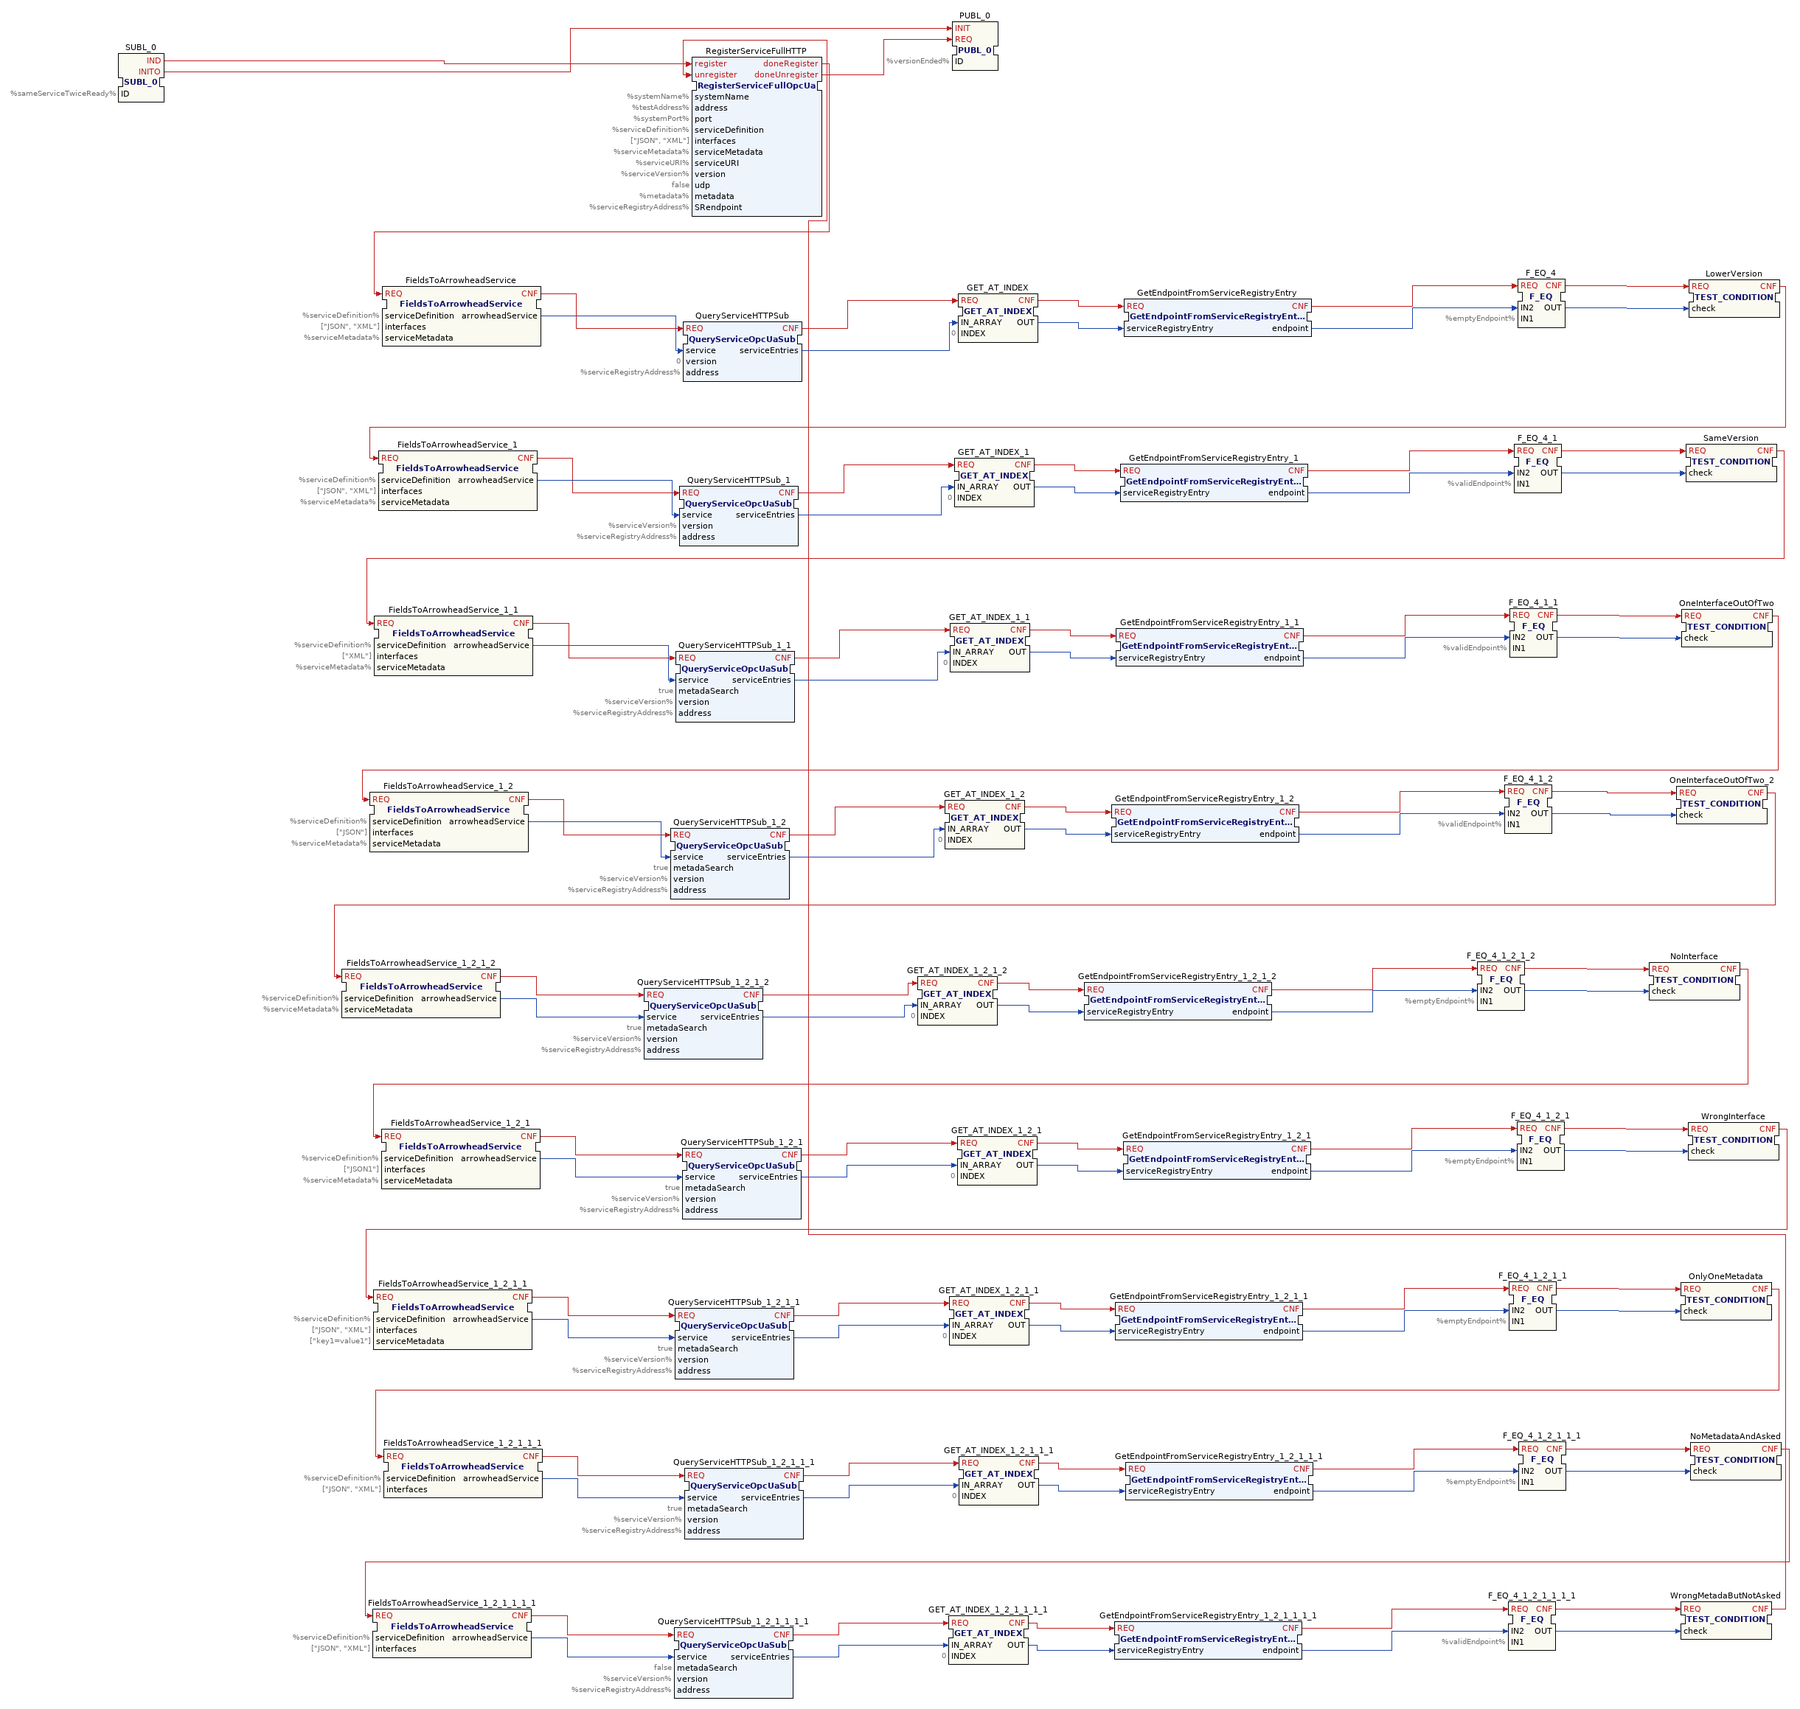
    [picture p25: application OpcUaTest5VersionAndMetadata]
    FBS
      FieldsToArrowheadService : FieldsToArrowheadService(serviceDefinition := %serviceDefinition%, interfaces := ["JSON", "XML"], serviceMetadata := %serviceMetadata%);
      GET_AT_INDEX : GET_AT_INDEX(INDEX := 0);
      F_EQ_4 : F_EQ(IN1 := %emptyEndpoint%);
      LowerVersion : TEST_CONDITION;
      FieldsToArrowheadService_1 : FieldsToArrowheadService(serviceDefinition := %serviceDefinition%, interfaces := ["JSON", "XML"], serviceMetadata := %serviceMetadata%);
      SameVersion : TEST_CONDITION;
      GET_AT_INDEX_1 : GET_AT_INDEX(INDEX := 0);
      F_EQ_4_1 : F_EQ(IN1 := %validEndpoint%);
      OneInterfaceOutOfTwo : TEST_CONDITION;
      F_EQ_4_1_1 : F_EQ(IN1 := %validEndpoint%);
      FieldsToArrowheadService_1_1 : FieldsToArrowheadService(serviceDefinition := %serviceDefinition%, interfaces := ["XML"], serviceMetadata := %serviceMetadata%);
      GET_AT_INDEX_1_1 : GET_AT_INDEX(INDEX := 0);
      OneInterfaceOutOfTwo_2 : TEST_CONDITION;
      F_EQ_4_1_2 : F_EQ(IN1 := %validEndpoint%);
      FieldsToArrowheadService_1_2 : FieldsToArrowheadService(serviceDefinition := %serviceDefinition%, interfaces := ["JSON"], serviceMetadata := %serviceMetadata%);
      GET_AT_INDEX_1_2 : GET_AT_INDEX(INDEX := 0);
      WrongInterface : TEST_CONDITION;
      GET_AT_INDEX_1_2_1 : GET_AT_INDEX(INDEX := 0);
      FieldsToArrowheadService_1_2_1 : FieldsToArrowheadService(serviceDefinition := %serviceDefinition%, interfaces := ["JSON1"], serviceMetadata := %serviceMetadata%);
      F_EQ_4_1_2_1 : F_EQ(IN1 := %emptyEndpoint%);
      SUBL_0 : SUBL_0(ID := %sameServiceTwiceReady%);
      OnlyOneMetadata : TEST_CONDITION;
      F_EQ_4_1_2_1_1 : F_EQ(IN1 := %emptyEndpoint%);
      FieldsToArrowheadService_1_2_1_1 : FieldsToArrowheadService(serviceDefinition := %serviceDefinition%, interfaces := ["JSON", "XML"], serviceMetadata := ["key1=value1"]);
      GET_AT_INDEX_1_2_1_1 : GET_AT_INDEX(INDEX := 0);
      FieldsToArrowheadService_1_2_1_1_1 : FieldsToArrowheadService(serviceDefinition := %serviceDefinition%, interfaces := ["JSON", "XML"]);
      F_EQ_4_1_2_1_1_1 : F_EQ(IN1 := %emptyEndpoint%);
      GET_AT_INDEX_1_2_1_1_1 : GET_AT_INDEX(INDEX := 0);
      NoMetadataAndAsked : TEST_CONDITION;
      F_EQ_4_1_2_1_2 : F_EQ(IN1 := %emptyEndpoint%);
      GET_AT_INDEX_1_2_1_2 : GET_AT_INDEX(INDEX := 0);
      FieldsToArrowheadService_1_2_1_2 : FieldsToArrowheadService(serviceDefinition := %serviceDefinition%, serviceMetadata := %serviceMetadata%);
      NoInterface : TEST_CONDITION;
      GET_AT_INDEX_1_2_1_1_1_1 : GET_AT_INDEX(INDEX := 0);
      F_EQ_4_1_2_1_1_1_1 : F_EQ(IN1 := %validEndpoint%);
      WrongMetadaButNotAsked : TEST_CONDITION;
      FieldsToArrowheadService_1_2_1_1_1_1 : FieldsToArrowheadService(serviceDefinition := %serviceDefinition%, interfaces := ["JSON", "XML"]);
      PUBL_0 : PUBL_0(ID := %versionEnded%);
    END_FBS
    SUBAPPS
      GetEndpointFromServiceRegistryEntry : GetEndpointFromServiceRegistryEntry;
      GetEndpointFromServiceRegistryEntry_1 : GetEndpointFromServiceRegistryEntry;
      GetEndpointFromServiceRegistryEntry_1_1 : GetEndpointFromServiceRegistryEntry;
      GetEndpointFromServiceRegistryEntry_1_2 : GetEndpointFromServiceRegistryEntry;
      GetEndpointFromServiceRegistryEntry_1_2_1 : GetEndpointFromServiceRegistryEntry;
      GetEndpointFromServiceRegistryEntry_1_2_1_1 : GetEndpointFromServiceRegistryEntry;
      GetEndpointFromServiceRegistryEntry_1_2_1_1_1 : GetEndpointFromServiceRegistryEntry;
      GetEndpointFromServiceRegistryEntry_1_2_1_2 : GetEndpointFromServiceRegistryEntry;
      GetEndpointFromServiceRegistryEntry_1_2_1_1_1_1 : GetEndpointFromServiceRegistryEntry;
      RegisterServiceFullHTTP : RegisterServiceFullOpcUa(systemName := %systemName%, address := %testAddress%, port := %systemPort%, serviceDefinition := %serviceDefinition%, interfaces := ["JSON", "XML"], serviceMetadata := %serviceMetadata%, serviceURI := %serviceURI%, version := %serviceVersion%, udp := false, metadata := %metadata%, SRendpoint := %serviceRegistryAddress%);
      QueryServiceHTTPSub : QueryServiceOpcUaSub(version := 0, address := %serviceRegistryAddress%);
      QueryServiceHTTPSub_1 : QueryServiceOpcUaSub(version := %serviceVersion%, address := %serviceRegistryAddress%);
      QueryServiceHTTPSub_1_1 : QueryServiceOpcUaSub(metadaSearch := true, version := %serviceVersion%, address := %serviceRegistryAddress%);
      QueryServiceHTTPSub_1_2 : QueryServiceOpcUaSub(metadaSearch := true, version := %serviceVersion%, address := %serviceRegistryAddress%);
      QueryServiceHTTPSub_1_2_1_2 : QueryServiceOpcUaSub(metadaSearch := true, version := %serviceVersion%, address := %serviceRegistryAddress%);
      QueryServiceHTTPSub_1_2_1 : QueryServiceOpcUaSub(metadaSearch := true, version := %serviceVersion%, address := %serviceRegistryAddress%);
      QueryServiceHTTPSub_1_2_1_1 : QueryServiceOpcUaSub(metadaSearch := true, version := %serviceVersion%, address := %serviceRegistryAddress%);
      QueryServiceHTTPSub_1_2_1_1_1 : QueryServiceOpcUaSub(metadaSearch := true, version := %serviceVersion%, address := %serviceRegistryAddress%);
      QueryServiceHTTPSub_1_2_1_1_1_1 : QueryServiceOpcUaSub(metadaSearch := false, version := %serviceVersion%, address := %serviceRegistryAddress%);
    END_SUBAPPS
    EVENT_CONNECTIONS
      GET_AT_INDEX.CNF TO GetEndpointFromServiceRegistryEntry.REQ;
      F_EQ_4.CNF TO LowerVersion.REQ;
      GetEndpointFromServiceRegistryEntry.CNF TO F_EQ_4.REQ;
      F_EQ_4_1.CNF TO SameVersion.REQ;
      GetEndpointFromServiceRegistryEntry_1.CNF TO F_EQ_4_1.REQ;
      GET_AT_INDEX_1.CNF TO GetEndpointFromServiceRegistryEntry_1.REQ;
      GET_AT_INDEX_1_1.CNF TO GetEndpointFromServiceRegistryEntry_1_1.REQ;
      GetEndpointFromServiceRegistryEntry_1_1.CNF TO F_EQ_4_1_1.REQ;
      F_EQ_4_1_1.CNF TO OneInterfaceOutOfTwo.REQ;
      GET_AT_INDEX_1_2.CNF TO GetEndpointFromServiceRegistryEntry_1_2.REQ;
      GetEndpointFromServiceRegistryEntry_1_2.CNF TO F_EQ_4_1_2.REQ;
      F_EQ_4_1_2.CNF TO OneInterfaceOutOfTwo_2.REQ;
      F_EQ_4_1_2_1.CNF TO WrongInterface.REQ;
      GET_AT_INDEX_1_2_1.CNF TO GetEndpointFromServiceRegistryEntry_1_2_1.REQ;
      GetEndpointFromServiceRegistryEntry_1_2_1.CNF TO F_EQ_4_1_2_1.REQ;
      GET_AT_INDEX_1_2_1_1.CNF TO GetEndpointFromServiceRegistryEntry_1_2_1_1.REQ;
      GetEndpointFromServiceRegistryEntry_1_2_1_1.CNF TO F_EQ_4_1_2_1_1.REQ;
      F_EQ_4_1_2_1_1.CNF TO OnlyOneMetadata.REQ;
      F_EQ_4_1_2_1_1_1.CNF TO NoMetadataAndAsked.REQ;
      GetEndpointFromServiceRegistryEntry_1_2_1_1_1.CNF TO F_EQ_4_1_2_1_1_1.REQ;
      GET_AT_INDEX_1_2_1_1_1.CNF TO GetEndpointFromServiceRegistryEntry_1_2_1_1_1.REQ;
      F_EQ_4_1_2_1_2.CNF TO NoInterface.REQ;
      GET_AT_INDEX_1_2_1_2.CNF TO GetEndpointFromServiceRegistryEntry_1_2_1_2.REQ;
      GetEndpointFromServiceRegistryEntry_1_2_1_2.CNF TO F_EQ_4_1_2_1_2.REQ;
      GET_AT_INDEX_1_2_1_1_1_1.CNF TO GetEndpointFromServiceRegistryEntry_1_2_1_1_1_1.REQ;
      F_EQ_4_1_2_1_1_1_1.CNF TO WrongMetadaButNotAsked.REQ;
      GetEndpointFromServiceRegistryEntry_1_2_1_1_1_1.CNF TO F_EQ_4_1_2_1_1_1_1.REQ;
      LowerVersion.CNF TO FieldsToArrowheadService_1.REQ;
      SameVersion.CNF TO FieldsToArrowheadService_1_1.REQ;
      OneInterfaceOutOfTwo.CNF TO FieldsToArrowheadService_1_2.REQ;
      OneInterfaceOutOfTwo_2.CNF TO FieldsToArrowheadService_1_2_1_2.REQ;
      NoInterface.CNF TO FieldsToArrowheadService_1_2_1.REQ;
      WrongInterface.CNF TO FieldsToArrowheadService_1_2_1_1.REQ;
      OnlyOneMetadata.CNF TO FieldsToArrowheadService_1_2_1_1_1.REQ;
      NoMetadataAndAsked.CNF TO FieldsToArrowheadService_1_2_1_1_1_1.REQ;
      SUBL_0.IND TO RegisterServiceFullHTTP.register;
      WrongMetadaButNotAsked.CNF TO RegisterServiceFullHTTP.unregister;
      RegisterServiceFullHTTP.doneRegister TO FieldsToArrowheadService.REQ;
      FieldsToArrowheadService.CNF TO QueryServiceHTTPSub.REQ;
      QueryServiceHTTPSub.CNF TO GET_AT_INDEX.REQ;
      FieldsToArrowheadService_1.CNF TO QueryServiceHTTPSub_1.REQ;
      QueryServiceHTTPSub_1.CNF TO GET_AT_INDEX_1.REQ;
      FieldsToArrowheadService_1_1.CNF TO QueryServiceHTTPSub_1_1.REQ;
      QueryServiceHTTPSub_1_1.CNF TO GET_AT_INDEX_1_1.REQ;
      FieldsToArrowheadService_1_2.CNF TO QueryServiceHTTPSub_1_2.REQ;
      QueryServiceHTTPSub_1_2.CNF TO GET_AT_INDEX_1_2.REQ;
      FieldsToArrowheadService_1_2_1_2.CNF TO QueryServiceHTTPSub_1_2_1_2.REQ;
      QueryServiceHTTPSub_1_2_1_2.CNF TO GET_AT_INDEX_1_2_1_2.REQ;
      FieldsToArrowheadService_1_2_1.CNF TO QueryServiceHTTPSub_1_2_1.REQ;
      QueryServiceHTTPSub_1_2_1.CNF TO GET_AT_INDEX_1_2_1.REQ;
      FieldsToArrowheadService_1_2_1_1.CNF TO QueryServiceHTTPSub_1_2_1_1.REQ;
      QueryServiceHTTPSub_1_2_1_1.CNF TO GET_AT_INDEX_1_2_1_1.REQ;
      FieldsToArrowheadService_1_2_1_1_1.CNF TO QueryServiceHTTPSub_1_2_1_1_1.REQ;
      QueryServiceHTTPSub_1_2_1_1_1.CNF TO GET_AT_INDEX_1_2_1_1_1.REQ;
      FieldsToArrowheadService_1_2_1_1_1_1.CNF TO QueryServiceHTTPSub_1_2_1_1_1_1.REQ;
      QueryServiceHTTPSub_1_2_1_1_1_1.CNF TO GET_AT_INDEX_1_2_1_1_1_1.REQ;
      SUBL_0.INITO TO PUBL_0.INIT;
      RegisterServiceFullHTTP.doneUnregister TO PUBL_0.REQ;
    END_CONNECTIONS
    DATA_CONNECTIONS
      GET_AT_INDEX.OUT TO GetEndpointFromServiceRegistryEntry.serviceRegistryEntry;
      F_EQ_4.OUT TO LowerVersion.check;
      GetEndpointFromServiceRegistryEntry.endpoint TO F_EQ_4.IN2;
      GetEndpointFromServiceRegistryEntry_1.endpoint TO F_EQ_4_1.IN2;
      F_EQ_4_1.OUT TO SameVersion.check;
      GET_AT_INDEX_1.OUT TO GetEndpointFromServiceRegistryEntry_1.serviceRegistryEntry;
      GET_AT_INDEX_1_1.OUT TO GetEndpointFromServiceRegistryEntry_1_1.serviceRegistryEntry;
      F_EQ_4_1_1.OUT TO OneInterfaceOutOfTwo.check;
      GetEndpointFromServiceRegistryEntry_1_1.endpoint TO F_EQ_4_1_1.IN2;
      GET_AT_INDEX_1_2.OUT TO GetEndpointFromServiceRegistryEntry_1_2.serviceRegistryEntry;
      F_EQ_4_1_2.OUT TO OneInterfaceOutOfTwo_2.check;
      GetEndpointFromServiceRegistryEntry_1_2.endpoint TO F_EQ_4_1_2.IN2;
      GetEndpointFromServiceRegistryEntry_1_2_1.endpoint TO F_EQ_4_1_2_1.IN2;
      F_EQ_4_1_2_1.OUT TO WrongInterface.check;
      GET_AT_INDEX_1_2_1.OUT TO GetEndpointFromServiceRegistryEntry_1_2_1.serviceRegistryEntry;
      F_EQ_4_1_2_1_1.OUT TO OnlyOneMetadata.check;
      GET_AT_INDEX_1_2_1_1.OUT TO GetEndpointFromServiceRegistryEntry_1_2_1_1.serviceRegistryEntry;
      GetEndpointFromServiceRegistryEntry_1_2_1_1.endpoint TO F_EQ_4_1_2_1_1.IN2;
      F_EQ_4_1_2_1_1_1.OUT TO NoMetadataAndAsked.check;
      GET_AT_INDEX_1_2_1_1_1.OUT TO GetEndpointFromServiceRegistryEntry_1_2_1_1_1.serviceRegistryEntry;
      GetEndpointFromServiceRegistryEntry_1_2_1_1_1.endpoint TO F_EQ_4_1_2_1_1_1.IN2;
      F_EQ_4_1_2_1_2.OUT TO NoInterface.check;
      GET_AT_INDEX_1_2_1_2.OUT TO GetEndpointFromServiceRegistryEntry_1_2_1_2.serviceRegistryEntry;
      GetEndpointFromServiceRegistryEntry_1_2_1_2.endpoint TO F_EQ_4_1_2_1_2.IN2;
      GET_AT_INDEX_1_2_1_1_1_1.OUT TO GetEndpointFromServiceRegistryEntry_1_2_1_1_1_1.serviceRegistryEntry;
      GetEndpointFromServiceRegistryEntry_1_2_1_1_1_1.endpoint TO F_EQ_4_1_2_1_1_1_1.IN2;
      F_EQ_4_1_2_1_1_1_1.OUT TO WrongMetadaButNotAsked.check;
      FieldsToArrowheadService.arrowheadService TO QueryServiceHTTPSub.service;
      QueryServiceHTTPSub.serviceEntries TO GET_AT_INDEX.IN_ARRAY;
      FieldsToArrowheadService_1.arrowheadService TO QueryServiceHTTPSub_1.service;
      QueryServiceHTTPSub_1.serviceEntries TO GET_AT_INDEX_1.IN_ARRAY;
      FieldsToArrowheadService_1_1.arrowheadService TO QueryServiceHTTPSub_1_1.service;
      QueryServiceHTTPSub_1_1.serviceEntries TO GET_AT_INDEX_1_1.IN_ARRAY;
      FieldsToArrowheadService_1_2.arrowheadService TO QueryServiceHTTPSub_1_2.service;
      QueryServiceHTTPSub_1_2.serviceEntries TO GET_AT_INDEX_1_2.IN_ARRAY;
      FieldsToArrowheadService_1_2_1_2.arrowheadService TO QueryServiceHTTPSub_1_2_1_2.service;
      QueryServiceHTTPSub_1_2_1_2.serviceEntries TO GET_AT_INDEX_1_2_1_2.IN_ARRAY;
      FieldsToArrowheadService_1_2_1.arrowheadService TO QueryServiceHTTPSub_1_2_1.service;
      QueryServiceHTTPSub_1_2_1.serviceEntries TO GET_AT_INDEX_1_2_1.IN_ARRAY;
      FieldsToArrowheadService_1_2_1_1.arrowheadService TO QueryServiceHTTPSub_1_2_1_1.service;
      QueryServiceHTTPSub_1_2_1_1.serviceEntries TO GET_AT_INDEX_1_2_1_1.IN_ARRAY;
      FieldsToArrowheadService_1_2_1_1_1.arrowheadService TO QueryServiceHTTPSub_1_2_1_1_1.service;
      QueryServiceHTTPSub_1_2_1_1_1.serviceEntries TO GET_AT_INDEX_1_2_1_1_1.IN_ARRAY;
      FieldsToArrowheadService_1_2_1_1_1_1.arrowheadService TO QueryServiceHTTPSub_1_2_1_1_1_1.service;
      QueryServiceHTTPSub_1_2_1_1_1_1.serviceEntries TO GET_AT_INDEX_1_2_1_1_1_1.IN_ARRAY;
    END_CONNECTIONS
  END_APPLICATION
  APPLICATION OpcUaTest6RegisterMoreServiceSubApp
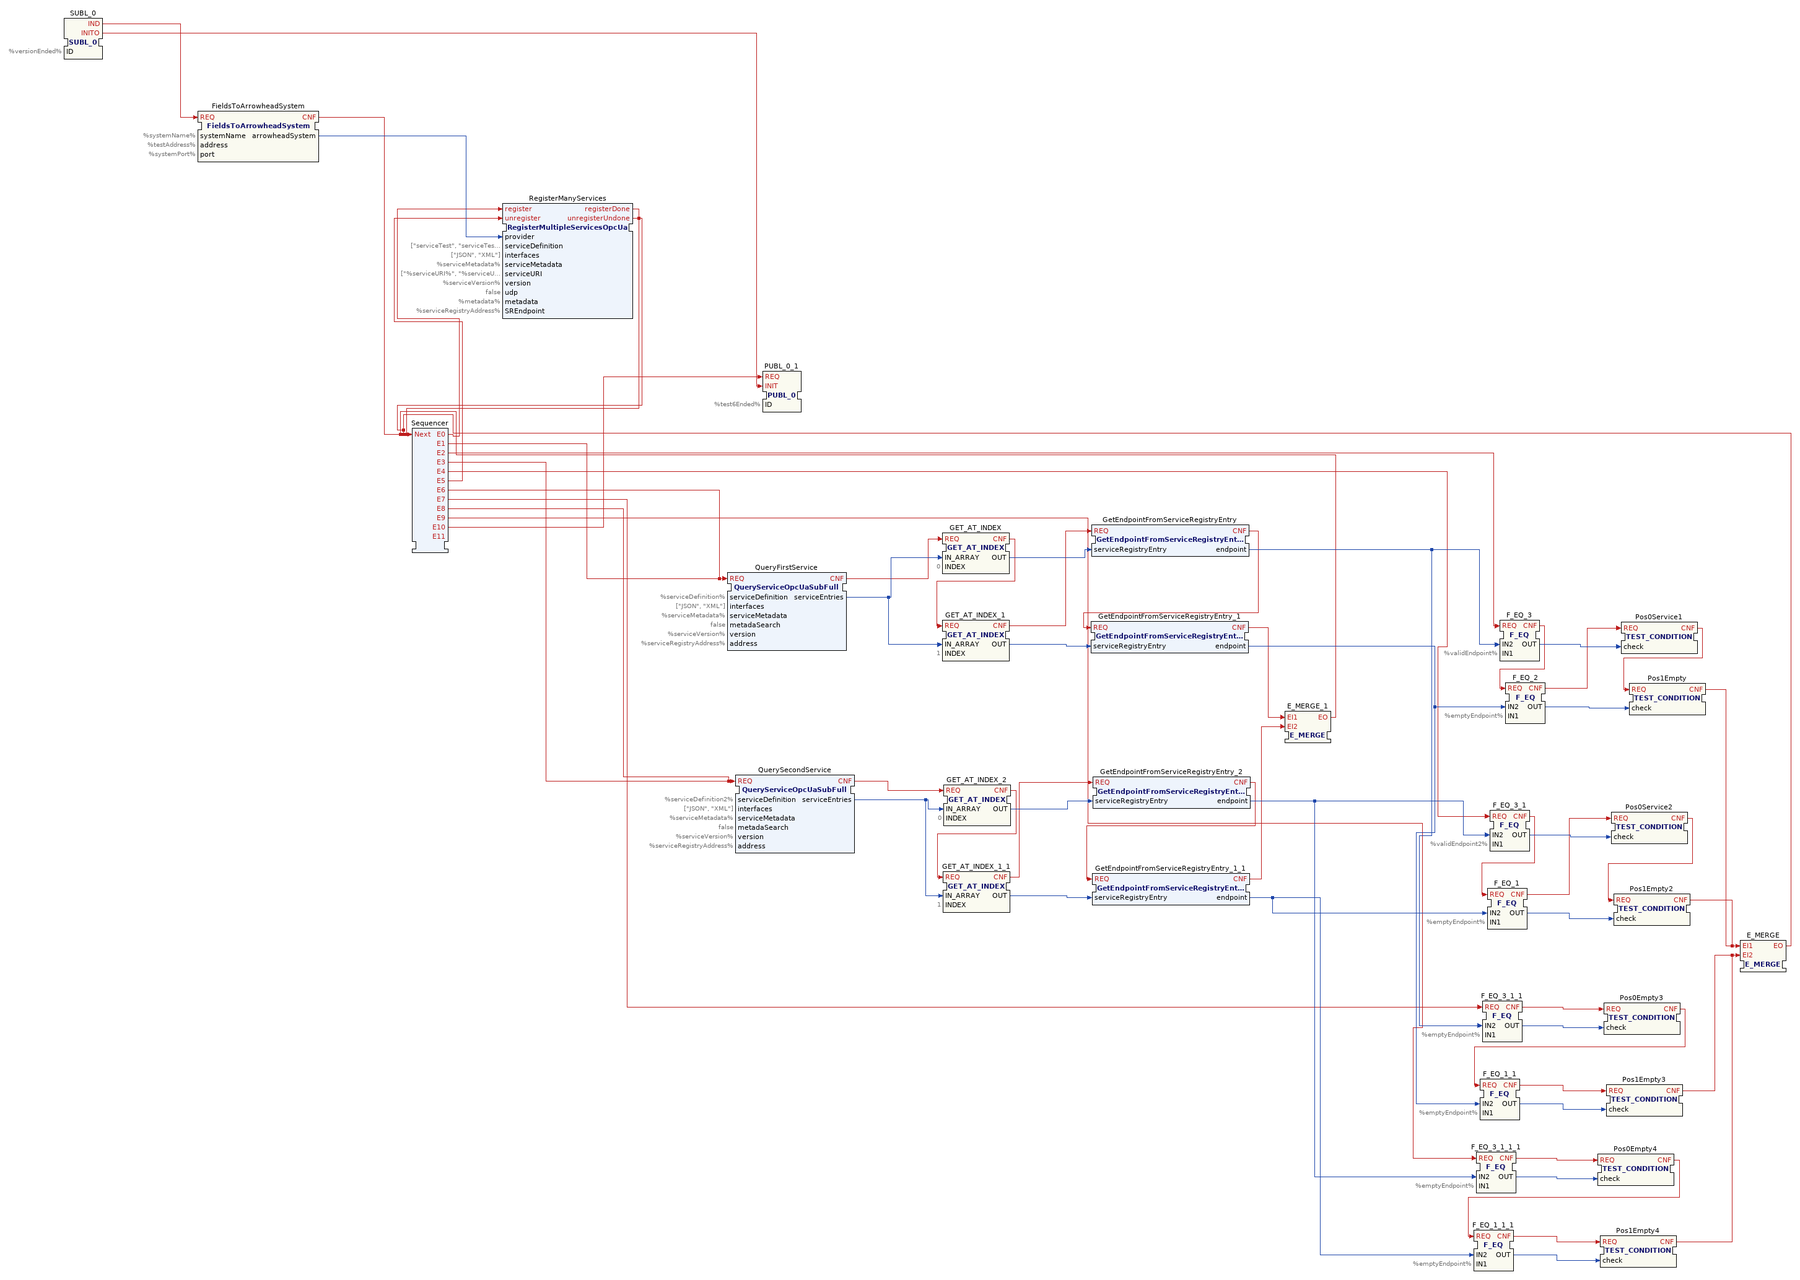
    FBS
      SUBL_0 : SUBL_0(ID := %versionEnded%);
      GET_AT_INDEX_1 : GET_AT_INDEX(INDEX := 1);
      FieldsToArrowheadSystem : FieldsToArrowheadSystem(systemName := %systemName%, address := %testAddress%, port := %systemPort%);
      F_EQ_2 : F_EQ(IN1 := %emptyEndpoint%);
      GET_AT_INDEX : GET_AT_INDEX(INDEX := 0);
      Pos1Empty2 : TEST_CONDITION;
      F_EQ_1 : F_EQ(IN1 := %emptyEndpoint%);
      Pos1Empty : TEST_CONDITION;
      GET_AT_INDEX_1_1 : GET_AT_INDEX(INDEX := 1);
      GET_AT_INDEX_2 : GET_AT_INDEX(INDEX := 0);
      Pos0Service1 : TEST_CONDITION;
      F_EQ_3 : F_EQ(IN1 := %validEndpoint%);
      F_EQ_3_1 : F_EQ(IN1 := %validEndpoint2%);
      Pos0Service2 : TEST_CONDITION;
      PUBL_0_1 : PUBL_0(ID := %test6Ended%);
      F_EQ_1_1 : F_EQ(IN1 := %emptyEndpoint%);
      F_EQ_3_1_1 : F_EQ(IN1 := %emptyEndpoint%);
      Pos1Empty3 : TEST_CONDITION;
      Pos0Empty3 : TEST_CONDITION;
      F_EQ_1_1_1 : F_EQ(IN1 := %emptyEndpoint%);
      Pos0Empty4 : TEST_CONDITION;
      Pos1Empty4 : TEST_CONDITION;
      F_EQ_3_1_1_1 : F_EQ(IN1 := %emptyEndpoint%);
      E_MERGE : E_MERGE;
      E_MERGE_1 : E_MERGE;
    END_FBS
    SUBAPPS
      GetEndpointFromServiceRegistryEntry_1 : GetEndpointFromServiceRegistryEntry;
      GetEndpointFromServiceRegistryEntry : GetEndpointFromServiceRegistryEntry;
      GetEndpointFromServiceRegistryEntry_1_1 : GetEndpointFromServiceRegistryEntry;
      GetEndpointFromServiceRegistryEntry_2 : GetEndpointFromServiceRegistryEntry;
      RegisterManyServices : RegisterMultipleServicesOpcUa(serviceDefinition := ["serviceTest", "serviceTest2"], interfaces := ["JSON", "XML"], serviceMetadata := %serviceMetadata%, serviceURI := ["%serviceURI%", "%serviceURI2%"], version := %serviceVersion%, udp := false, metadata := %metadata%, SREndpoint := %serviceRegistryAddress%);
      QueryFirstService : QueryServiceOpcUaSubFull(serviceDefinition := %serviceDefinition%, interfaces := ["JSON", "XML"], serviceMetadata := %serviceMetadata%, metadaSearch := false, version := %serviceVersion%, address := %serviceRegistryAddress%);
      QuerySecondService : QueryServiceOpcUaSubFull(serviceDefinition := %serviceDefinition2%, interfaces := ["JSON", "XML"], serviceMetadata := %serviceMetadata%, metadaSearch := false, version := %serviceVersion%, address := %serviceRegistryAddress%);
    END_SUBAPPS
    SUBAPPLICATION Sequencer
      EVENT_INPUT
        Next;
      END_EVENT
      EVENT_OUTPUT
        E0;
        E1;
        E2;
        E3;
        E4;
        E5;
        E6;
        E7;
        E8;
        E9;
        E10;
        E11;
      END_EVENT
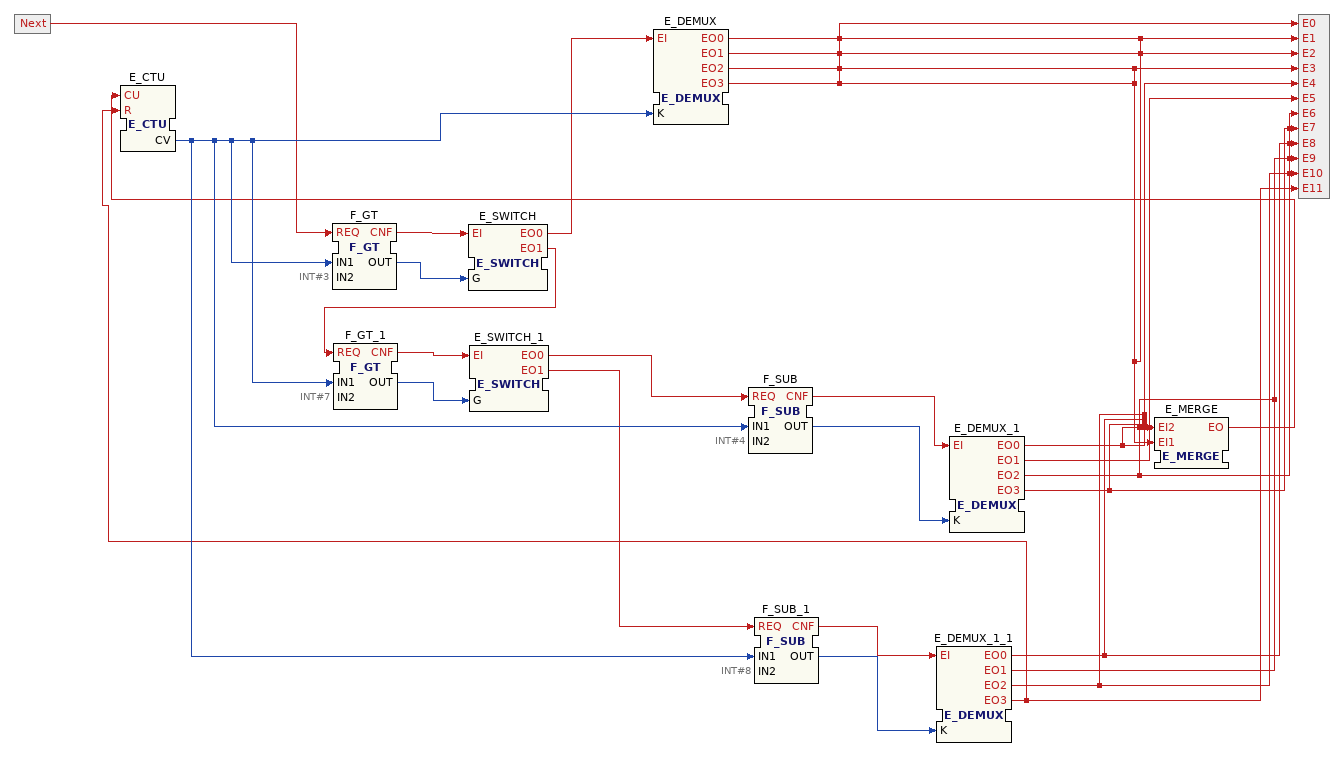
      FBS
        E_DEMUX : E_DEMUX;
        E_CTU : E_CTU;
        E_DEMUX_1 : E_DEMUX;
        E_SWITCH : E_SWITCH;
        F_GT : F_GT(IN2 := INT#3);
        E_MERGE : E_MERGE;
        F_SUB : F_SUB(IN2 := INT#4);
        E_DEMUX_1_1 : E_DEMUX;
        F_GT_1 : F_GT(IN2 := INT#7);
        F_SUB_1 : F_SUB(IN2 := INT#8);
        E_SWITCH_1 : E_SWITCH;
      END_FBS
      EVENT_CONNECTIONS
        E_DEMUX.EO0 TO E0;
        E_DEMUX.EO1 TO E1;
        E_DEMUX.EO2 TO E2;
        E_DEMUX.EO3 TO E3;
        E_DEMUX_1.EO0 TO E4;
        E_DEMUX_1.EO1 TO E5;
        E_DEMUX_1.EO2 TO E6;
        E_DEMUX_1.EO3 TO E7;
        F_GT.CNF TO E_SWITCH.EI;
        E_SWITCH.EO0 TO E_DEMUX.EI;
        E_MERGE.EO TO E_CTU.CU;
        F_SUB.CNF TO E_DEMUX_1.EI;
        E_DEMUX_1.EO0 TO E_MERGE.EI2;
        E_DEMUX_1.EO1 TO E_MERGE.EI2;
        E_DEMUX_1.EO2 TO E_MERGE.EI2;
        E_DEMUX.EO3 TO E_MERGE.EI1;
        E_DEMUX.EO2 TO E_MERGE.EI1;
        E_DEMUX.EO1 TO E_MERGE.EI1;
        E_DEMUX.EO0 TO E_MERGE.EI1;
        E_SWITCH.EO1 TO F_GT_1.REQ;
        F_GT_1.CNF TO E_SWITCH_1.EI;
        E_SWITCH_1.EO0 TO F_SUB.REQ;
        E_SWITCH_1.EO1 TO F_SUB_1.REQ;
        F_SUB_1.CNF TO E_DEMUX_1_1.EI;
        E_DEMUX_1_1.EO0 TO E8;
        E_DEMUX_1_1.EO1 TO E9;
        E_DEMUX_1_1.EO2 TO E10;
        E_DEMUX_1_1.EO3 TO E11;
        E_DEMUX_1.EO3 TO E_MERGE.EI2;
        E_DEMUX_1_1.EO0 TO E_MERGE.EI2;
        E_DEMUX_1_1.EO1 TO E_MERGE.EI2;
        E_DEMUX_1_1.EO2 TO E_MERGE.EI2;
        E_DEMUX_1_1.EO3 TO E_CTU.R;
        Next TO F_GT.REQ;
      END_CONNECTIONS
      DATA_CONNECTIONS
        E_CTU.CV TO E_DEMUX.K;
        F_GT.OUT TO E_SWITCH.G;
        F_SUB.OUT TO E_DEMUX_1.K;
        E_CTU.CV TO F_GT.IN1;
        E_CTU.CV TO F_SUB.IN1;
        E_CTU.CV TO F_SUB_1.IN1;
        E_CTU.CV TO F_GT_1.IN1;
        F_GT_1.OUT TO E_SWITCH_1.G;
        F_SUB_1.OUT TO E_DEMUX_1_1.K;
      END_CONNECTIONS
    END_SUBAPPLICATION
    EVENT_CONNECTIONS
      GET_AT_INDEX_1_1.CNF TO GetEndpointFromServiceRegistryEntry_2.REQ;
      GET_AT_INDEX.CNF TO GET_AT_INDEX_1.REQ;
      GET_AT_INDEX_2.CNF TO GET_AT_INDEX_1_1.REQ;
      GET_AT_INDEX_1.CNF TO GetEndpointFromServiceRegistryEntry.REQ;
      GetEndpointFromServiceRegistryEntry.CNF TO GetEndpointFromServiceRegistryEntry_1.REQ;
      GetEndpointFromServiceRegistryEntry_2.CNF TO GetEndpointFromServiceRegistryEntry_1_1.REQ;
      SUBL_0.IND TO FieldsToArrowheadSystem.REQ;
      F_EQ_3.CNF TO F_EQ_2.REQ;
      F_EQ_2.CNF TO Pos0Service1.REQ;
      Pos0Service1.CNF TO Pos1Empty.REQ;
      F_EQ_3_1.CNF TO F_EQ_1.REQ;
      F_EQ_1.CNF TO Pos0Service2.REQ;
      Pos0Service2.CNF TO Pos1Empty2.REQ;
      FieldsToArrowheadSystem.CNF TO Sequencer.Next;
      F_EQ_3_1_1.CNF TO Pos0Empty3.REQ;
      F_EQ_1_1.CNF TO Pos1Empty3.REQ;
      F_EQ_1_1_1.CNF TO Pos1Empty4.REQ;
      F_EQ_3_1_1_1.CNF TO Pos0Empty4.REQ;
      Pos0Empty3.CNF TO F_EQ_1_1.REQ;
      Pos0Empty4.CNF TO F_EQ_1_1_1.REQ;
      E_MERGE.EO TO Sequencer.Next;
      Pos1Empty.CNF TO E_MERGE.EI1;
      Pos1Empty2.CNF TO E_MERGE.EI1;
      Pos1Empty3.CNF TO E_MERGE.EI2;
      Pos1Empty4.CNF TO E_MERGE.EI2;
      Sequencer.E2 TO F_EQ_3.REQ;
      GetEndpointFromServiceRegistryEntry_1.CNF TO E_MERGE_1.EI1;
      GetEndpointFromServiceRegistryEntry_1_1.CNF TO E_MERGE_1.EI2;
      E_MERGE_1.EO TO Sequencer.Next;
      Sequencer.E4 TO F_EQ_3_1.REQ;
      Sequencer.E7 TO F_EQ_3_1_1.REQ;
      Sequencer.E9 TO F_EQ_3_1_1_1.REQ;
      Sequencer.E0 TO RegisterManyServices.register;
      Sequencer.E5 TO RegisterManyServices.unregister;
      RegisterManyServices.registerDone TO Sequencer.Next;
      RegisterManyServices.unregisterUndone TO Sequencer.Next;
      Sequencer.E1 TO QueryFirstService.REQ;
      Sequencer.E6 TO QueryFirstService.REQ;
      QueryFirstService.CNF TO GET_AT_INDEX.REQ;
      Sequencer.E3 TO QuerySecondService.REQ;
      Sequencer.E8 TO QuerySecondService.REQ;
      QuerySecondService.CNF TO GET_AT_INDEX_2.REQ;
      Sequencer.E10 TO PUBL_0_1.REQ;
      SUBL_0.INITO TO PUBL_0_1.INIT;
    END_CONNECTIONS
    DATA_CONNECTIONS
      GET_AT_INDEX.OUT TO GetEndpointFromServiceRegistryEntry.serviceRegistryEntry;
      GET_AT_INDEX_2.OUT TO GetEndpointFromServiceRegistryEntry_2.serviceRegistryEntry;
      F_EQ_1.OUT TO Pos1Empty2.check;
      GetEndpointFromServiceRegistryEntry_2.endpoint TO F_EQ_3_1.IN2;
      GET_AT_INDEX_1.OUT TO GetEndpointFromServiceRegistryEntry_1.serviceRegistryEntry;
      F_EQ_2.OUT TO Pos1Empty.check;
      F_EQ_3_1.OUT TO Pos0Service2.check;
      GetEndpointFromServiceRegistryEntry.endpoint TO F_EQ_3.IN2;
      GET_AT_INDEX_1_1.OUT TO GetEndpointFromServiceRegistryEntry_1_1.serviceRegistryEntry;
      F_EQ_3.OUT TO Pos0Service1.check;
      GetEndpointFromServiceRegistryEntry_1.endpoint TO F_EQ_2.IN2;
      GetEndpointFromServiceRegistryEntry_1_1.endpoint TO F_EQ_1.IN2;
      F_EQ_3_1_1.OUT TO Pos0Empty3.check;
      F_EQ_1_1.OUT TO Pos1Empty3.check;
      F_EQ_3_1_1_1.OUT TO Pos0Empty4.check;
      F_EQ_1_1_1.OUT TO Pos1Empty4.check;
      GetEndpointFromServiceRegistryEntry.endpoint TO F_EQ_3_1_1.IN2;
      GetEndpointFromServiceRegistryEntry_1.endpoint TO F_EQ_1_1.IN2;
      GetEndpointFromServiceRegistryEntry_2.endpoint TO F_EQ_3_1_1_1.IN2;
      GetEndpointFromServiceRegistryEntry_1_1.endpoint TO F_EQ_1_1_1.IN2;
      FieldsToArrowheadSystem.arrowheadSystem TO RegisterManyServices.provider;
      QueryFirstService.serviceEntries TO GET_AT_INDEX_1.IN_ARRAY;
      QueryFirstService.serviceEntries TO GET_AT_INDEX.IN_ARRAY;
      QuerySecondService.serviceEntries TO GET_AT_INDEX_1_1.IN_ARRAY;
      QuerySecondService.serviceEntries TO GET_AT_INDEX_2.IN_ARRAY;
    END_CONNECTIONS
  END_APPLICATION
  APPLICATION OpcUaTest7OrchestrationNoRules
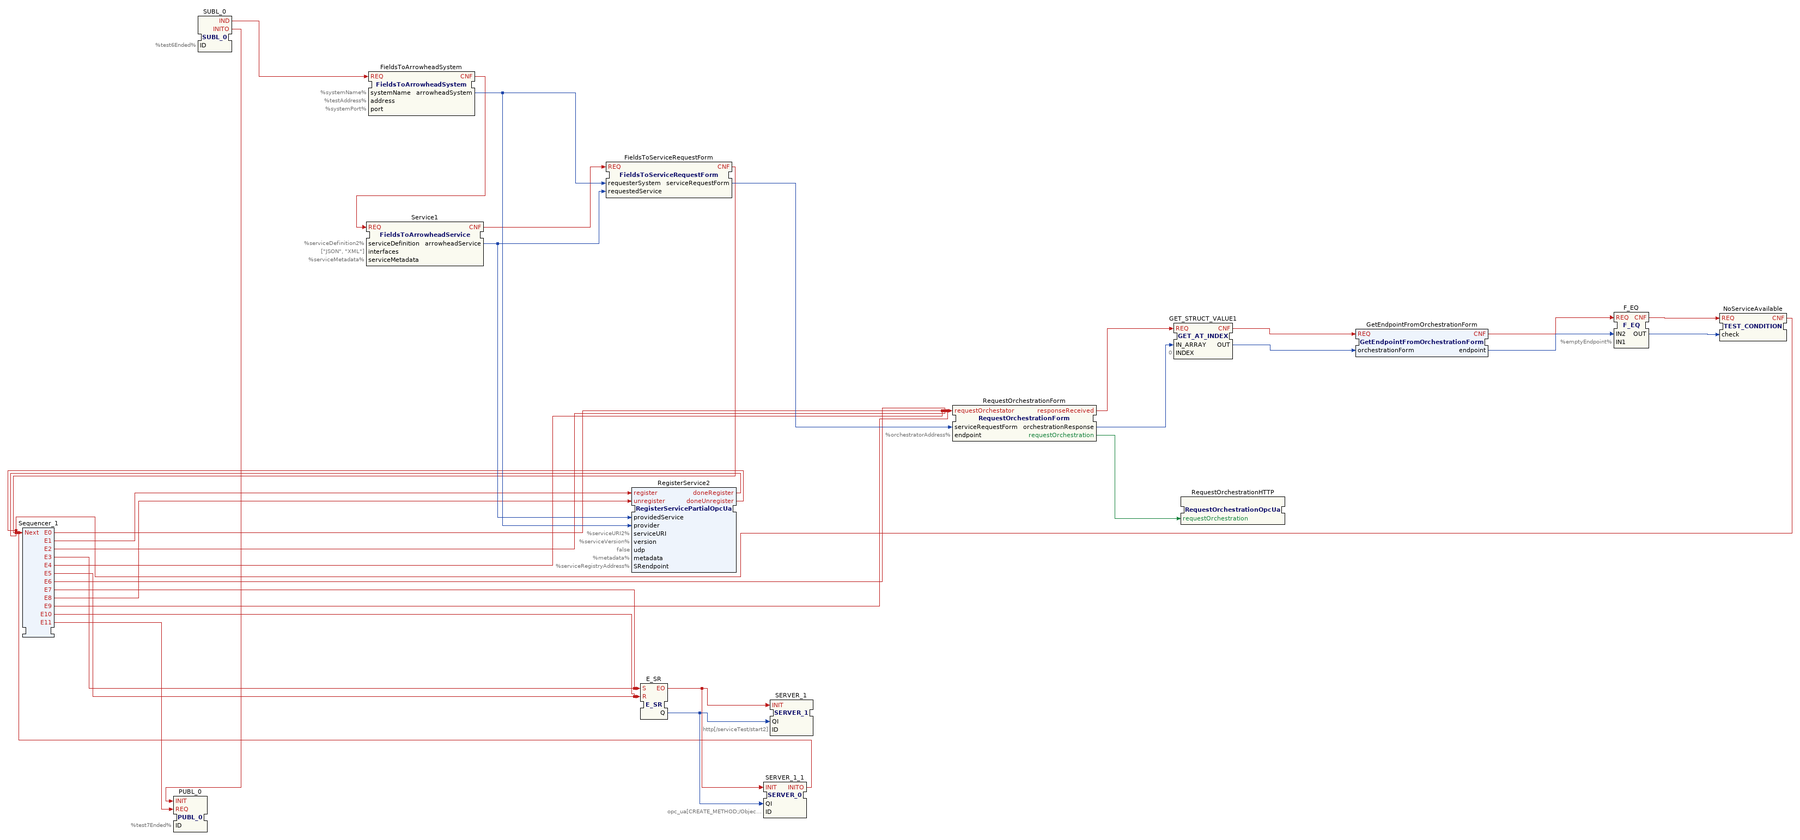
    FBS
      FieldsToServiceRequestForm : FieldsToServiceRequestForm;
      FieldsToArrowheadSystem : FieldsToArrowheadSystem(systemName := %systemName%, address := %testAddress%, port := %systemPort%);
      Service1 : FieldsToArrowheadService(serviceDefinition := %serviceDefinition2%, interfaces := ["JSON", "XML"], serviceMetadata := %serviceMetadata%);
      F_EQ : F_EQ(IN1 := %emptyEndpoint%);
      NoServiceAvailable : TEST_CONDITION;
      SERVER_1 : SERVER_1(ID := http[/serviceTest/start2]);
      E_SR : E_SR;
      SUBL_0 : SUBL_0(ID := %test6Ended%);
      PUBL_0 : PUBL_0(ID := %test7Ended%);
      GET_STRUCT_VALUE1 : GET_AT_INDEX(INDEX := 0);
      RequestOrchestrationForm : RequestOrchestrationForm(endpoint := %orchestratorAddress%);
      RequestOrchestrationHTTP : RequestOrchestrationOpcUa;
      SERVER_1_1 : SERVER_0(ID := opc_ua[CREATE_METHOD;/Objects/serviceTest/start2]);
    END_FBS
    SUBAPPS
      GetEndpointFromOrchestrationForm : GetEndpointFromOrchestrationForm;
      RegisterService2 : RegisterServicePartialOpcUa(serviceURI := %serviceURI2%, version := %serviceVersion%, udp := false, metadata := %metadata%, SRendpoint := %serviceRegistryAddress%);
    END_SUBAPPS
    SUBAPPLICATION Sequencer_1
      EVENT_INPUT
        Next;
      END_EVENT
      EVENT_OUTPUT
        E0;
        E1;
        E2;
        E3;
        E4;
        E5;
        E6;
        E7;
        E8;
        E9;
        E10;
        E11;
      END_EVENT
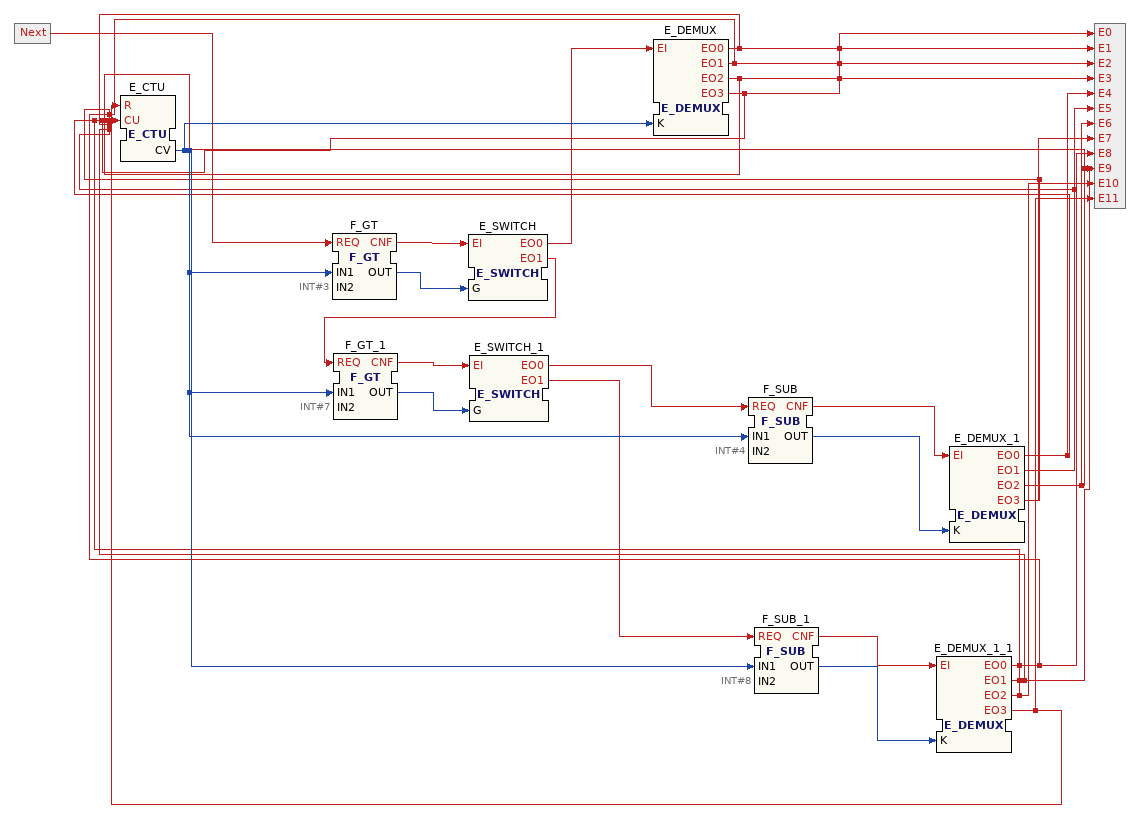
      FBS
        E_DEMUX : E_DEMUX;
        E_CTU : E_CTU;
        E_DEMUX_1 : E_DEMUX;
        E_SWITCH : E_SWITCH;
        F_GT : F_GT(IN2 := INT#3);
        F_SUB : F_SUB(IN2 := INT#4);
        E_DEMUX_1_1 : E_DEMUX;
        F_GT_1 : F_GT(IN2 := INT#7);
        F_SUB_1 : F_SUB(IN2 := INT#8);
        E_SWITCH_1 : E_SWITCH;
      END_FBS
      EVENT_CONNECTIONS
        E_DEMUX.EO0 TO E0;
        E_DEMUX.EO1 TO E1;
        E_DEMUX.EO2 TO E2;
        E_DEMUX.EO3 TO E3;
        E_DEMUX_1.EO0 TO E4;
        E_DEMUX_1.EO1 TO E5;
        E_DEMUX_1.EO2 TO E6;
        E_DEMUX_1.EO3 TO E7;
        F_GT.CNF TO E_SWITCH.EI;
        E_SWITCH.EO0 TO E_DEMUX.EI;
        F_SUB.CNF TO E_DEMUX_1.EI;
        E_SWITCH.EO1 TO F_GT_1.REQ;
        F_GT_1.CNF TO E_SWITCH_1.EI;
        E_SWITCH_1.EO0 TO F_SUB.REQ;
        E_SWITCH_1.EO1 TO F_SUB_1.REQ;
        F_SUB_1.CNF TO E_DEMUX_1_1.EI;
        E_DEMUX_1_1.EO0 TO E8;
        E_DEMUX_1_1.EO1 TO E9;
        E_DEMUX_1_1.EO2 TO E10;
        E_DEMUX_1_1.EO3 TO E11;
        E_DEMUX_1_1.EO3 TO E_CTU.R;
        Next TO F_GT.REQ;
        E_DEMUX.EO3 TO E_CTU.CU;
        E_DEMUX.EO2 TO E_CTU.CU;
        E_DEMUX.EO1 TO E_CTU.CU;
        E_DEMUX.EO0 TO E_CTU.CU;
        E_DEMUX_1_1.EO2 TO E_CTU.CU;
        E_DEMUX_1_1.EO1 TO E_CTU.CU;
        E_DEMUX_1_1.EO0 TO E_CTU.CU;
        E_DEMUX_1.EO3 TO E_CTU.CU;
        E_DEMUX_1.EO2 TO E_CTU.CU;
        E_DEMUX_1.EO1 TO E_CTU.CU;
        E_DEMUX_1.EO0 TO E_CTU.CU;
      END_CONNECTIONS
      DATA_CONNECTIONS
        E_CTU.CV TO E_DEMUX.K;
        F_GT.OUT TO E_SWITCH.G;
        F_SUB.OUT TO E_DEMUX_1.K;
        E_CTU.CV TO F_GT.IN1;
        E_CTU.CV TO F_SUB.IN1;
        E_CTU.CV TO F_SUB_1.IN1;
        E_CTU.CV TO F_GT_1.IN1;
        F_GT_1.OUT TO E_SWITCH_1.G;
        F_SUB_1.OUT TO E_DEMUX_1_1.K;
      END_CONNECTIONS
    END_SUBAPPLICATION
    EVENT_CONNECTIONS
      FieldsToArrowheadSystem.CNF TO Service1.REQ;
      Service1.CNF TO FieldsToServiceRequestForm.REQ;
      F_EQ.CNF TO NoServiceAvailable.REQ;
      GetEndpointFromOrchestrationForm.CNF TO F_EQ.REQ;
      E_SR.EO TO SERVER_1.INIT;
      SUBL_0.IND TO FieldsToArrowheadSystem.REQ;
      GET_STRUCT_VALUE1.CNF TO GetEndpointFromOrchestrationForm.REQ;
      Sequencer_1.E3 TO E_SR.S;
      Sequencer_1.E5 TO E_SR.R;
      Sequencer_1.E7 TO E_SR.S;
      Sequencer_1.E10 TO E_SR.R;
      NoServiceAvailable.CNF TO Sequencer_1.Next;
      FieldsToServiceRequestForm.CNF TO Sequencer_1.Next;
      Sequencer_1.E0 TO RequestOrchestrationForm.requestOrchestator;
      Sequencer_1.E2 TO RequestOrchestrationForm.requestOrchestator;
      Sequencer_1.E4 TO RequestOrchestrationForm.requestOrchestator;
      Sequencer_1.E6 TO RequestOrchestrationForm.requestOrchestator;
      Sequencer_1.E9 TO RequestOrchestrationForm.requestOrchestator;
      RequestOrchestrationForm.responseReceived TO GET_STRUCT_VALUE1.REQ;
      Sequencer_1.E1 TO RegisterService2.register;
      Sequencer_1.E8 TO RegisterService2.unregister;
      RegisterService2.doneRegister TO Sequencer_1.Next;
      RegisterService2.doneUnregister TO Sequencer_1.Next;
      E_SR.EO TO SERVER_1_1.INIT;
      SERVER_1_1.INITO TO Sequencer_1.Next;
      SUBL_0.INITO TO PUBL_0.INIT;
      Sequencer_1.E11 TO PUBL_0.REQ;
    END_CONNECTIONS
    DATA_CONNECTIONS
      FieldsToArrowheadSystem.arrowheadSystem TO FieldsToServiceRequestForm.requesterSystem;
      Service1.arrowheadService TO FieldsToServiceRequestForm.requestedService;
      F_EQ.OUT TO NoServiceAvailable.check;
      GetEndpointFromOrchestrationForm.endpoint TO F_EQ.IN2;
      E_SR.Q TO SERVER_1.QI;
      GET_STRUCT_VALUE1.OUT TO GetEndpointFromOrchestrationForm.orchestrationForm;
      FieldsToServiceRequestForm.serviceRequestForm TO RequestOrchestrationForm.serviceRequestForm;
      RequestOrchestrationForm.orchestrationResponse TO GET_STRUCT_VALUE1.IN_ARRAY;
      Service1.arrowheadService TO RegisterService2.providedService;
      FieldsToArrowheadSystem.arrowheadSystem TO RegisterService2.provider;
      E_SR.Q TO SERVER_1_1.QI;
    END_CONNECTIONS
    ADAPTER_CONNECTIONS
      RequestOrchestrationForm.requestOrchestration TO RequestOrchestrationHTTP.requestOrchestration;
    END_CONNECTIONS
  END_APPLICATION
  APPLICATION OpcUaTest8OrchestrationWithRules
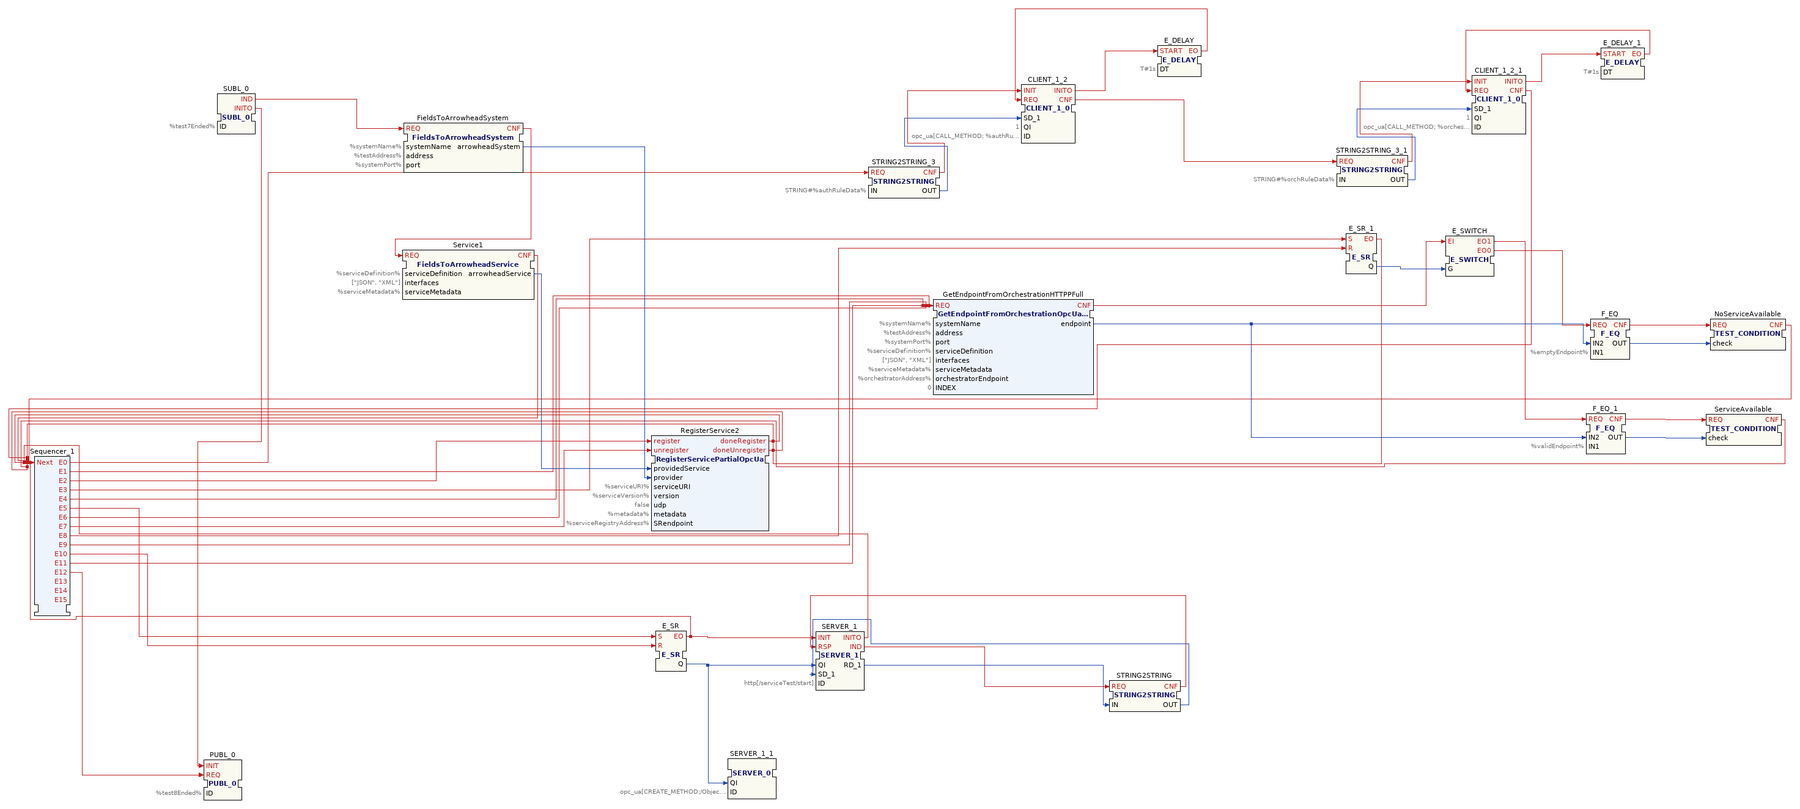
    FBS
      FieldsToArrowheadSystem : FieldsToArrowheadSystem(systemName := %systemName%, address := %testAddress%, port := %systemPort%);
      Service1 : FieldsToArrowheadService(serviceDefinition := %serviceDefinition%, interfaces := ["JSON", "XML"], serviceMetadata := %serviceMetadata%);
      F_EQ : F_EQ(IN1 := %emptyEndpoint%);
      NoServiceAvailable : TEST_CONDITION;
      SERVER_1 : SERVER_1(ID := http[/serviceTest/start]);
      E_SR : E_SR;
      SUBL_0 : SUBL_0(ID := %test7Ended%);
      PUBL_0 : PUBL_0(ID := %test8Ended%);
      F_EQ_1 : F_EQ(IN1 := %validEndpoint%);
      ServiceAvailable : TEST_CONDITION;
      E_SR_1 : E_SR;
      E_SWITCH : E_SWITCH;
      STRING2STRING : STRING2STRING;
      SERVER_1_1 : SERVER_0(ID := opc_ua[CREATE_METHOD;/Objects/serviceTest/start2]);
      E_DELAY : E_DELAY(DT := T#1s);
      E_DELAY_1 : E_DELAY(DT := T#1s);
      STRING2STRING_3 : STRING2STRING(IN := STRING#%authRuleData%);
      STRING2STRING_3_1 : STRING2STRING(IN := STRING#%orchRuleData%);
      CLIENT_1_2 : CLIENT_1_0(QI := 1, ID := opc_ua[CALL_METHOD; %authRuleEndpoint%#; /Objects/2:Authorization/2:addSystemToAuthorized]);
      CLIENT_1_2_1 : CLIENT_1_0(QI := 1, ID := opc_ua[CALL_METHOD; %orchestratorEndpoint%#; /Objects/2:Orchestrator/2:store]);
    END_FBS
    SUBAPPS
      RegisterService2 : RegisterServicePartialOpcUa(serviceURI := %serviceURI%, version := %serviceVersion%, udp := false, metadata := %metadata%, SRendpoint := %serviceRegistryAddress%);
      GetEndpointFromOrchestrationHTTPPFull : GetEndpointFromOrchestrationOpcUaFull(systemName := %systemName%, address := %testAddress%, port := %systemPort%, serviceDefinition := %serviceDefinition%, interfaces := ["JSON", "XML"], serviceMetadata := %serviceMetadata%, orchestratorEndpoint := %orchestratorAddress%, INDEX := 0);
    END_SUBAPPS
    SUBAPPLICATION Sequencer_1
      EVENT_INPUT
        Next;
      END_EVENT
      EVENT_OUTPUT
        E0;
        E1;
        E2;
        E3;
        E4;
        E5;
        E6;
        E7;
        E8;
        E9;
        E10;
        E11;
        E12;
        E13;
        E14;
        E15;
      END_EVENT
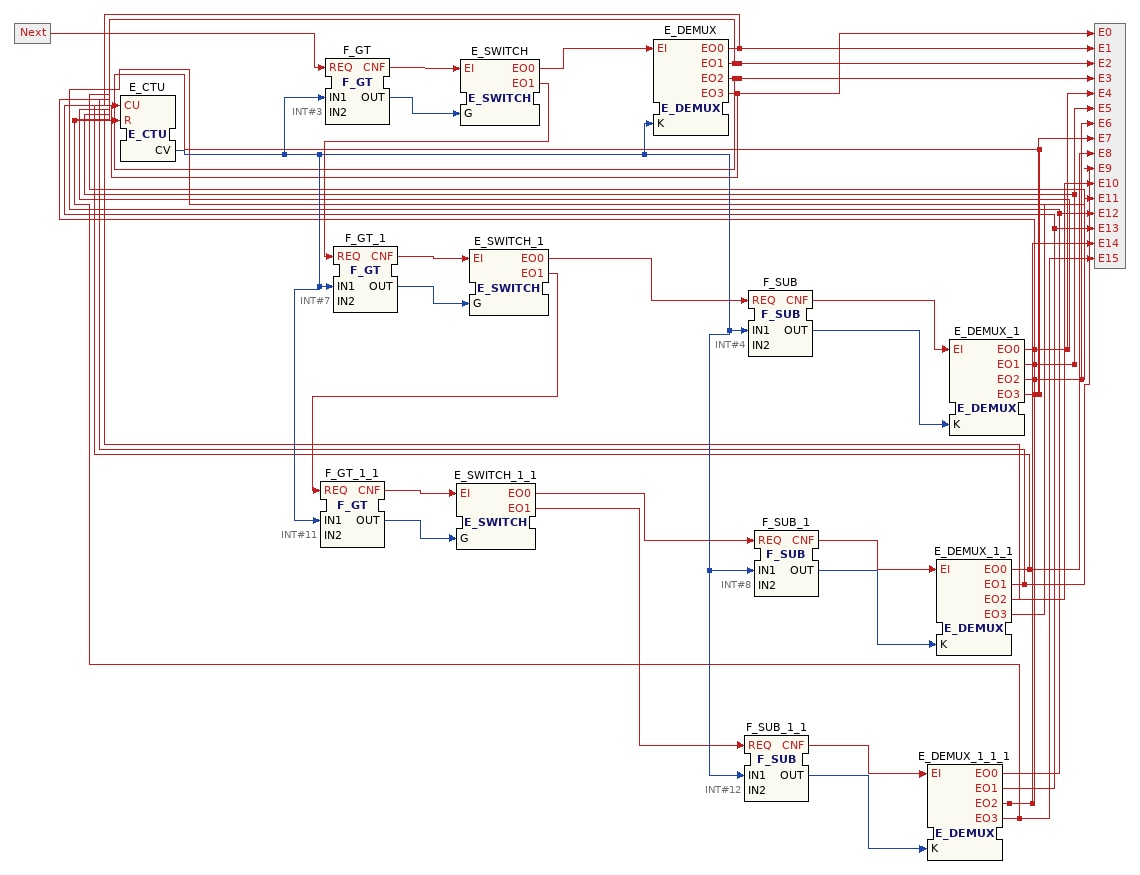
      FBS
        E_DEMUX : E_DEMUX;
        E_CTU : E_CTU;
        E_DEMUX_1 : E_DEMUX;
        E_SWITCH : E_SWITCH;
        F_GT : F_GT(IN2 := INT#3);
        F_SUB : F_SUB(IN2 := INT#4);
        E_DEMUX_1_1 : E_DEMUX;
        F_GT_1 : F_GT(IN2 := INT#7);
        F_SUB_1 : F_SUB(IN2 := INT#8);
        E_SWITCH_1 : E_SWITCH;
        F_GT_1_1 : F_GT(IN2 := INT#11);
        E_SWITCH_1_1 : E_SWITCH;
        E_DEMUX_1_1_1 : E_DEMUX;
        F_SUB_1_1 : F_SUB(IN2 := INT#12);
      END_FBS
      EVENT_CONNECTIONS
        E_DEMUX.EO0 TO E0;
        E_DEMUX.EO1 TO E1;
        E_DEMUX.EO2 TO E2;
        E_DEMUX.EO3 TO E3;
        E_DEMUX_1.EO0 TO E4;
        E_DEMUX_1.EO1 TO E5;
        E_DEMUX_1.EO2 TO E6;
        E_DEMUX_1.EO3 TO E7;
        F_GT.CNF TO E_SWITCH.EI;
        E_SWITCH.EO0 TO E_DEMUX.EI;
        F_SUB.CNF TO E_DEMUX_1.EI;
        E_SWITCH.EO1 TO F_GT_1.REQ;
        F_GT_1.CNF TO E_SWITCH_1.EI;
        E_SWITCH_1.EO0 TO F_SUB.REQ;
        F_SUB_1.CNF TO E_DEMUX_1_1.EI;
        E_DEMUX_1_1.EO0 TO E8;
        E_DEMUX_1_1.EO1 TO E9;
        E_DEMUX_1_1.EO2 TO E10;
        E_DEMUX.EO3 TO E_CTU.CU;
        E_DEMUX.EO2 TO E_CTU.CU;
        E_DEMUX.EO1 TO E_CTU.CU;
        E_DEMUX.EO0 TO E_CTU.CU;
        E_DEMUX_1_1.EO2 TO E_CTU.CU;
        E_DEMUX_1_1.EO1 TO E_CTU.CU;
        E_DEMUX_1_1.EO0 TO E_CTU.CU;
        E_DEMUX_1.EO3 TO E_CTU.CU;
        E_DEMUX_1.EO2 TO E_CTU.CU;
        E_DEMUX_1.EO1 TO E_CTU.CU;
        E_DEMUX_1.EO0 TO E_CTU.CU;
        F_GT_1_1.CNF TO E_SWITCH_1_1.EI;
        F_SUB_1_1.CNF TO E_DEMUX_1_1_1.EI;
        E_DEMUX_1_1_1.EO0 TO E12;
        E_DEMUX_1_1_1.EO1 TO E13;
        E_DEMUX_1_1_1.EO2 TO E14;
        E_DEMUX_1_1_1.EO3 TO E15;
        E_SWITCH_1.EO1 TO F_GT_1_1.REQ;
        E_SWITCH_1_1.EO0 TO F_SUB_1.REQ;
        E_SWITCH_1_1.EO1 TO F_SUB_1_1.REQ;
        E_DEMUX_1_1_1.EO3 TO E_CTU.R;
        E_DEMUX_1_1_1.EO0 TO E_CTU.CU;
        E_DEMUX_1_1_1.EO1 TO E_CTU.CU;
        E_DEMUX_1_1_1.EO2 TO E_CTU.CU;
        E_DEMUX_1_1_1.EO3 TO E_CTU.CU;
        E_DEMUX_1_1.EO3 TO E11;
        E_DEMUX_1_1.EO3 TO E_CTU.CU;
        Next TO F_GT.REQ;
      END_CONNECTIONS
      DATA_CONNECTIONS
        E_CTU.CV TO E_DEMUX.K;
        F_GT.OUT TO E_SWITCH.G;
        F_SUB.OUT TO E_DEMUX_1.K;
        E_CTU.CV TO F_GT.IN1;
        E_CTU.CV TO F_SUB.IN1;
        E_CTU.CV TO F_SUB_1.IN1;
        E_CTU.CV TO F_GT_1.IN1;
        F_GT_1.OUT TO E_SWITCH_1.G;
        F_SUB_1.OUT TO E_DEMUX_1_1.K;
        F_GT_1_1.OUT TO E_SWITCH_1_1.G;
        F_SUB_1_1.OUT TO E_DEMUX_1_1_1.K;
        E_CTU.CV TO F_SUB_1_1.IN1;
        E_CTU.CV TO F_GT_1_1.IN1;
      END_CONNECTIONS
    END_SUBAPPLICATION
    EVENT_CONNECTIONS
      F_EQ.CNF TO NoServiceAvailable.REQ;
      E_SR.EO TO SERVER_1.INIT;
      SUBL_0.IND TO FieldsToArrowheadSystem.REQ;
      NoServiceAvailable.CNF TO Sequencer_1.Next;
      FieldsToArrowheadSystem.CNF TO Service1.REQ;
      F_EQ_1.CNF TO ServiceAvailable.REQ;
      E_SWITCH.EO1 TO F_EQ_1.REQ;
      E_SWITCH.EO0 TO F_EQ.REQ;
      E_SR_1.EO TO Sequencer_1.Next;
      SERVER_1.INITO TO Sequencer_1.Next;
      SERVER_1.IND TO STRING2STRING.REQ;
      STRING2STRING.CNF TO SERVER_1.RSP;
      ServiceAvailable.CNF TO Sequencer_1.Next;
      Sequencer_1.E3 TO E_SR_1.S;
      Sequencer_1.E5 TO E_SR.S;
      Sequencer_1.E8 TO E_SR_1.R;
      Sequencer_1.E10 TO E_SR.R;
      Service1.CNF TO Sequencer_1.Next;
      Sequencer_1.E2 TO RegisterService2.register;
      Sequencer_1.E7 TO RegisterService2.unregister;
      RegisterService2.doneRegister TO Sequencer_1.Next;
      RegisterService2.doneUnregister TO Sequencer_1.Next;
      Sequencer_1.E11 TO GetEndpointFromOrchestrationHTTPPFull.REQ;
      Sequencer_1.E9 TO GetEndpointFromOrchestrationHTTPPFull.REQ;
      Sequencer_1.E6 TO GetEndpointFromOrchestrationHTTPPFull.REQ;
      Sequencer_1.E4 TO GetEndpointFromOrchestrationHTTPPFull.REQ;
      Sequencer_1.E1 TO GetEndpointFromOrchestrationHTTPPFull.REQ;
      GetEndpointFromOrchestrationHTTPPFull.CNF TO E_SWITCH.EI;
      SUBL_0.INITO TO PUBL_0.INIT;
      Sequencer_1.E12 TO PUBL_0.REQ;
      Sequencer_1.E0 TO STRING2STRING_3.REQ;
      E_SR.EO TO Sequencer_1.Next;
      STRING2STRING_3.CNF TO CLIENT_1_2.INIT;
      E_DELAY.EO TO CLIENT_1_2.REQ;
      CLIENT_1_2.INITO TO E_DELAY.START;
      CLIENT_1_2.CNF TO STRING2STRING_3_1.REQ;
      STRING2STRING_3_1.CNF TO CLIENT_1_2_1.INIT;
      E_DELAY_1.EO TO CLIENT_1_2_1.REQ;
      CLIENT_1_2_1.INITO TO E_DELAY_1.START;
      CLIENT_1_2_1.CNF TO Sequencer_1.Next;
    END_CONNECTIONS
    DATA_CONNECTIONS
      F_EQ.OUT TO NoServiceAvailable.check;
      E_SR.Q TO SERVER_1.QI;
      F_EQ_1.OUT TO ServiceAvailable.check;
      E_SR_1.Q TO E_SWITCH.G;
      SERVER_1.RD_1 TO STRING2STRING.IN;
      STRING2STRING.OUT TO SERVER_1.SD_1;
      E_SR.Q TO SERVER_1_1.QI;
      Service1.arrowheadService TO RegisterService2.providedService;
      FieldsToArrowheadSystem.arrowheadSystem TO RegisterService2.provider;
      GetEndpointFromOrchestrationHTTPPFull.endpoint TO F_EQ_1.IN2;
      GetEndpointFromOrchestrationHTTPPFull.endpoint TO F_EQ.IN2;
      STRING2STRING_3.OUT TO CLIENT_1_2.SD_1;
      STRING2STRING_3_1.OUT TO CLIENT_1_2_1.SD_1;
    END_CONNECTIONS
  END_APPLICATION
  APPLICATION OpcUaTest9PublishSubscribe
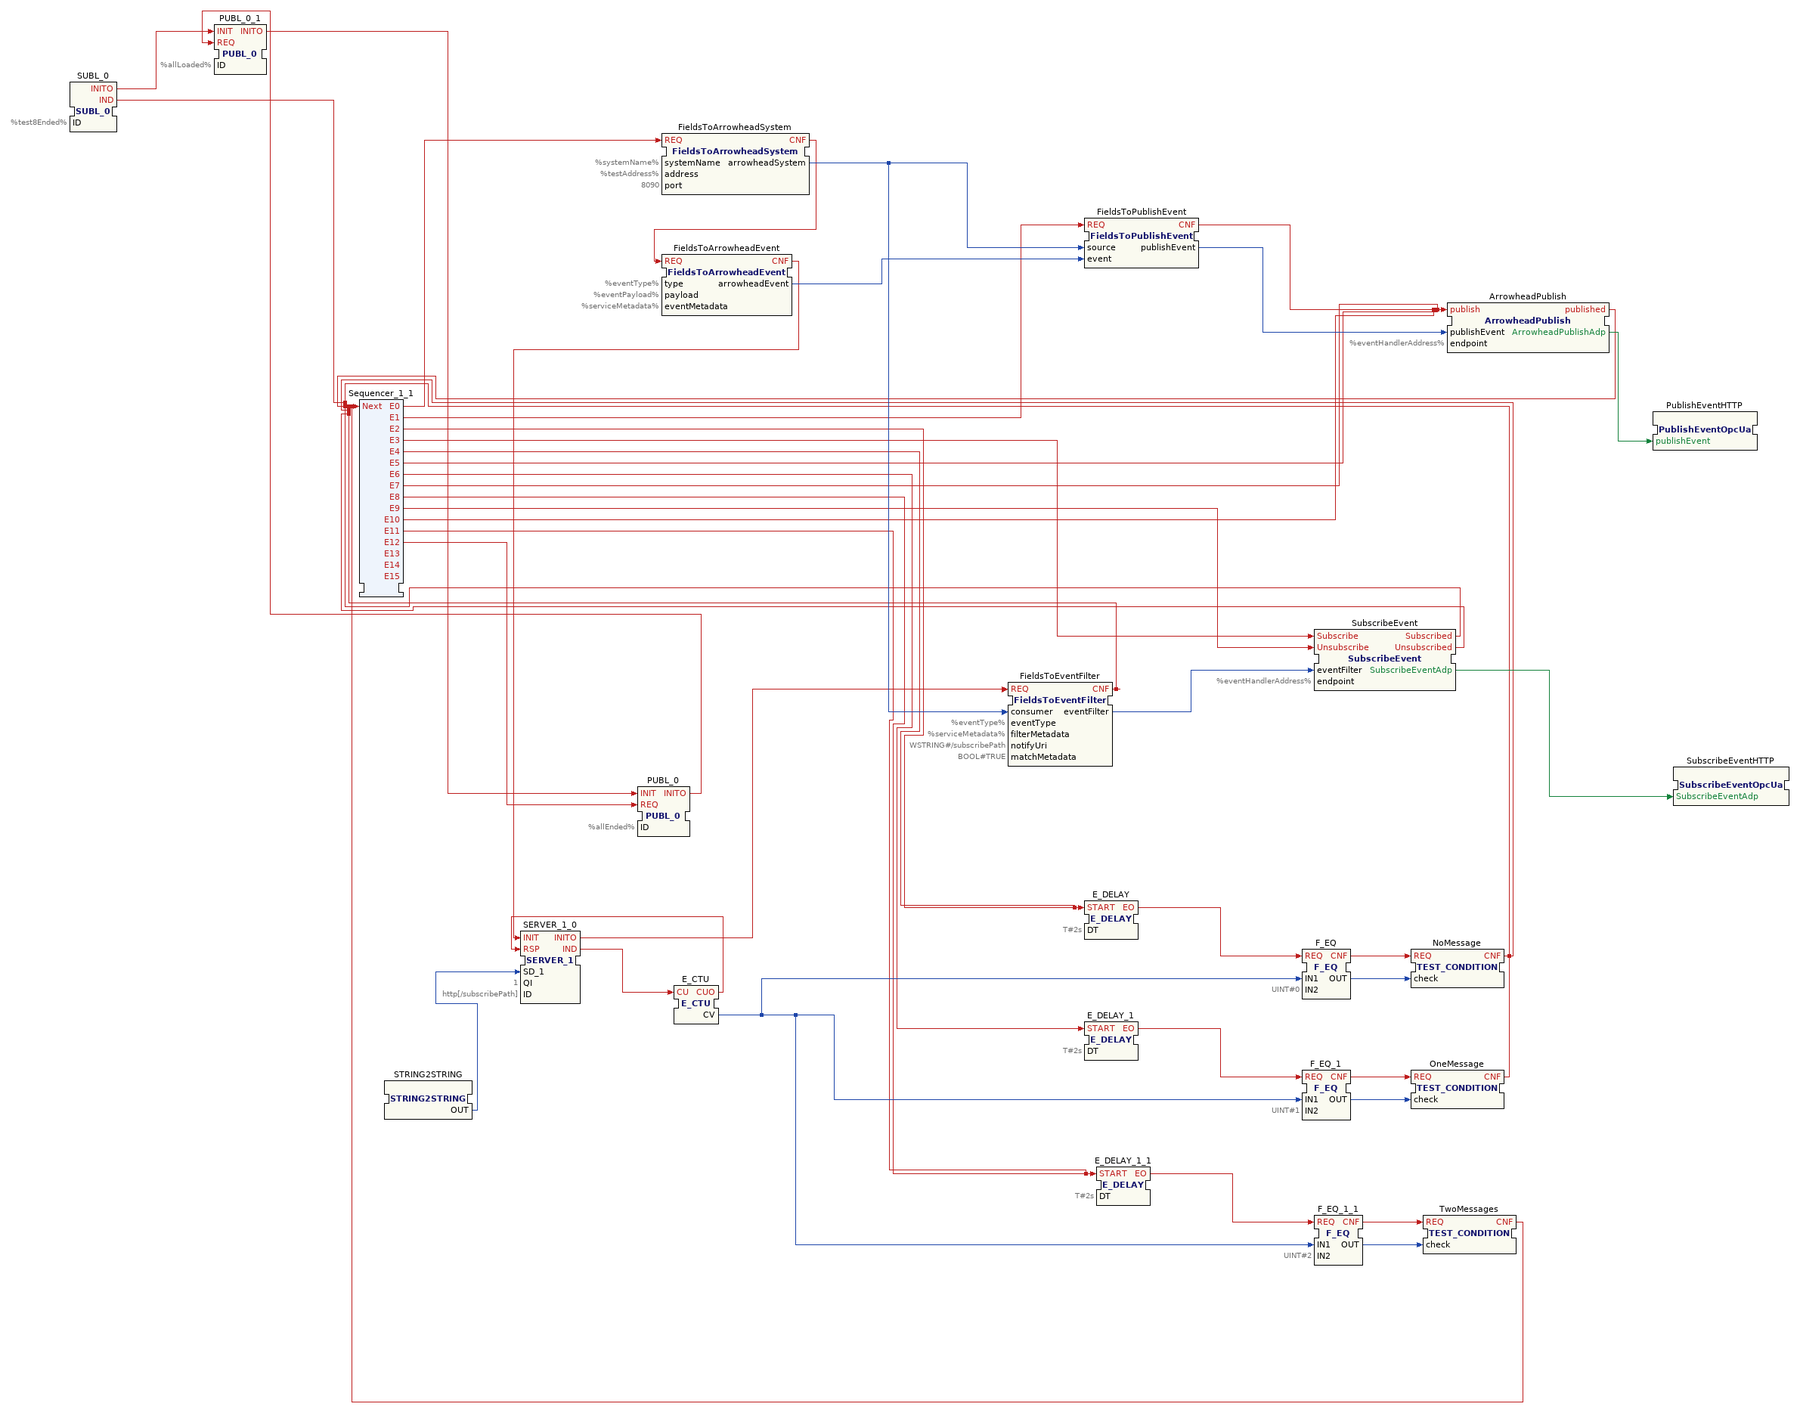
    FBS
      FieldsToPublishEvent : FieldsToPublishEvent;
      FieldsToArrowheadSystem : FieldsToArrowheadSystem(systemName := %systemName%, address := %testAddress%, port := 8090);
      ArrowheadPublish : ArrowheadPublish(endpoint := %eventHandlerAddress%);
      PublishEventHTTP : PublishEventOpcUa;
      FieldsToArrowheadEvent : FieldsToArrowheadEvent(type := %eventType%, payload := %eventPayload%, eventMetadata := %serviceMetadata%);
      FieldsToEventFilter : FieldsToEventFilter(eventType := %eventType%, filterMetadata := %serviceMetadata%, notifyUri := WSTRING#/subscribePath, matchMetadata := BOOL#TRUE);
      SubscribeEvent : SubscribeEvent(endpoint := %eventHandlerAddress%);
      SubscribeEventHTTP : SubscribeEventOpcUa;
      E_CTU : E_CTU;
      F_EQ : F_EQ(IN2 := UINT#0);
      E_DELAY : E_DELAY(DT := T#2s);
      NoMessage : TEST_CONDITION;
      F_EQ_1 : F_EQ(IN2 := UINT#1);
      OneMessage : TEST_CONDITION;
      E_DELAY_1 : E_DELAY(DT := T#2s);
      E_DELAY_1_1 : E_DELAY(DT := T#2s);
      F_EQ_1_1 : F_EQ(IN2 := UINT#2);
      TwoMessages : TEST_CONDITION;
      SUBL_0 : SUBL_0(ID := %test8Ended%);
      PUBL_0_1 : PUBL_0(ID := %allLoaded%);
      PUBL_0 : PUBL_0(ID := %allEnded%);
      SERVER_1_0 : SERVER_1(QI := 1, ID := http[/subscribePath]);
      STRING2STRING : STRING2STRING;
    END_FBS
    SUBAPPLICATION Sequencer_1_1
      EVENT_INPUT
        Next;
      END_EVENT
      EVENT_OUTPUT
        E0;
        E1;
        E2;
        E3;
        E4;
        E5;
        E6;
        E7;
        E8;
        E9;
        E10;
        E11;
        E12;
        E13;
        E14;
        E15;
      END_EVENT
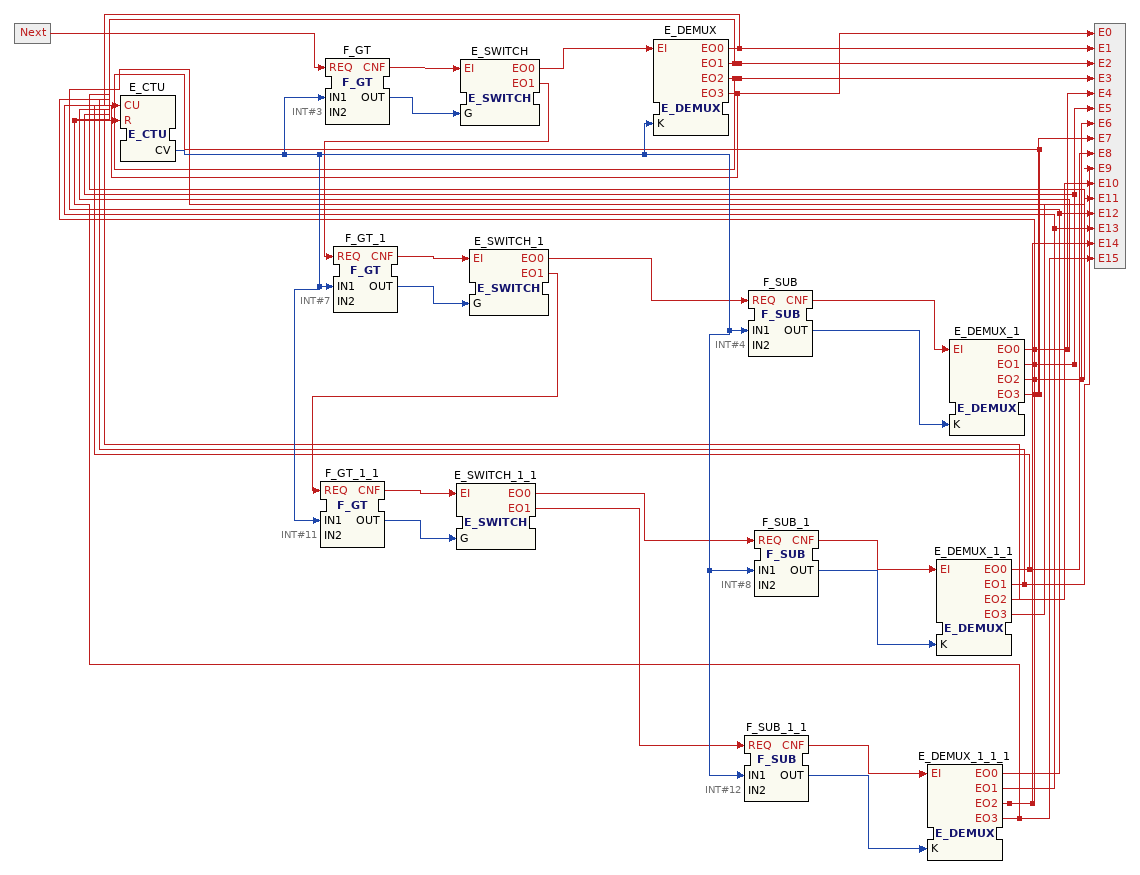
      FBS
        E_DEMUX : E_DEMUX;
        E_CTU : E_CTU;
        E_DEMUX_1 : E_DEMUX;
        E_SWITCH : E_SWITCH;
        F_GT : F_GT(IN2 := INT#3);
        F_SUB : F_SUB(IN2 := INT#4);
        E_DEMUX_1_1 : E_DEMUX;
        F_GT_1 : F_GT(IN2 := INT#7);
        F_SUB_1 : F_SUB(IN2 := INT#8);
        E_SWITCH_1 : E_SWITCH;
        F_GT_1_1 : F_GT(IN2 := INT#11);
        E_SWITCH_1_1 : E_SWITCH;
        E_DEMUX_1_1_1 : E_DEMUX;
        F_SUB_1_1 : F_SUB(IN2 := INT#12);
      END_FBS
      EVENT_CONNECTIONS
        E_DEMUX.EO0 TO E0;
        E_DEMUX.EO1 TO E1;
        E_DEMUX.EO2 TO E2;
        E_DEMUX.EO3 TO E3;
        E_DEMUX_1.EO0 TO E4;
        E_DEMUX_1.EO1 TO E5;
        E_DEMUX_1.EO2 TO E6;
        E_DEMUX_1.EO3 TO E7;
        F_GT.CNF TO E_SWITCH.EI;
        E_SWITCH.EO0 TO E_DEMUX.EI;
        F_SUB.CNF TO E_DEMUX_1.EI;
        E_SWITCH.EO1 TO F_GT_1.REQ;
        F_GT_1.CNF TO E_SWITCH_1.EI;
        E_SWITCH_1.EO0 TO F_SUB.REQ;
        F_SUB_1.CNF TO E_DEMUX_1_1.EI;
        E_DEMUX_1_1.EO0 TO E8;
        E_DEMUX_1_1.EO1 TO E9;
        E_DEMUX_1_1.EO2 TO E10;
        E_DEMUX.EO3 TO E_CTU.CU;
        E_DEMUX.EO2 TO E_CTU.CU;
        E_DEMUX.EO1 TO E_CTU.CU;
        E_DEMUX.EO0 TO E_CTU.CU;
        E_DEMUX_1_1.EO2 TO E_CTU.CU;
        E_DEMUX_1_1.EO1 TO E_CTU.CU;
        E_DEMUX_1_1.EO0 TO E_CTU.CU;
        E_DEMUX_1.EO3 TO E_CTU.CU;
        E_DEMUX_1.EO2 TO E_CTU.CU;
        E_DEMUX_1.EO1 TO E_CTU.CU;
        E_DEMUX_1.EO0 TO E_CTU.CU;
        F_GT_1_1.CNF TO E_SWITCH_1_1.EI;
        F_SUB_1_1.CNF TO E_DEMUX_1_1_1.EI;
        E_DEMUX_1_1_1.EO0 TO E12;
        E_DEMUX_1_1_1.EO1 TO E13;
        E_DEMUX_1_1_1.EO2 TO E14;
        E_DEMUX_1_1_1.EO3 TO E15;
        E_SWITCH_1.EO1 TO F_GT_1_1.REQ;
        E_SWITCH_1_1.EO0 TO F_SUB_1.REQ;
        E_SWITCH_1_1.EO1 TO F_SUB_1_1.REQ;
        E_DEMUX_1_1_1.EO3 TO E_CTU.R;
        E_DEMUX_1_1_1.EO0 TO E_CTU.CU;
        E_DEMUX_1_1_1.EO1 TO E_CTU.CU;
        E_DEMUX_1_1_1.EO2 TO E_CTU.CU;
        E_DEMUX_1_1_1.EO3 TO E_CTU.CU;
        E_DEMUX_1_1.EO3 TO E11;
        E_DEMUX_1_1.EO3 TO E_CTU.CU;
        Next TO F_GT.REQ;
      END_CONNECTIONS
      DATA_CONNECTIONS
        E_CTU.CV TO E_DEMUX.K;
        F_GT.OUT TO E_SWITCH.G;
        F_SUB.OUT TO E_DEMUX_1.K;
        E_CTU.CV TO F_GT.IN1;
        E_CTU.CV TO F_SUB.IN1;
        E_CTU.CV TO F_SUB_1.IN1;
        E_CTU.CV TO F_GT_1.IN1;
        F_GT_1.OUT TO E_SWITCH_1.G;
        F_SUB_1.OUT TO E_DEMUX_1_1.K;
        F_GT_1_1.OUT TO E_SWITCH_1_1.G;
        F_SUB_1_1.OUT TO E_DEMUX_1_1_1.K;
        E_CTU.CV TO F_SUB_1_1.IN1;
        E_CTU.CV TO F_GT_1_1.IN1;
      END_CONNECTIONS
    END_SUBAPPLICATION
    EVENT_CONNECTIONS
      FieldsToPublishEvent.CNF TO ArrowheadPublish.publish;
      FieldsToArrowheadSystem.CNF TO FieldsToArrowheadEvent.REQ;
      E_DELAY.EO TO F_EQ.REQ;
      F_EQ.CNF TO NoMessage.REQ;
      E_DELAY_1.EO TO F_EQ_1.REQ;
      F_EQ_1.CNF TO OneMessage.REQ;
      E_DELAY_1_1.EO TO F_EQ_1_1.REQ;
      F_EQ_1_1.CNF TO TwoMessages.REQ;
      Sequencer_1_1.E0 TO FieldsToArrowheadSystem.REQ;
      Sequencer_1_1.E1 TO FieldsToPublishEvent.REQ;
      Sequencer_1_1.E2 TO E_DELAY.START;
      Sequencer_1_1.E3 TO SubscribeEvent.Subscribe;
      Sequencer_1_1.E4 TO E_DELAY.START;
      Sequencer_1_1.E5 TO ArrowheadPublish.publish;
      Sequencer_1_1.E6 TO E_DELAY_1.START;
      Sequencer_1_1.E7 TO ArrowheadPublish.publish;
      Sequencer_1_1.E8 TO E_DELAY_1_1.START;
      Sequencer_1_1.E9 TO SubscribeEvent.Unsubscribe;
      Sequencer_1_1.E10 TO ArrowheadPublish.publish;
      TwoMessages.CNF TO Sequencer_1_1.Next;
      OneMessage.CNF TO Sequencer_1_1.Next;
      NoMessage.CNF TO Sequencer_1_1.Next;
      FieldsToEventFilter.CNF TO Sequencer_1_1.Next;
      Sequencer_1_1.E11 TO E_DELAY_1_1.START;
      ArrowheadPublish.published TO Sequencer_1_1.Next;
      SubscribeEvent.Subscribed TO Sequencer_1_1.Next;
      SubscribeEvent.Unsubscribed TO Sequencer_1_1.Next;
      SUBL_0.INITO TO PUBL_0_1.INIT;
      SUBL_0.IND TO Sequencer_1_1.Next;
      PUBL_0_1.INITO TO PUBL_0.INIT;
      Sequencer_1_1.E12 TO PUBL_0.REQ;
      PUBL_0.INITO TO PUBL_0_1.REQ;
      FieldsToArrowheadEvent.CNF TO SERVER_1_0.INIT;
      E_CTU.CUO TO SERVER_1_0.RSP;
      SERVER_1_0.INITO TO FieldsToEventFilter.REQ;
      SERVER_1_0.IND TO E_CTU.CU;
    END_CONNECTIONS
    DATA_CONNECTIONS
      FieldsToArrowheadSystem.arrowheadSystem TO FieldsToPublishEvent.source;
      FieldsToPublishEvent.publishEvent TO ArrowheadPublish.publishEvent;
      FieldsToArrowheadEvent.arrowheadEvent TO FieldsToPublishEvent.event;
      FieldsToEventFilter.eventFilter TO SubscribeEvent.eventFilter;
      FieldsToArrowheadSystem.arrowheadSystem TO FieldsToEventFilter.consumer;
      E_CTU.CV TO F_EQ.IN1;
      F_EQ.OUT TO NoMessage.check;
      E_CTU.CV TO F_EQ_1.IN1;
      F_EQ_1.OUT TO OneMessage.check;
      F_EQ_1_1.OUT TO TwoMessages.check;
      E_CTU.CV TO F_EQ_1_1.IN1;
      STRING2STRING.OUT TO SERVER_1_0.SD_1;
    END_CONNECTIONS
    ADAPTER_CONNECTIONS
      ArrowheadPublish.ArrowheadPublishAdp TO PublishEventHTTP.publishEvent;
      SubscribeEvent.SubscribeEventAdp TO SubscribeEventHTTP.SubscribeEventAdp;
    END_CONNECTIONS
  END_APPLICATION
  APPLICATION HTTPTest9PublishSubscribe
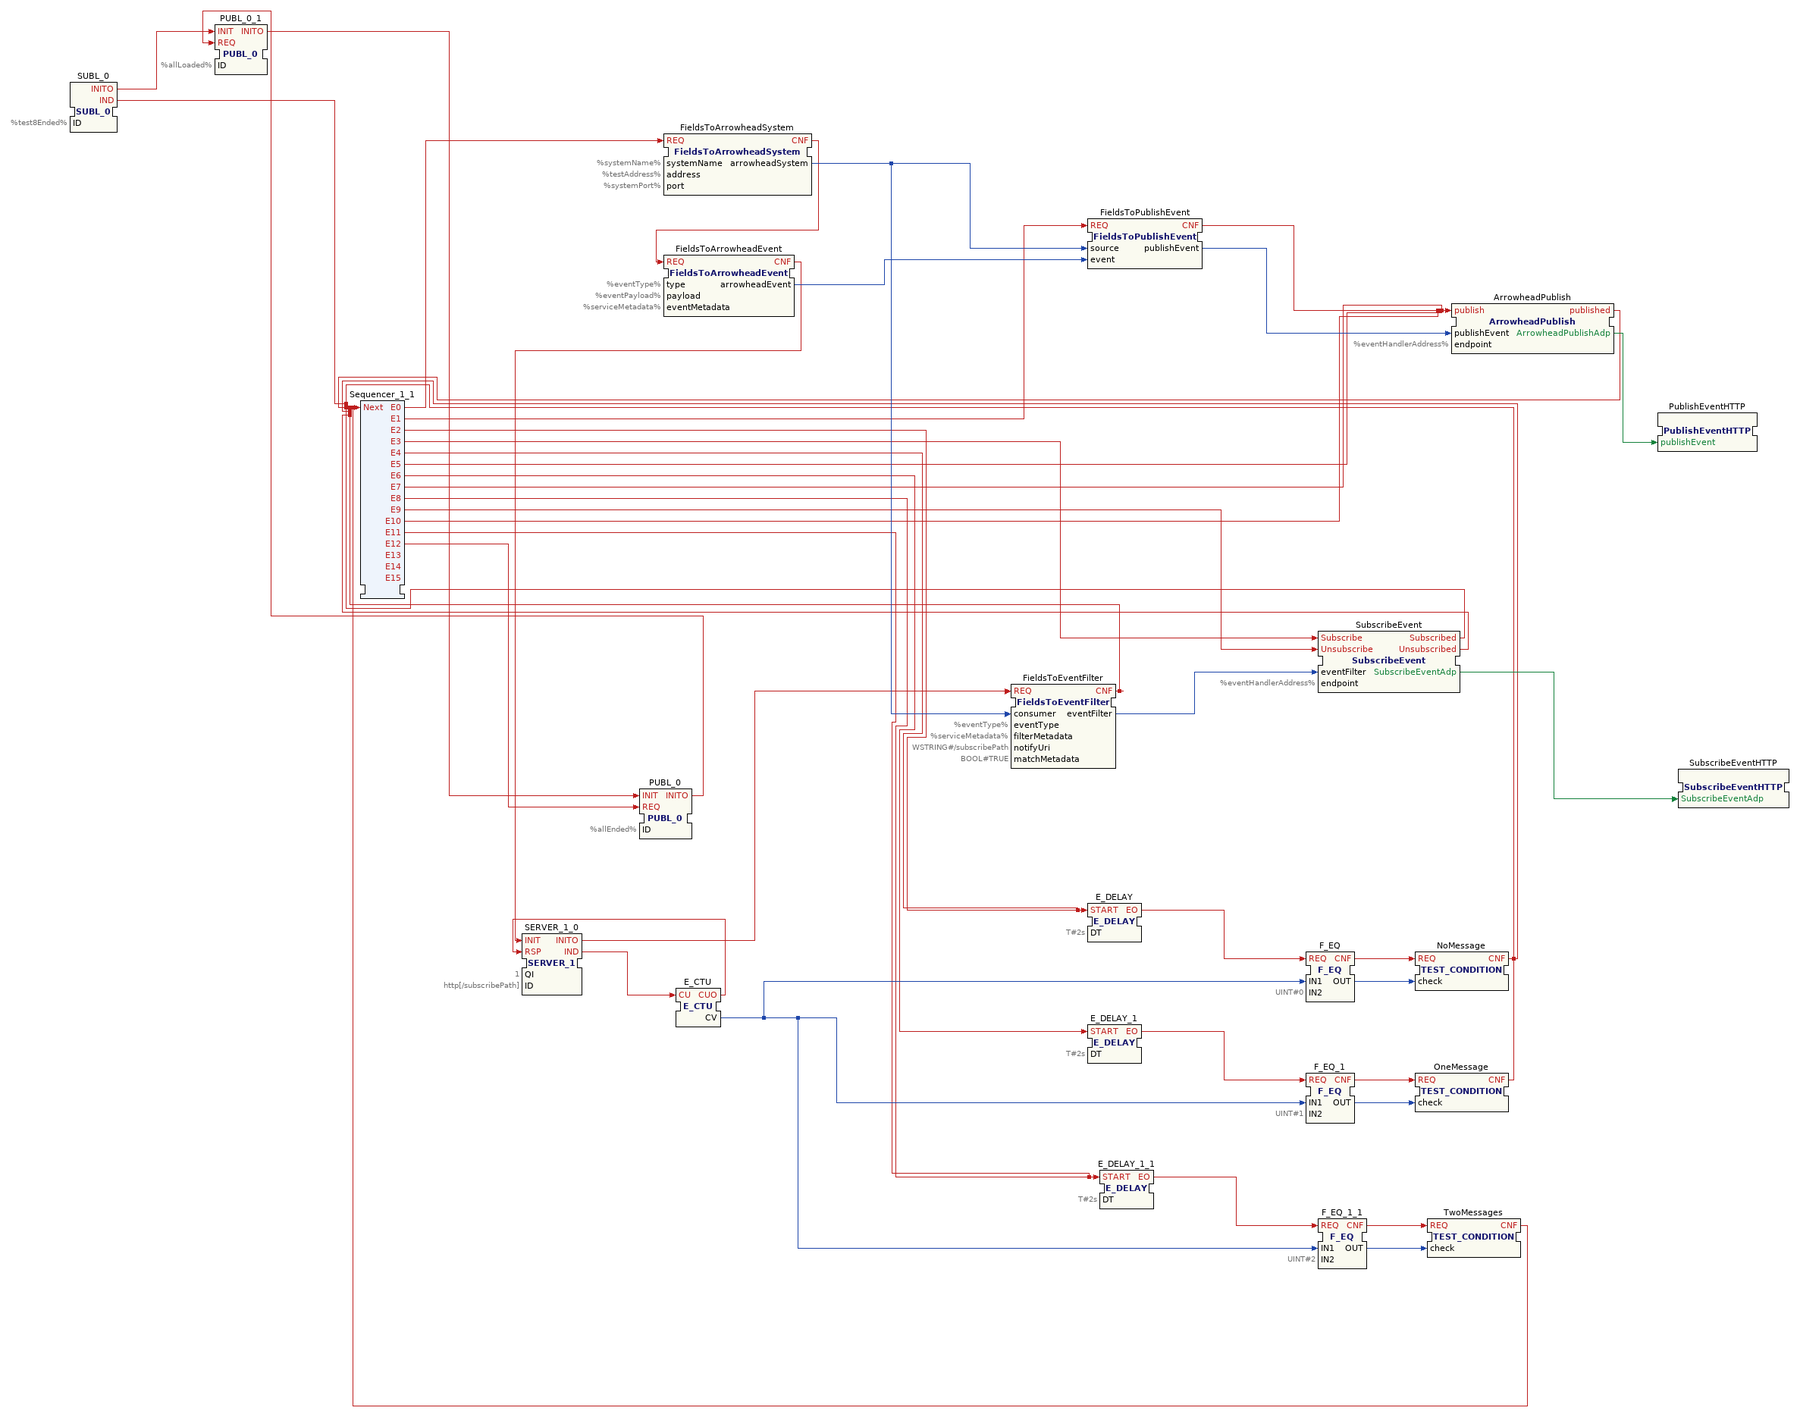
    FBS
      FieldsToPublishEvent : FieldsToPublishEvent;
      FieldsToArrowheadSystem : FieldsToArrowheadSystem(systemName := %systemName%, address := %testAddress%, port := %systemPort%);
      ArrowheadPublish : ArrowheadPublish(endpoint := %eventHandlerAddress%);
      FieldsToArrowheadEvent : FieldsToArrowheadEvent(type := %eventType%, payload := %eventPayload%, eventMetadata := %serviceMetadata%);
      FieldsToEventFilter : FieldsToEventFilter(eventType := %eventType%, filterMetadata := %serviceMetadata%, notifyUri := WSTRING#/subscribePath, matchMetadata := BOOL#TRUE);
      SubscribeEvent : SubscribeEvent(endpoint := %eventHandlerAddress%);
      E_CTU : E_CTU;
      F_EQ : F_EQ(IN2 := UINT#0);
      E_DELAY : E_DELAY(DT := T#2s);
      NoMessage : TEST_CONDITION;
      F_EQ_1 : F_EQ(IN2 := UINT#1);
      OneMessage : TEST_CONDITION;
      E_DELAY_1 : E_DELAY(DT := T#2s);
      E_DELAY_1_1 : E_DELAY(DT := T#2s);
      F_EQ_1_1 : F_EQ(IN2 := UINT#2);
      TwoMessages : TEST_CONDITION;
      SERVER_1_0 : SERVER_1(QI := 1, ID := http[/subscribePath]);
      SUBL_0 : SUBL_0(ID := %test8Ended%);
      PUBL_0_1 : PUBL_0(ID := %allLoaded%);
      PUBL_0 : PUBL_0(ID := %allEnded%);
      PublishEventHTTP : PublishEventHTTP;
      SubscribeEventHTTP : SubscribeEventHTTP;
    END_FBS
    SUBAPPLICATION Sequencer_1_1
      EVENT_INPUT
        Next;
      END_EVENT
      EVENT_OUTPUT
        E0;
        E1;
        E2;
        E3;
        E4;
        E5;
        E6;
        E7;
        E8;
        E9;
        E10;
        E11;
        E12;
        E13;
        E14;
        E15;
      END_EVENT
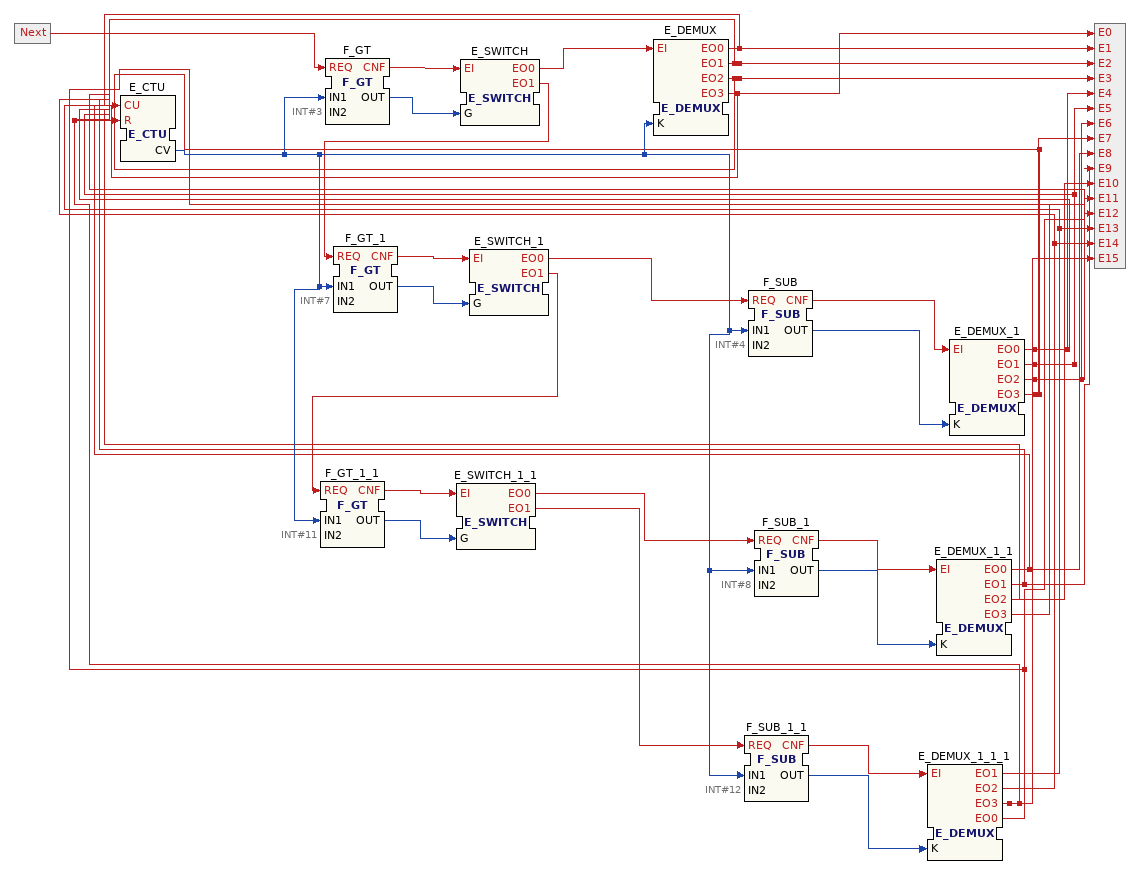
      FBS
        E_DEMUX : E_DEMUX;
        E_CTU : E_CTU;
        E_DEMUX_1 : E_DEMUX;
        E_SWITCH : E_SWITCH;
        F_GT : F_GT(IN2 := INT#3);
        F_SUB : F_SUB(IN2 := INT#4);
        E_DEMUX_1_1 : E_DEMUX;
        F_GT_1 : F_GT(IN2 := INT#7);
        F_SUB_1 : F_SUB(IN2 := INT#8);
        E_SWITCH_1 : E_SWITCH;
        F_GT_1_1 : F_GT(IN2 := INT#11);
        E_SWITCH_1_1 : E_SWITCH;
        E_DEMUX_1_1_1 : E_DEMUX;
        F_SUB_1_1 : F_SUB(IN2 := INT#12);
      END_FBS
      EVENT_CONNECTIONS
        E_DEMUX.EO0 TO E0;
        E_DEMUX.EO1 TO E1;
        E_DEMUX.EO2 TO E2;
        E_DEMUX.EO3 TO E3;
        E_DEMUX_1.EO0 TO E4;
        E_DEMUX_1.EO1 TO E5;
        E_DEMUX_1.EO2 TO E6;
        E_DEMUX_1.EO3 TO E7;
        F_GT.CNF TO E_SWITCH.EI;
        E_SWITCH.EO0 TO E_DEMUX.EI;
        F_SUB.CNF TO E_DEMUX_1.EI;
        E_SWITCH.EO1 TO F_GT_1.REQ;
        F_GT_1.CNF TO E_SWITCH_1.EI;
        E_SWITCH_1.EO0 TO F_SUB.REQ;
        F_SUB_1.CNF TO E_DEMUX_1_1.EI;
        E_DEMUX_1_1.EO0 TO E8;
        E_DEMUX_1_1.EO1 TO E9;
        E_DEMUX_1_1.EO2 TO E10;
        E_DEMUX.EO3 TO E_CTU.CU;
        E_DEMUX.EO2 TO E_CTU.CU;
        E_DEMUX.EO1 TO E_CTU.CU;
        E_DEMUX.EO0 TO E_CTU.CU;
        E_DEMUX_1_1.EO2 TO E_CTU.CU;
        E_DEMUX_1_1.EO1 TO E_CTU.CU;
        E_DEMUX_1_1.EO0 TO E_CTU.CU;
        E_DEMUX_1.EO3 TO E_CTU.CU;
        E_DEMUX_1.EO2 TO E_CTU.CU;
        E_DEMUX_1.EO1 TO E_CTU.CU;
        E_DEMUX_1.EO0 TO E_CTU.CU;
        F_GT_1_1.CNF TO E_SWITCH_1_1.EI;
        F_SUB_1_1.CNF TO E_DEMUX_1_1_1.EI;
        E_DEMUX_1_1_1.EO1 TO E13;
        E_DEMUX_1_1_1.EO2 TO E14;
        E_DEMUX_1_1_1.EO3 TO E15;
        E_SWITCH_1.EO1 TO F_GT_1_1.REQ;
        E_SWITCH_1_1.EO0 TO F_SUB_1.REQ;
        E_SWITCH_1_1.EO1 TO F_SUB_1_1.REQ;
        E_DEMUX_1_1_1.EO3 TO E_CTU.R;
        E_DEMUX_1_1_1.EO0 TO E_CTU.CU;
        E_DEMUX_1_1_1.EO1 TO E_CTU.CU;
        E_DEMUX_1_1_1.EO2 TO E_CTU.CU;
        E_DEMUX_1_1_1.EO3 TO E_CTU.CU;
        E_DEMUX_1_1.EO3 TO E11;
        E_DEMUX_1_1.EO3 TO E_CTU.CU;
        Next TO F_GT.REQ;
        E_DEMUX_1_1_1.EO0 TO E12;
      END_CONNECTIONS
      DATA_CONNECTIONS
        E_CTU.CV TO E_DEMUX.K;
        F_GT.OUT TO E_SWITCH.G;
        F_SUB.OUT TO E_DEMUX_1.K;
        E_CTU.CV TO F_GT.IN1;
        E_CTU.CV TO F_SUB.IN1;
        E_CTU.CV TO F_SUB_1.IN1;
        E_CTU.CV TO F_GT_1.IN1;
        F_GT_1.OUT TO E_SWITCH_1.G;
        F_SUB_1.OUT TO E_DEMUX_1_1.K;
        F_GT_1_1.OUT TO E_SWITCH_1_1.G;
        F_SUB_1_1.OUT TO E_DEMUX_1_1_1.K;
        E_CTU.CV TO F_SUB_1_1.IN1;
        E_CTU.CV TO F_GT_1_1.IN1;
      END_CONNECTIONS
    END_SUBAPPLICATION
    EVENT_CONNECTIONS
      FieldsToPublishEvent.CNF TO ArrowheadPublish.publish;
      FieldsToArrowheadSystem.CNF TO FieldsToArrowheadEvent.REQ;
      E_DELAY.EO TO F_EQ.REQ;
      F_EQ.CNF TO NoMessage.REQ;
      E_DELAY_1.EO TO F_EQ_1.REQ;
      F_EQ_1.CNF TO OneMessage.REQ;
      E_DELAY_1_1.EO TO F_EQ_1_1.REQ;
      F_EQ_1_1.CNF TO TwoMessages.REQ;
      Sequencer_1_1.E0 TO FieldsToArrowheadSystem.REQ;
      Sequencer_1_1.E1 TO FieldsToPublishEvent.REQ;
      Sequencer_1_1.E2 TO E_DELAY.START;
      Sequencer_1_1.E3 TO SubscribeEvent.Subscribe;
      Sequencer_1_1.E4 TO E_DELAY.START;
      Sequencer_1_1.E5 TO ArrowheadPublish.publish;
      Sequencer_1_1.E6 TO E_DELAY_1.START;
      Sequencer_1_1.E7 TO ArrowheadPublish.publish;
      Sequencer_1_1.E8 TO E_DELAY_1_1.START;
      Sequencer_1_1.E9 TO SubscribeEvent.Unsubscribe;
      Sequencer_1_1.E10 TO ArrowheadPublish.publish;
      TwoMessages.CNF TO Sequencer_1_1.Next;
      OneMessage.CNF TO Sequencer_1_1.Next;
      NoMessage.CNF TO Sequencer_1_1.Next;
      FieldsToEventFilter.CNF TO Sequencer_1_1.Next;
      Sequencer_1_1.E11 TO E_DELAY_1_1.START;
      ArrowheadPublish.published TO Sequencer_1_1.Next;
      SubscribeEvent.Subscribed TO Sequencer_1_1.Next;
      FieldsToArrowheadEvent.CNF TO SERVER_1_0.INIT;
      E_CTU.CUO TO SERVER_1_0.RSP;
      SERVER_1_0.INITO TO FieldsToEventFilter.REQ;
      SERVER_1_0.IND TO E_CTU.CU;
      SubscribeEvent.Unsubscribed TO Sequencer_1_1.Next;
      SUBL_0.INITO TO PUBL_0_1.INIT;
      SUBL_0.IND TO Sequencer_1_1.Next;
      PUBL_0_1.INITO TO PUBL_0.INIT;
      PUBL_0.INITO TO PUBL_0_1.REQ;
      Sequencer_1_1.E12 TO PUBL_0.REQ;
    END_CONNECTIONS
    DATA_CONNECTIONS
      FieldsToArrowheadSystem.arrowheadSystem TO FieldsToPublishEvent.source;
      FieldsToPublishEvent.publishEvent TO ArrowheadPublish.publishEvent;
      FieldsToArrowheadEvent.arrowheadEvent TO FieldsToPublishEvent.event;
      FieldsToEventFilter.eventFilter TO SubscribeEvent.eventFilter;
      FieldsToArrowheadSystem.arrowheadSystem TO FieldsToEventFilter.consumer;
      E_CTU.CV TO F_EQ.IN1;
      F_EQ.OUT TO NoMessage.check;
      E_CTU.CV TO F_EQ_1.IN1;
      F_EQ_1.OUT TO OneMessage.check;
      F_EQ_1_1.OUT TO TwoMessages.check;
      E_CTU.CV TO F_EQ_1_1.IN1;
    END_CONNECTIONS
    ADAPTER_CONNECTIONS
      ArrowheadPublish.ArrowheadPublishAdp TO PublishEventHTTP.publishEvent;
      SubscribeEvent.SubscribeEventAdp TO SubscribeEventHTTP.SubscribeEventAdp;
    END_CONNECTIONS
  END_APPLICATION
  DEVICE HTTPTest : FORTE_PC(MGR_ID := %httpTestAddress%)
    {SET_ATTRIBUTE(Profile, HOLOBLOC)} (* device profile *)
    RESOURCE cleanAll : EMB_RES
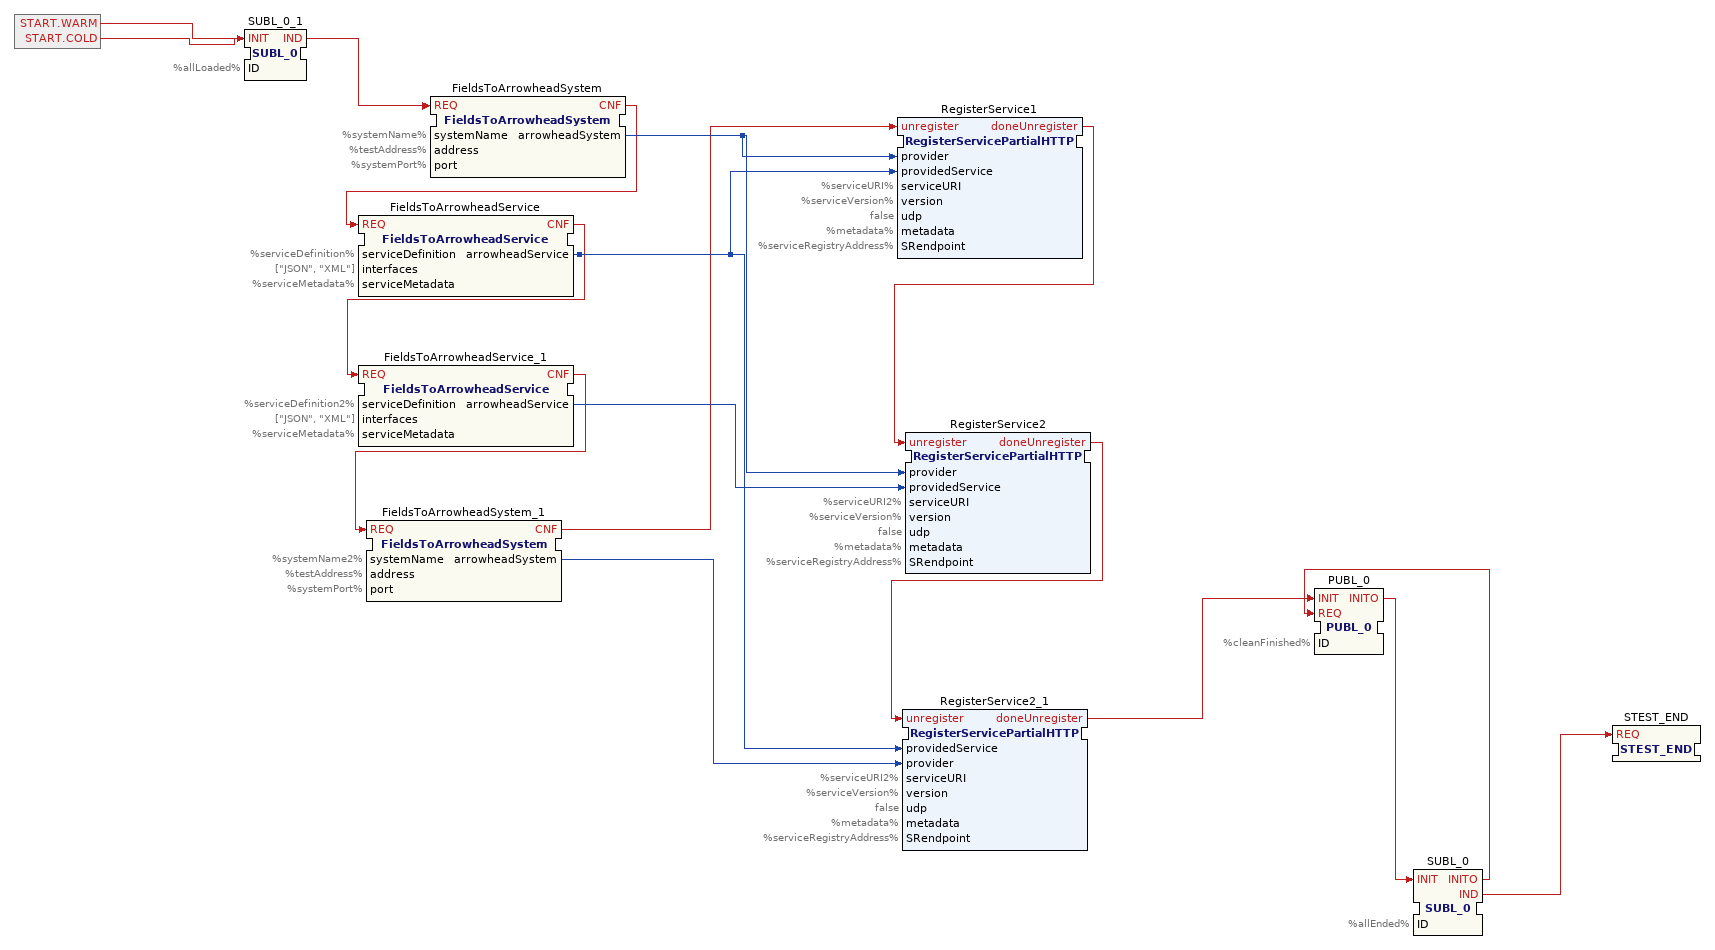
      FBS
        FieldsToArrowheadSystem : FieldsToArrowheadSystem(systemName := %systemName%, address := %testAddress%, port := %systemPort%);
        PUBL_0 : PUBL_0(ID := %cleanFinished%);
        FieldsToArrowheadService : FieldsToArrowheadService(serviceDefinition := %serviceDefinition%, interfaces := ["JSON", "XML"], serviceMetadata := %serviceMetadata%);
        FieldsToArrowheadService_1 : FieldsToArrowheadService(serviceDefinition := %serviceDefinition2%, interfaces := ["JSON", "XML"], serviceMetadata := %serviceMetadata%);
        FieldsToArrowheadSystem_1 : FieldsToArrowheadSystem(systemName := %systemName2%, address := %testAddress%, port := %systemPort%);
        SUBL_0 : SUBL_0(ID := %allEnded%);
        STEST_END : STEST_END;
        SUBL_0_1 : SUBL_0(ID := %allLoaded%);
      END_FBS
      SUBAPPS
        RegisterService1 : RegisterServicePartialHTTP(serviceURI := %serviceURI%, version := %serviceVersion%, udp := false, metadata := %metadata%, SRendpoint := %serviceRegistryAddress%);
        RegisterService2 : RegisterServicePartialHTTP(serviceURI := %serviceURI2%, version := %serviceVersion%, udp := false, metadata := %metadata%, SRendpoint := %serviceRegistryAddress%);
        RegisterService2_1 : RegisterServicePartialHTTP(serviceURI := %serviceURI2%, version := %serviceVersion%, udp := false, metadata := %metadata%, SRendpoint := %serviceRegistryAddress%);
      END_SUBAPPS
      EVENT_CONNECTIONS
        RegisterService1.doneUnregister TO RegisterService2.unregister;
        FieldsToArrowheadSystem.CNF TO FieldsToArrowheadService.REQ;
        FieldsToArrowheadService.CNF TO FieldsToArrowheadService_1.REQ;
        RegisterService2.doneUnregister TO RegisterService2_1.unregister;
        RegisterService2_1.doneUnregister TO PUBL_0.INIT;
        FieldsToArrowheadSystem_1.CNF TO RegisterService1.unregister;
        FieldsToArrowheadService_1.CNF TO FieldsToArrowheadSystem_1.REQ;
        SUBL_0.INITO TO PUBL_0.REQ;
        PUBL_0.INITO TO SUBL_0.INIT;
        SUBL_0.IND TO STEST_END.REQ;
        SUBL_0_1.IND TO FieldsToArrowheadSystem.REQ;
        START.WARM TO SUBL_0_1.INIT;
        START.COLD TO SUBL_0_1.INIT;
      END_CONNECTIONS
      DATA_CONNECTIONS
        FieldsToArrowheadSystem.arrowheadSystem TO RegisterService1.provider;
        FieldsToArrowheadSystem.arrowheadSystem TO RegisterService2.provider;
        FieldsToArrowheadService.arrowheadService TO RegisterService1.providedService;
        FieldsToArrowheadService_1.arrowheadService TO RegisterService2.providedService;
        FieldsToArrowheadService.arrowheadService TO RegisterService2_1.providedService;
        FieldsToArrowheadSystem_1.arrowheadSystem TO RegisterService2_1.provider;
      END_CONNECTIONS
    END_RESOURCE
    RESOURCE RegisterUnregister : EMB_RES
      FBS
        GET_AT_INDEX : GET_AT_INDEX(INDEX := 0);
        ServiceNotRegisteredPos1 : TEST_CONDITION;
        FieldsToServiceQueryForm : FieldsToServiceQueryForm(version := %serviceVersion%);
        QueryServiceHTTP : QueryServiceHTTP;
        FieldsToArrowheadService : FieldsToArrowheadService(serviceDefinition := %serviceDefinition%, interfaces := ["JSON", "XML"], serviceMetadata := %serviceMetadata%);
        F_EQ : F_EQ(IN1 := %emptyEndpoint%);
        QueryService : QueryService(address := %serviceRegistryAddress%);
        Registered : E_SR;
        E_SWITCH : E_SWITCH;
        F_EQ_1 : F_EQ(IN1 := %validEndpoint%);
        ServiceRegisteredPos0 : TEST_CONDITION;
        RegisterServiceHTTP : RegisterServiceHTTP;
        RegisterService : RegisterService(endpoint := %serviceRegistryAddress%);
        FieldsToServiceRegistryEntry : FieldsToServiceRegistryEntry(serviceURI := %serviceURI%, version := %serviceVersion%, udp := false, metadata := %metadata%);
        FieldsToArrowheadSystem : FieldsToArrowheadSystem(systemName := %systemName%, address := %testAddress%, port := %systemPort%);
        F_EQ_2 : F_EQ(IN1 := %emptyEndpoint%);
        ServiceNotRegisteredPos0 : TEST_CONDITION;
        GET_AT_INDEX_1 : GET_AT_INDEX(INDEX := 1);
        PUBLISH_0 : PUBL_0(ID := %firstResourceReady%);
        SUBL_0 : SUBL_0(ID := %cleanFinished%);
      END_FBS
      SUBAPPS
        GetEndpointFromServiceRegistryEntry : GetEndpointFromServiceRegistryEntry;
        GetEndpointFromServiceRegistryEntry_1 : GetEndpointFromServiceRegistryEntry;
      END_SUBAPPS
      SUBAPPLICATION Sequencer
        EVENT_INPUT
          Next;
        END_EVENT
        EVENT_OUTPUT
          E0;
          E1;
          E2;
          E3;
          E4;
          E5;
          E6;
          E7;
        END_EVENT
      END_SUBAPPLICATION
      EVENT_CONNECTIONS
        FieldsToArrowheadService.CNF TO FieldsToServiceQueryForm.REQ;
        F_EQ.CNF TO ServiceNotRegisteredPos1.REQ;
        GET_AT_INDEX.CNF TO GetEndpointFromServiceRegistryEntry.REQ;
        QueryService.queried TO GET_AT_INDEX.REQ;
        GetEndpointFromServiceRegistryEntry.CNF TO E_SWITCH.EI;
        E_SWITCH.EO1 TO F_EQ_1.REQ;
        F_EQ_1.CNF TO ServiceRegisteredPos0.REQ;
        ServiceRegisteredPos0.CNF TO Sequencer.Next;
        RegisterService.doneUnregister TO Sequencer.Next;
        RegisterService.doneUnregister TO Registered.R;
        RegisterService.doneRegister TO Sequencer.Next;
        RegisterService.doneRegister TO Registered.S;
        FieldsToArrowheadSystem.CNF TO FieldsToServiceRegistryEntry.REQ;
        F_EQ_2.CNF TO ServiceNotRegisteredPos0.REQ;
        GET_AT_INDEX_1.CNF TO GetEndpointFromServiceRegistryEntry_1.REQ;
        QueryService.queried TO GET_AT_INDEX_1.REQ;
        E_SWITCH.EO0 TO F_EQ_2.REQ;
        GetEndpointFromServiceRegistryEntry_1.CNF TO F_EQ.REQ;
        ServiceNotRegisteredPos0.CNF TO Sequencer.Next;
        FieldsToServiceQueryForm.CNF TO FieldsToArrowheadSystem.REQ;
        FieldsToServiceRegistryEntry.CNF TO Sequencer.Next;
        Sequencer.E4 TO QueryService.query;
        Sequencer.E3 TO RegisterService.unregister;
        Sequencer.E2 TO QueryService.query;
        Sequencer.E1 TO RegisterService.register;
        Sequencer.E0 TO QueryService.query;
        SUBL_0.IND TO FieldsToArrowheadService.REQ;
        START.WARM TO SUBL_0.INIT;
        START.COLD TO SUBL_0.INIT;
        Sequencer.E5 TO PUBLISH_0.REQ;
        SUBL_0.INITO TO PUBLISH_0.INIT;
      END_CONNECTIONS
      DATA_CONNECTIONS
        FieldsToArrowheadService.arrowheadService TO FieldsToServiceQueryForm.service;
        F_EQ.OUT TO ServiceNotRegisteredPos1.check;
        GET_AT_INDEX.OUT TO GetEndpointFromServiceRegistryEntry.serviceRegistryEntry;
        FieldsToServiceQueryForm.serviceQueryForm TO QueryService.serviceQueryForm;
        QueryService.serviceEntries TO GET_AT_INDEX.IN_ARRAY;
        Registered.Q TO E_SWITCH.G;
        F_EQ_1.OUT TO ServiceRegisteredPos0.check;
        GetEndpointFromServiceRegistryEntry.endpoint TO F_EQ_1.IN2;
        FieldsToServiceRegistryEntry.serviceRegistryEntry TO RegisterService.serviceRegistryEntry;
        FieldsToArrowheadService.arrowheadService TO FieldsToServiceRegistryEntry.providedService;
        FieldsToArrowheadSystem.arrowheadSystem TO FieldsToServiceRegistryEntry.provider;
        F_EQ_2.OUT TO ServiceNotRegisteredPos0.check;
        GET_AT_INDEX_1.OUT TO GetEndpointFromServiceRegistryEntry_1.serviceRegistryEntry;
        QueryService.serviceEntries TO GET_AT_INDEX_1.IN_ARRAY;
        GetEndpointFromServiceRegistryEntry.endpoint TO F_EQ_2.IN2;
        GetEndpointFromServiceRegistryEntry_1.endpoint TO F_EQ.IN2;
      END_CONNECTIONS
      ADAPTER_CONNECTIONS
        QueryService.queryServices TO QueryServiceHTTP.queryServices;
        RegisterService.registerService TO RegisterServiceHTTP.registerService;
      END_CONNECTIONS
    END_RESOURCE
    RESOURCE DoubleRegister : EMB_RES
      FBS
        QueryService : QueryService(address := %serviceRegistryAddress%);
        QueryServiceHTTP : QueryServiceHTTP;
        GET_AT_INDEX : GET_AT_INDEX(INDEX := 0);
        F_EQ : F_EQ(IN1 := %emptyEndpoint%);
        ServiceNotRegisteredPos1 : TEST_CONDITION;
        FieldsToArrowheadService : FieldsToArrowheadService(serviceDefinition := %serviceDefinition%, interfaces := ["JSON", "XML"], serviceMetadata := %serviceMetadata%);
        FieldsToServiceQueryForm : FieldsToServiceQueryForm(version := %serviceVersion%);
        Registered : E_SR;
        E_SWITCH : E_SWITCH;
        F_EQ_1 : F_EQ(IN1 := %validEndpoint%);
        ServiceRegisteredPos0 : TEST_CONDITION;
        FieldsToArrowheadSystem : FieldsToArrowheadSystem(systemName := %systemName%, address := %testAddress%, port := %systemPort%);
        FieldsToServiceRegistryEntry : FieldsToServiceRegistryEntry(serviceURI := %serviceURI%, version := %serviceVersion%, udp := false, metadata := %metadata%);
        RegisterService : RegisterService(endpoint := %serviceRegistryAddress%);
        RegisterServiceHTTP : RegisterServiceHTTP;
        GET_AT_INDEX_1 : GET_AT_INDEX(INDEX := 1);
        F_EQ_2 : F_EQ(IN1 := %emptyEndpoint%);
        ServiceNotRegisteredPos0 : TEST_CONDITION;
        SUBSCRIBE_0 : SUBL_0(ID := %firstResourceReady%);
        PUBL_0 : PUBL_0(ID := %secondResourceReady%);
      END_FBS
      SUBAPPS
        GetEndpointFromServiceRegistryEntry : GetEndpointFromServiceRegistryEntry;
        GetEndpointFromServiceRegistryEntry_1 : GetEndpointFromServiceRegistryEntry;
      END_SUBAPPS
      SUBAPPLICATION Sequencer
        EVENT_INPUT
          Next;
        END_EVENT
        EVENT_OUTPUT
          E0;
          E1;
          E2;
          E3;
          E4;
          E5;
          E6;
          E7;
        END_EVENT
      END_SUBAPPLICATION
      EVENT_CONNECTIONS
        QueryService.queried TO GET_AT_INDEX.REQ;
        F_EQ.CNF TO ServiceNotRegisteredPos1.REQ;
        GET_AT_INDEX.CNF TO GetEndpointFromServiceRegistryEntry.REQ;
        FieldsToArrowheadService.CNF TO FieldsToServiceQueryForm.REQ;
        GetEndpointFromServiceRegistryEntry.CNF TO E_SWITCH.EI;
        E_SWITCH.EO1 TO F_EQ_1.REQ;
        F_EQ_1.CNF TO ServiceRegisteredPos0.REQ;
        ServiceRegisteredPos0.CNF TO Sequencer.Next;
        FieldsToArrowheadSystem.CNF TO FieldsToServiceRegistryEntry.REQ;
        RegisterService.doneRegister TO Registered.S;
        RegisterService.doneUnregister TO Registered.R;
        QueryService.queried TO GET_AT_INDEX_1.REQ;
        E_SWITCH.EO0 TO F_EQ_2.REQ;
        F_EQ_2.CNF TO ServiceNotRegisteredPos0.REQ;
        ServiceNotRegisteredPos0.CNF TO Sequencer.Next;
        START.COLD TO SUBSCRIBE_0.INIT;
        START.WARM TO SUBSCRIBE_0.INIT;
        Sequencer.E0 TO RegisterService.register;
        Sequencer.E1 TO RegisterService.register;
        Sequencer.E2 TO QueryService.query;
        Sequencer.E4 TO QueryService.query;
        FieldsToServiceRegistryEntry.CNF TO Sequencer.Next;
        SUBSCRIBE_0.IND TO FieldsToArrowheadService.REQ;
        FieldsToServiceQueryForm.CNF TO FieldsToArrowheadSystem.REQ;
        Sequencer.E3 TO RegisterService.unregister;
        RegisterService.doneRegister TO Sequencer.Next;
        RegisterService.doneUnregister TO Sequencer.Next;
        Sequencer.E5 TO PUBL_0.REQ;
        SUBSCRIBE_0.INITO TO PUBL_0.INIT;
        GET_AT_INDEX_1.CNF TO GetEndpointFromServiceRegistryEntry_1.REQ;
        GetEndpointFromServiceRegistryEntry_1.CNF TO F_EQ.REQ;
      END_CONNECTIONS
      DATA_CONNECTIONS
        QueryService.serviceEntries TO GET_AT_INDEX.IN_ARRAY;
        F_EQ.OUT TO ServiceNotRegisteredPos1.check;
        GET_AT_INDEX.OUT TO GetEndpointFromServiceRegistryEntry.serviceRegistryEntry;
        FieldsToArrowheadService.arrowheadService TO FieldsToServiceQueryForm.service;
        FieldsToServiceQueryForm.serviceQueryForm TO QueryService.serviceQueryForm;
        Registered.Q TO E_SWITCH.G;
        GetEndpointFromServiceRegistryEntry.endpoint TO F_EQ_1.IN2;
        F_EQ_1.OUT TO ServiceRegisteredPos0.check;
        FieldsToArrowheadService.arrowheadService TO FieldsToServiceRegistryEntry.providedService;
        FieldsToArrowheadSystem.arrowheadSystem TO FieldsToServiceRegistryEntry.provider;
        FieldsToServiceRegistryEntry.serviceRegistryEntry TO RegisterService.serviceRegistryEntry;
        QueryService.serviceEntries TO GET_AT_INDEX_1.IN_ARRAY;
        GetEndpointFromServiceRegistryEntry.endpoint TO F_EQ_2.IN2;
        F_EQ_2.OUT TO ServiceNotRegisteredPos0.check;
        GET_AT_INDEX_1.OUT TO GetEndpointFromServiceRegistryEntry_1.serviceRegistryEntry;
        GetEndpointFromServiceRegistryEntry_1.endpoint TO F_EQ.IN2;
      END_CONNECTIONS
      ADAPTER_CONNECTIONS
        QueryService.queryServices TO QueryServiceHTTP.queryServices;
        RegisterService.registerService TO RegisterServiceHTTP.registerService;
      END_CONNECTIONS
    END_RESOURCE
    RESOURCE RegisterMoreServices : EMB_RES
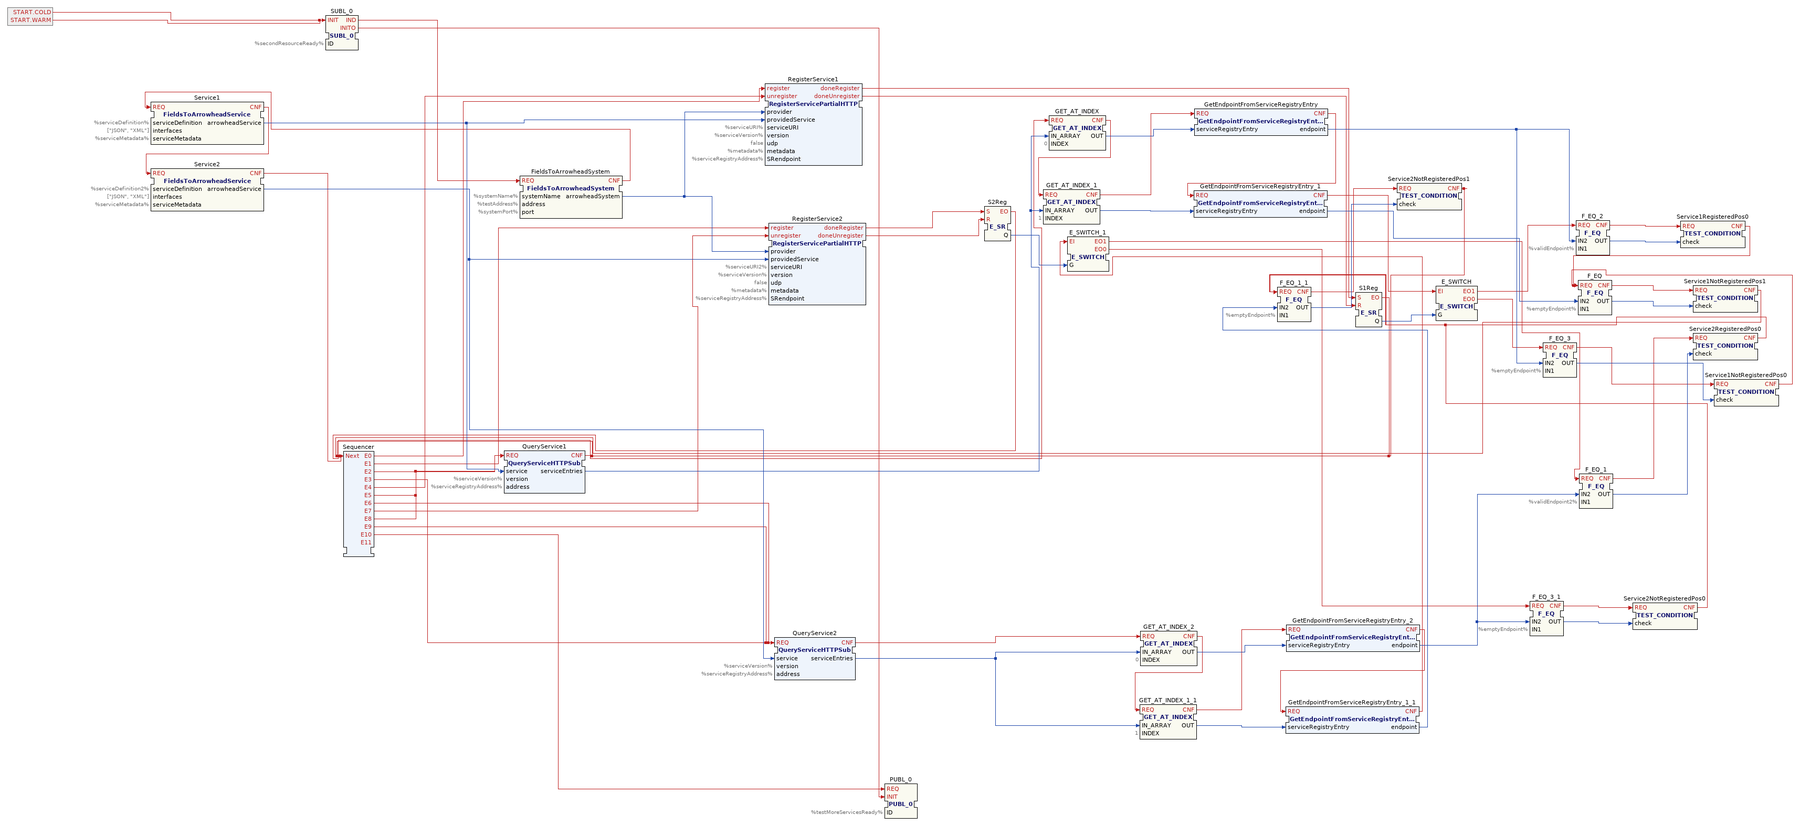
      FBS
        E_SWITCH : E_SWITCH;
        FieldsToArrowheadSystem : FieldsToArrowheadSystem(systemName := %systemName%, address := %testAddress%, port := %systemPort%);
        Service2RegisteredPos0 : TEST_CONDITION;
        Service1RegisteredPos0 : TEST_CONDITION;
        F_EQ : F_EQ(IN1 := %emptyEndpoint%);
        F_EQ_2 : F_EQ(IN1 := %validEndpoint%);
        Service1NotRegisteredPos1 : TEST_CONDITION;
        GET_AT_INDEX : GET_AT_INDEX(INDEX := 0);
        GET_AT_INDEX_1 : GET_AT_INDEX(INDEX := 1);
        F_EQ_1 : F_EQ(IN1 := %validEndpoint2%);
        S1Reg : E_SR;
        Service2NotRegisteredPos1 : TEST_CONDITION;
        F_EQ_1_1 : F_EQ(IN1 := %emptyEndpoint%);
        S2Reg : E_SR;
        E_SWITCH_1 : E_SWITCH;
        GET_AT_INDEX_1_1 : GET_AT_INDEX(INDEX := 1);
        GET_AT_INDEX_2 : GET_AT_INDEX(INDEX := 0);
        SUBL_0 : SUBL_0(ID := %secondResourceReady%);
        F_EQ_3 : F_EQ(IN1 := %emptyEndpoint%);
        Service1NotRegisteredPos0 : TEST_CONDITION;
        F_EQ_3_1 : F_EQ(IN1 := %emptyEndpoint%);
        Service2NotRegisteredPos0 : TEST_CONDITION;
        Service1 : FieldsToArrowheadService(serviceDefinition := %serviceDefinition%, interfaces := ["JSON", "XML"], serviceMetadata := %serviceMetadata%);
        Service2 : FieldsToArrowheadService(serviceDefinition := %serviceDefinition2%, interfaces := ["JSON", "XML"], serviceMetadata := %serviceMetadata%);
        PUBL_0 : PUBL_0(ID := %testMoreServicesReady%);
      END_FBS
      SUBAPPS
        GetEndpointFromServiceRegistryEntry_1 : GetEndpointFromServiceRegistryEntry;
        GetEndpointFromServiceRegistryEntry : GetEndpointFromServiceRegistryEntry;
        RegisterService2 : RegisterServicePartialHTTP(serviceURI := %serviceURI2%, version := %serviceVersion%, udp := false, metadata := %metadata%, SRendpoint := %serviceRegistryAddress%);
        RegisterService1 : RegisterServicePartialHTTP(serviceURI := %serviceURI%, version := %serviceVersion%, udp := false, metadata := %metadata%, SRendpoint := %serviceRegistryAddress%);
        GetEndpointFromServiceRegistryEntry_1_1 : GetEndpointFromServiceRegistryEntry;
        GetEndpointFromServiceRegistryEntry_2 : GetEndpointFromServiceRegistryEntry;
        QueryService2 : QueryServiceHTTPSub(version := %serviceVersion%, address := %serviceRegistryAddress%);
        QueryService1 : QueryServiceHTTPSub(version := %serviceVersion%, address := %serviceRegistryAddress%);
      END_SUBAPPS
      SUBAPPLICATION Sequencer
        EVENT_INPUT
          Next;
        END_EVENT
        EVENT_OUTPUT
          E0;
          E1;
          E2;
          E3;
          E4;
          E5;
          E6;
          E7;
          E8;
          E9;
          E10;
          E11;
        END_EVENT
      END_SUBAPPLICATION
      EVENT_CONNECTIONS
        F_EQ_2.CNF TO Service1RegisteredPos0.REQ;
        F_EQ.CNF TO Service1NotRegisteredPos1.REQ;
        F_EQ_1.CNF TO Service2RegisteredPos0.REQ;
        RegisterService1.doneRegister TO S1Reg.S;
        RegisterService1.doneUnregister TO S1Reg.R;
        F_EQ_1_1.CNF TO Service2NotRegisteredPos1.REQ;
        RegisterService2.doneRegister TO S2Reg.S;
        RegisterService2.doneUnregister TO S2Reg.R;
        SUBL_0.IND TO FieldsToArrowheadSystem.REQ;
        GET_AT_INDEX.CNF TO GET_AT_INDEX_1.REQ;
        GET_AT_INDEX_1.CNF TO GetEndpointFromServiceRegistryEntry.REQ;
        GetEndpointFromServiceRegistryEntry.CNF TO GetEndpointFromServiceRegistryEntry_1.REQ;
        Service1RegisteredPos0.CNF TO F_EQ.REQ;
        Service2RegisteredPos0.CNF TO F_EQ_1_1.REQ;
        QueryService2.CNF TO GET_AT_INDEX_2.REQ;
        GET_AT_INDEX_2.CNF TO GET_AT_INDEX_1_1.REQ;
        GET_AT_INDEX_1_1.CNF TO GetEndpointFromServiceRegistryEntry_2.REQ;
        GetEndpointFromServiceRegistryEntry_2.CNF TO GetEndpointFromServiceRegistryEntry_1_1.REQ;
        GetEndpointFromServiceRegistryEntry_1.CNF TO E_SWITCH.EI;
        E_SWITCH.EO1 TO F_EQ_2.REQ;
        E_SWITCH.EO0 TO F_EQ_3.REQ;
        F_EQ_3.CNF TO Service1NotRegisteredPos0.REQ;
        Service1NotRegisteredPos0.CNF TO F_EQ.REQ;
        F_EQ_3_1.CNF TO Service2NotRegisteredPos0.REQ;
        GetEndpointFromServiceRegistryEntry_1_1.CNF TO E_SWITCH_1.EI;
        E_SWITCH_1.EO1 TO F_EQ_1.REQ;
        E_SWITCH_1.EO0 TO F_EQ_3_1.REQ;
        Service2NotRegisteredPos0.CNF TO F_EQ_1_1.REQ;
        Service2NotRegisteredPos1.CNF TO Sequencer.Next;
        Service1NotRegisteredPos1.CNF TO Sequencer.Next;
        START.COLD TO SUBL_0.INIT;
        START.WARM TO SUBL_0.INIT;
        S2Reg.EO TO Sequencer.Next;
        S1Reg.EO TO Sequencer.Next;
        Sequencer.E0 TO RegisterService1.register;
        Sequencer.E1 TO RegisterService2.register;
        Sequencer.E3 TO QueryService2.REQ;
        Sequencer.E4 TO RegisterService1.unregister;
        Sequencer.E6 TO QueryService2.REQ;
        Sequencer.E7 TO RegisterService2.unregister;
        Sequencer.E9 TO QueryService2.REQ;
        Sequencer.E2 TO QueryService1.REQ;
        Sequencer.E5 TO QueryService1.REQ;
        Sequencer.E8 TO QueryService1.REQ;
        QueryService1.CNF TO GET_AT_INDEX.REQ;
        FieldsToArrowheadSystem.CNF TO Service1.REQ;
        Service1.CNF TO Service2.REQ;
        Service2.CNF TO Sequencer.Next;
        Sequencer.E10 TO PUBL_0.REQ;
        SUBL_0.INITO TO PUBL_0.INIT;
      END_CONNECTIONS
      DATA_CONNECTIONS
        F_EQ_2.OUT TO Service1RegisteredPos0.check;
        F_EQ.OUT TO Service1NotRegisteredPos1.check;
        GET_AT_INDEX.OUT TO GetEndpointFromServiceRegistryEntry.serviceRegistryEntry;
        GET_AT_INDEX_1.OUT TO GetEndpointFromServiceRegistryEntry_1.serviceRegistryEntry;
        F_EQ_1.OUT TO Service2RegisteredPos0.check;
        S1Reg.Q TO E_SWITCH.G;
        FieldsToArrowheadSystem.arrowheadSystem TO RegisterService2.provider;
        FieldsToArrowheadSystem.arrowheadSystem TO RegisterService1.provider;
        F_EQ_1_1.OUT TO Service2NotRegisteredPos1.check;
        S2Reg.Q TO E_SWITCH_1.G;
        GET_AT_INDEX_1_1.OUT TO GetEndpointFromServiceRegistryEntry_1_1.serviceRegistryEntry;
        QueryService2.serviceEntries TO GET_AT_INDEX_1_1.IN_ARRAY;
        QueryService2.serviceEntries TO GET_AT_INDEX_2.IN_ARRAY;
        GET_AT_INDEX_2.OUT TO GetEndpointFromServiceRegistryEntry_2.serviceRegistryEntry;
        GetEndpointFromServiceRegistryEntry_1.endpoint TO F_EQ.IN2;
        GetEndpointFromServiceRegistryEntry.endpoint TO F_EQ_2.IN2;
        GetEndpointFromServiceRegistryEntry_2.endpoint TO F_EQ_1.IN2;
        GetEndpointFromServiceRegistryEntry_1_1.endpoint TO F_EQ_1_1.IN2;
        GetEndpointFromServiceRegistryEntry.endpoint TO F_EQ_3.IN2;
        F_EQ_3.OUT TO Service1NotRegisteredPos0.check;
        F_EQ_3_1.OUT TO Service2NotRegisteredPos0.check;
        GetEndpointFromServiceRegistryEntry_2.endpoint TO F_EQ_3_1.IN2;
        QueryService1.serviceEntries TO GET_AT_INDEX.IN_ARRAY;
        QueryService1.serviceEntries TO GET_AT_INDEX_1.IN_ARRAY;
        Service1.arrowheadService TO RegisterService1.providedService;
        Service2.arrowheadService TO RegisterService2.providedService;
        Service1.arrowheadService TO QueryService1.service;
        Service2.arrowheadService TO QueryService2.service;
      END_CONNECTIONS
    END_RESOURCE
    RESOURCE SameServiceTwice : EMB_RES
      FBS
        SUBL_0 : SUBL_0(ID := %testMoreServicesReady%);
        Service1 : FieldsToArrowheadService(serviceDefinition := %serviceDefinition%, interfaces := ["JSON", "XML"], serviceMetadata := %serviceMetadata%);
        FieldsToArrowheadSystem : FieldsToArrowheadSystem(systemName := %systemName%, address := %testAddress%, port := %systemPort%);
        GET_AT_INDEX_1 : GET_AT_INDEX(INDEX := 1);
        GET_AT_INDEX : GET_AT_INDEX(INDEX := 0);
        Service1RegisteredPos0 : TEST_CONDITION;
        F_EQ_2 : F_EQ(IN1 := %validEndpoint%);
        BothServicesRegistered : TEST_CONDITION;
        F_EQ_3 : F_EQ(IN1 := %validEndpoint2%);
        F_EQ : F_EQ(IN1 := %validEndpoint%);
        F_EQ_2_1 : F_EQ(IN1 := %validEndpoint2%);
        F_EQ_3_1 : F_EQ(IN1 := %validEndpoint%);
        Service2RegisteredPos0 : TEST_CONDITION;
        F_EQ_1 : F_EQ(IN1 := %validEndpoint2%);
        BothServicesNotRegistered : TEST_CONDITION;
        F_EQ_1_1 : F_EQ(IN1 := %emptyEndpoint%);
        F_EQ_1_1_1 : F_EQ(IN1 := %emptyEndpoint%);
        Service2NotRegisteredPos1 : TEST_CONDITION;
        F_EQ_4 : F_EQ(IN1 := %emptyEndpoint%);
        F_EQ_4_1 : F_EQ(IN1 := %emptyEndpoint%);
        Service1NotRegisteredPos1 : TEST_CONDITION;
        F_AND : F_AND;
        E_MERGE : E_MERGE;
        E_MERGE_1 : E_MERGE;
        F_AND_1 : F_AND;
        F_OR : F_OR;
        F_AND_1_1 : F_AND;
        BOOL2BOOL : BOOL2BOOL;
        BOOL2BOOL_1 : BOOL2BOOL;
        FieldsToArrowheadSystem_1 : FieldsToArrowheadSystem(systemName := %systemName2%, address := %testAddress%, port := %systemPort%);
        PUBL_0 : PUBL_0(ID := %sameServiceTwiceReady%);
      END_FBS
      SUBAPPS
        RegisterService2 : RegisterServicePartialHTTP(serviceURI := %serviceURI2%, version := %serviceVersion%, udp := false, metadata := %metadata%, SRendpoint := %serviceRegistryAddress%);
        RegisterService1 : RegisterServicePartialHTTP(serviceURI := %serviceURI%, version := %serviceVersion%, udp := false, metadata := %metadata%, SRendpoint := %serviceRegistryAddress%);
        QueryServiceHTTPSub : QueryServiceHTTPSub(version := %serviceVersion%, address := %serviceRegistryAddress%);
        GetEndpointFromServiceRegistryEntry : GetEndpointFromServiceRegistryEntry;
        GetEndpointFromServiceRegistryEntry_1 : GetEndpointFromServiceRegistryEntry;
      END_SUBAPPS
      SUBAPPLICATION Sequencer
        EVENT_INPUT
          Next;
        END_EVENT
        EVENT_OUTPUT
          E0;
          E1;
          E2;
          E3;
          E4;
          E5;
          E6;
          E7;
          E8;
          E9;
          E10;
          E11;
        END_EVENT
      END_SUBAPPLICATION
      EVENT_CONNECTIONS
        Sequencer.E1 TO RegisterService2.register;
        Sequencer.E7 TO RegisterService2.unregister;
        Sequencer.E0 TO RegisterService1.register;
        Sequencer.E4 TO RegisterService1.unregister;
        FieldsToArrowheadSystem.CNF TO Service1.REQ;
        Sequencer.E2 TO QueryServiceHTTPSub.REQ;
        Sequencer.E5 TO QueryServiceHTTPSub.REQ;
        Sequencer.E8 TO QueryServiceHTTPSub.REQ;
        GET_AT_INDEX_1.CNF TO GetEndpointFromServiceRegistryEntry.REQ;
        QueryServiceHTTPSub.CNF TO GET_AT_INDEX.REQ;
        GET_AT_INDEX.CNF TO GET_AT_INDEX_1.REQ;
        GetEndpointFromServiceRegistryEntry.CNF TO GetEndpointFromServiceRegistryEntry_1.REQ;
        GetEndpointFromServiceRegistryEntry_1.CNF TO Sequencer.Next;
        F_EQ_3.CNF TO F_EQ_2.REQ;
        F_EQ.CNF TO Service1RegisteredPos0.REQ;
        Sequencer.E3 TO F_EQ_3_1.REQ;
        F_EQ_3_1.CNF TO F_EQ_2_1.REQ;
        Sequencer.E6 TO F_EQ_1.REQ;
        F_EQ_1.CNF TO Service2RegisteredPos0.REQ;
        Sequencer.E9 TO F_EQ_1_1.REQ;
        F_EQ_1_1.CNF TO F_EQ_1_1_1.REQ;
        Service1RegisteredPos0.CNF TO F_EQ_4.REQ;
        F_EQ_4.CNF TO Service2NotRegisteredPos1.REQ;
        Service2RegisteredPos0.CNF TO F_EQ_4_1.REQ;
        F_EQ_4_1.CNF TO Service1NotRegisteredPos1.REQ;
        F_EQ_1_1_1.CNF TO F_AND.REQ;
        F_AND.CNF TO BothServicesNotRegistered.REQ;
        BothServicesRegistered.CNF TO E_MERGE.EI1;
        BothServicesNotRegistered.CNF TO E_MERGE.EI2;
        Service1NotRegisteredPos1.CNF TO E_MERGE.EI2;
        Service2NotRegisteredPos1.CNF TO E_MERGE.EI2;
        E_MERGE.EO TO Sequencer.Next;
        RegisterService1.doneRegister TO E_MERGE_1.EI1;
        RegisterService2.doneRegister TO E_MERGE_1.EI1;
        RegisterService1.doneUnregister TO E_MERGE_1.EI2;
        RegisterService2.doneUnregister TO E_MERGE_1.EI2;
        E_MERGE_1.EO TO Sequencer.Next;
        F_EQ_2_1.CNF TO F_AND_1.REQ;
        F_OR.CNF TO BothServicesRegistered.REQ;
        F_EQ_2.CNF TO F_AND_1_1.REQ;
        F_AND_1.CNF TO BOOL2BOOL.REQ;
        BOOL2BOOL.CNF TO F_EQ_3.REQ;
        F_AND_1_1.CNF TO BOOL2BOOL_1.REQ;
        BOOL2BOOL_1.CNF TO F_OR.REQ;
        START.COLD TO SUBL_0.INIT;
        START.WARM TO SUBL_0.INIT;
        Service1.CNF TO Sequencer.Next;
        FieldsToArrowheadSystem_1.CNF TO FieldsToArrowheadSystem.REQ;
        SUBL_0.IND TO FieldsToArrowheadSystem_1.REQ;
        SUBL_0.INITO TO PUBL_0.INIT;
        Sequencer.E10 TO PUBL_0.REQ;
      END_CONNECTIONS
      DATA_CONNECTIONS
        Service1.arrowheadService TO RegisterService2.providedService;
        Service1.arrowheadService TO RegisterService1.providedService;
        FieldsToArrowheadSystem.arrowheadSystem TO RegisterService1.provider;
        Service1.arrowheadService TO QueryServiceHTTPSub.service;
        QueryServiceHTTPSub.serviceEntries TO GET_AT_INDEX_1.IN_ARRAY;
        QueryServiceHTTPSub.serviceEntries TO GET_AT_INDEX.IN_ARRAY;
        GET_AT_INDEX.OUT TO GetEndpointFromServiceRegistryEntry.serviceRegistryEntry;
        GET_AT_INDEX_1.OUT TO GetEndpointFromServiceRegistryEntry_1.serviceRegistryEntry;
        GetEndpointFromServiceRegistryEntry_1.endpoint TO F_EQ_2.IN2;
        GetEndpointFromServiceRegistryEntry.endpoint TO F_EQ_3.IN2;
        GetEndpointFromServiceRegistryEntry.endpoint TO F_EQ.IN2;
        F_EQ.OUT TO Service1RegisteredPos0.check;
        GetEndpointFromServiceRegistryEntry_1.endpoint TO F_EQ_2_1.IN2;
        GetEndpointFromServiceRegistryEntry.endpoint TO F_EQ_3_1.IN2;
        GetEndpointFromServiceRegistryEntry.endpoint TO F_EQ_1.IN2;
        F_EQ_1.OUT TO Service2RegisteredPos0.check;
        GetEndpointFromServiceRegistryEntry.endpoint TO F_EQ_1_1.IN2;
        GetEndpointFromServiceRegistryEntry_1.endpoint TO F_EQ_1_1_1.IN2;
        GetEndpointFromServiceRegistryEntry_1.endpoint TO F_EQ_4.IN2;
        F_EQ_4.OUT TO Service2NotRegisteredPos1.check;
        GetEndpointFromServiceRegistryEntry_1.endpoint TO F_EQ_4_1.IN2;
        F_EQ_4_1.OUT TO Service1NotRegisteredPos1.check;
        F_EQ_1_1.OUT TO F_AND.IN1;
        F_EQ_1_1_1.OUT TO F_AND.IN2;
        F_AND.OUT TO BothServicesNotRegistered.check;
        F_EQ_3_1.OUT TO F_AND_1.IN1;
        F_EQ_2_1.OUT TO F_AND_1.IN2;
        F_OR.OUT TO BothServicesRegistered.check;
        F_EQ_3.OUT TO F_AND_1_1.IN1;
        F_EQ_2.OUT TO F_AND_1_1.IN2;
        F_AND_1.OUT TO BOOL2BOOL.IN;
        BOOL2BOOL.OUT TO F_OR.IN1;
        F_AND_1_1.OUT TO BOOL2BOOL_1.IN;
        BOOL2BOOL_1.OUT TO F_OR.IN2;
        FieldsToArrowheadSystem_1.arrowheadSystem TO RegisterService2.provider;
      END_CONNECTIONS
    END_RESOURCE
    RESOURCE VersionInterfaceAndMetadata : EMB_RES
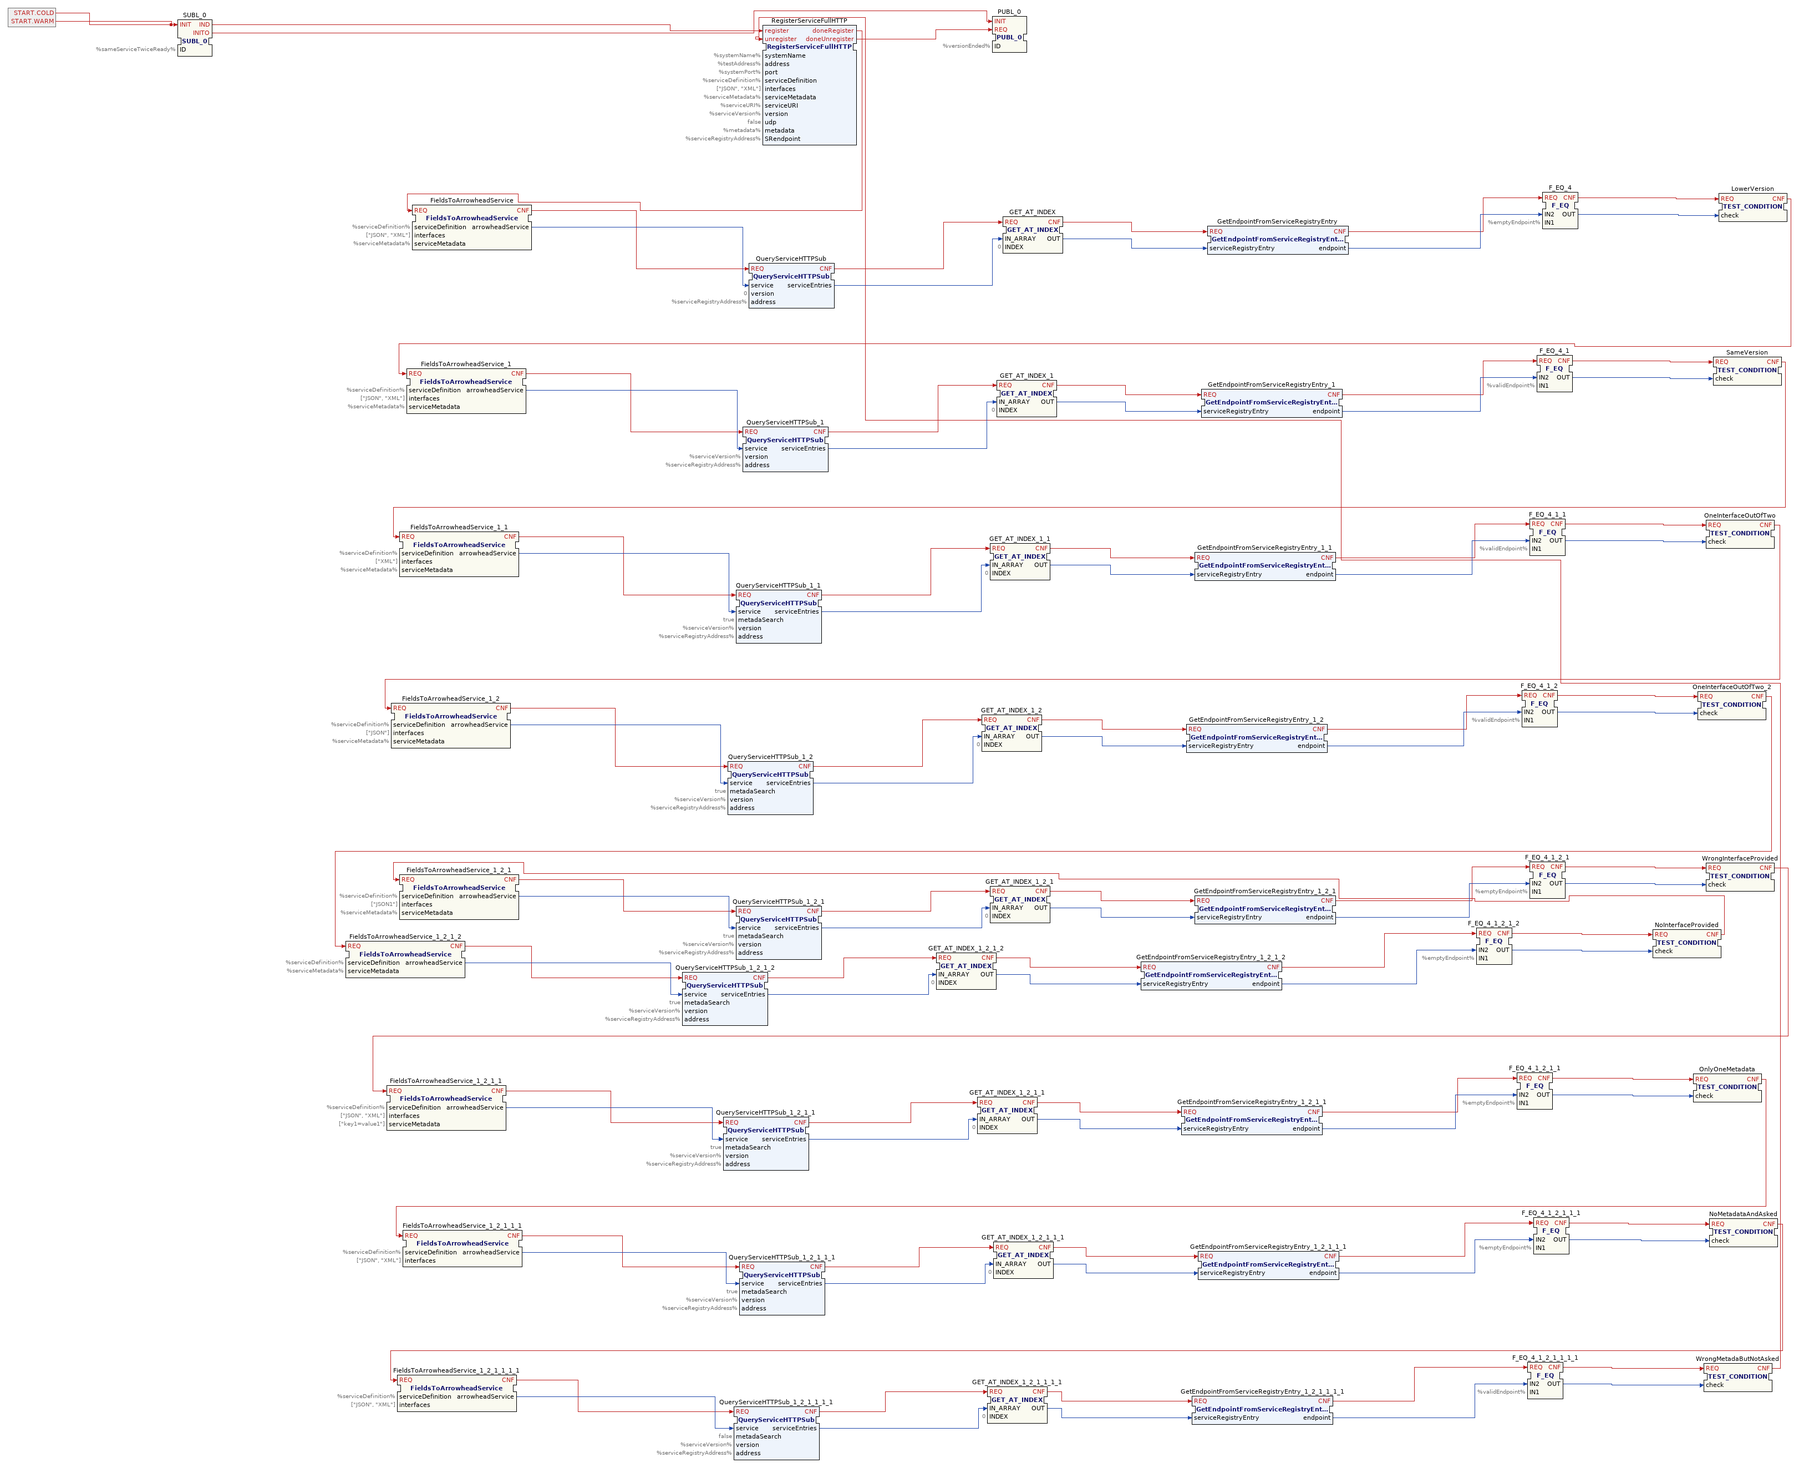
      FBS
        FieldsToArrowheadService : FieldsToArrowheadService(serviceDefinition := %serviceDefinition%, interfaces := ["JSON", "XML"], serviceMetadata := %serviceMetadata%);
        GET_AT_INDEX : GET_AT_INDEX(INDEX := 0);
        F_EQ_4 : F_EQ(IN1 := %emptyEndpoint%);
        LowerVersion : TEST_CONDITION;
        FieldsToArrowheadService_1 : FieldsToArrowheadService(serviceDefinition := %serviceDefinition%, interfaces := ["JSON", "XML"], serviceMetadata := %serviceMetadata%);
        SameVersion : TEST_CONDITION;
        GET_AT_INDEX_1 : GET_AT_INDEX(INDEX := 0);
        F_EQ_4_1 : F_EQ(IN1 := %validEndpoint%);
        OneInterfaceOutOfTwo : TEST_CONDITION;
        F_EQ_4_1_1 : F_EQ(IN1 := %validEndpoint%);
        FieldsToArrowheadService_1_1 : FieldsToArrowheadService(serviceDefinition := %serviceDefinition%, interfaces := ["XML"], serviceMetadata := %serviceMetadata%);
        GET_AT_INDEX_1_1 : GET_AT_INDEX(INDEX := 0);
        OneInterfaceOutOfTwo_2 : TEST_CONDITION;
        F_EQ_4_1_2 : F_EQ(IN1 := %validEndpoint%);
        FieldsToArrowheadService_1_2 : FieldsToArrowheadService(serviceDefinition := %serviceDefinition%, interfaces := ["JSON"], serviceMetadata := %serviceMetadata%);
        GET_AT_INDEX_1_2 : GET_AT_INDEX(INDEX := 0);
        WrongInterfaceProvided : TEST_CONDITION;
        GET_AT_INDEX_1_2_1 : GET_AT_INDEX(INDEX := 0);
        FieldsToArrowheadService_1_2_1 : FieldsToArrowheadService(serviceDefinition := %serviceDefinition%, interfaces := ["JSON1"], serviceMetadata := %serviceMetadata%);
        F_EQ_4_1_2_1 : F_EQ(IN1 := %emptyEndpoint%);
        SUBL_0 : SUBL_0(ID := %sameServiceTwiceReady%);
        OnlyOneMetadata : TEST_CONDITION;
        F_EQ_4_1_2_1_1 : F_EQ(IN1 := %emptyEndpoint%);
        FieldsToArrowheadService_1_2_1_1 : FieldsToArrowheadService(serviceDefinition := %serviceDefinition%, interfaces := ["JSON", "XML"], serviceMetadata := ["key1=value1"]);
        GET_AT_INDEX_1_2_1_1 : GET_AT_INDEX(INDEX := 0);
        FieldsToArrowheadService_1_2_1_1_1 : FieldsToArrowheadService(serviceDefinition := %serviceDefinition%, interfaces := ["JSON", "XML"]);
        F_EQ_4_1_2_1_1_1 : F_EQ(IN1 := %emptyEndpoint%);
        GET_AT_INDEX_1_2_1_1_1 : GET_AT_INDEX(INDEX := 0);
        NoMetadataAndAsked : TEST_CONDITION;
        FieldsToArrowheadService_1_2_1_2 : FieldsToArrowheadService(serviceDefinition := %serviceDefinition%, serviceMetadata := %serviceMetadata%);
        F_EQ_4_1_2_1_2 : F_EQ(IN1 := %emptyEndpoint%);
        GET_AT_INDEX_1_2_1_2 : GET_AT_INDEX(INDEX := 0);
        NoInterfaceProvided : TEST_CONDITION;
        GET_AT_INDEX_1_2_1_1_1_1 : GET_AT_INDEX(INDEX := 0);
        FieldsToArrowheadService_1_2_1_1_1_1 : FieldsToArrowheadService(serviceDefinition := %serviceDefinition%, interfaces := ["JSON", "XML"]);
        WrongMetadaButNotAsked : TEST_CONDITION;
        F_EQ_4_1_2_1_1_1_1 : F_EQ(IN1 := %validEndpoint%);
        PUBL_0 : PUBL_0(ID := %versionEnded%);
      END_FBS
      SUBAPPS
        RegisterServiceFullHTTP : RegisterServiceFullHTTP(systemName := %systemName%, address := %testAddress%, port := %systemPort%, serviceDefinition := %serviceDefinition%, interfaces := ["JSON", "XML"], serviceMetadata := %serviceMetadata%, serviceURI := %serviceURI%, version := %serviceVersion%, udp := false, metadata := %metadata%, SRendpoint := %serviceRegistryAddress%);
        QueryServiceHTTPSub : QueryServiceHTTPSub(version := 0, address := %serviceRegistryAddress%);
        GetEndpointFromServiceRegistryEntry : GetEndpointFromServiceRegistryEntry;
        QueryServiceHTTPSub_1 : QueryServiceHTTPSub(version := %serviceVersion%, address := %serviceRegistryAddress%);
        GetEndpointFromServiceRegistryEntry_1 : GetEndpointFromServiceRegistryEntry;
        QueryServiceHTTPSub_1_1 : QueryServiceHTTPSub(metadaSearch := true, version := %serviceVersion%, address := %serviceRegistryAddress%);
        GetEndpointFromServiceRegistryEntry_1_1 : GetEndpointFromServiceRegistryEntry;
        QueryServiceHTTPSub_1_2 : QueryServiceHTTPSub(metadaSearch := true, version := %serviceVersion%, address := %serviceRegistryAddress%);
        GetEndpointFromServiceRegistryEntry_1_2 : GetEndpointFromServiceRegistryEntry;
        QueryServiceHTTPSub_1_2_1 : QueryServiceHTTPSub(metadaSearch := true, version := %serviceVersion%, address := %serviceRegistryAddress%);
        GetEndpointFromServiceRegistryEntry_1_2_1 : GetEndpointFromServiceRegistryEntry;
        GetEndpointFromServiceRegistryEntry_1_2_1_1 : GetEndpointFromServiceRegistryEntry;
        QueryServiceHTTPSub_1_2_1_1 : QueryServiceHTTPSub(metadaSearch := true, version := %serviceVersion%, address := %serviceRegistryAddress%);
        QueryServiceHTTPSub_1_2_1_1_1 : QueryServiceHTTPSub(metadaSearch := true, version := %serviceVersion%, address := %serviceRegistryAddress%);
        GetEndpointFromServiceRegistryEntry_1_2_1_1_1 : GetEndpointFromServiceRegistryEntry;
        GetEndpointFromServiceRegistryEntry_1_2_1_2 : GetEndpointFromServiceRegistryEntry;
        QueryServiceHTTPSub_1_2_1_2 : QueryServiceHTTPSub(metadaSearch := true, version := %serviceVersion%, address := %serviceRegistryAddress%);
        QueryServiceHTTPSub_1_2_1_1_1_1 : QueryServiceHTTPSub(metadaSearch := false, version := %serviceVersion%, address := %serviceRegistryAddress%);
        GetEndpointFromServiceRegistryEntry_1_2_1_1_1_1 : GetEndpointFromServiceRegistryEntry;
      END_SUBAPPS
      EVENT_CONNECTIONS
        FieldsToArrowheadService.CNF TO QueryServiceHTTPSub.REQ;
        QueryServiceHTTPSub.CNF TO GET_AT_INDEX.REQ;
        GET_AT_INDEX.CNF TO GetEndpointFromServiceRegistryEntry.REQ;
        GetEndpointFromServiceRegistryEntry.CNF TO F_EQ_4.REQ;
        F_EQ_4.CNF TO LowerVersion.REQ;
        FieldsToArrowheadService_1.CNF TO QueryServiceHTTPSub_1.REQ;
        QueryServiceHTTPSub_1.CNF TO GET_AT_INDEX_1.REQ;
        GET_AT_INDEX_1.CNF TO GetEndpointFromServiceRegistryEntry_1.REQ;
        GetEndpointFromServiceRegistryEntry_1.CNF TO F_EQ_4_1.REQ;
        F_EQ_4_1.CNF TO SameVersion.REQ;
        GetEndpointFromServiceRegistryEntry_1_1.CNF TO F_EQ_4_1_1.REQ;
        F_EQ_4_1_1.CNF TO OneInterfaceOutOfTwo.REQ;
        FieldsToArrowheadService_1_1.CNF TO QueryServiceHTTPSub_1_1.REQ;
        QueryServiceHTTPSub_1_1.CNF TO GET_AT_INDEX_1_1.REQ;
        GET_AT_INDEX_1_1.CNF TO GetEndpointFromServiceRegistryEntry_1_1.REQ;
        GetEndpointFromServiceRegistryEntry_1_2.CNF TO F_EQ_4_1_2.REQ;
        F_EQ_4_1_2.CNF TO OneInterfaceOutOfTwo_2.REQ;
        FieldsToArrowheadService_1_2.CNF TO QueryServiceHTTPSub_1_2.REQ;
        QueryServiceHTTPSub_1_2.CNF TO GET_AT_INDEX_1_2.REQ;
        GET_AT_INDEX_1_2.CNF TO GetEndpointFromServiceRegistryEntry_1_2.REQ;
        QueryServiceHTTPSub_1_2_1.CNF TO GET_AT_INDEX_1_2_1.REQ;
        GET_AT_INDEX_1_2_1.CNF TO GetEndpointFromServiceRegistryEntry_1_2_1.REQ;
        FieldsToArrowheadService_1_2_1.CNF TO QueryServiceHTTPSub_1_2_1.REQ;
        GetEndpointFromServiceRegistryEntry_1_2_1.CNF TO F_EQ_4_1_2_1.REQ;
        F_EQ_4_1_2_1.CNF TO WrongInterfaceProvided.REQ;
        GetEndpointFromServiceRegistryEntry_1_2_1_1.CNF TO F_EQ_4_1_2_1_1.REQ;
        F_EQ_4_1_2_1_1.CNF TO OnlyOneMetadata.REQ;
        GET_AT_INDEX_1_2_1_1.CNF TO GetEndpointFromServiceRegistryEntry_1_2_1_1.REQ;
        FieldsToArrowheadService_1_2_1_1.CNF TO QueryServiceHTTPSub_1_2_1_1.REQ;
        QueryServiceHTTPSub_1_2_1_1.CNF TO GET_AT_INDEX_1_2_1_1.REQ;
        FieldsToArrowheadService_1_2_1_1_1.CNF TO QueryServiceHTTPSub_1_2_1_1_1.REQ;
        GetEndpointFromServiceRegistryEntry_1_2_1_1_1.CNF TO F_EQ_4_1_2_1_1_1.REQ;
        QueryServiceHTTPSub_1_2_1_1_1.CNF TO GET_AT_INDEX_1_2_1_1_1.REQ;
        GET_AT_INDEX_1_2_1_1_1.CNF TO GetEndpointFromServiceRegistryEntry_1_2_1_1_1.REQ;
        F_EQ_4_1_2_1_1_1.CNF TO NoMetadataAndAsked.REQ;
        START.COLD TO SUBL_0.INIT;
        START.WARM TO SUBL_0.INIT;
        GetEndpointFromServiceRegistryEntry_1_2_1_2.CNF TO F_EQ_4_1_2_1_2.REQ;
        GET_AT_INDEX_1_2_1_2.CNF TO GetEndpointFromServiceRegistryEntry_1_2_1_2.REQ;
        F_EQ_4_1_2_1_2.CNF TO NoInterfaceProvided.REQ;
        FieldsToArrowheadService_1_2_1_2.CNF TO QueryServiceHTTPSub_1_2_1_2.REQ;
        QueryServiceHTTPSub_1_2_1_2.CNF TO GET_AT_INDEX_1_2_1_2.REQ;
        FieldsToArrowheadService_1_2_1_1_1_1.CNF TO QueryServiceHTTPSub_1_2_1_1_1_1.REQ;
        QueryServiceHTTPSub_1_2_1_1_1_1.CNF TO GET_AT_INDEX_1_2_1_1_1_1.REQ;
        GET_AT_INDEX_1_2_1_1_1_1.CNF TO GetEndpointFromServiceRegistryEntry_1_2_1_1_1_1.REQ;
        GetEndpointFromServiceRegistryEntry_1_2_1_1_1_1.CNF TO F_EQ_4_1_2_1_1_1_1.REQ;
        F_EQ_4_1_2_1_1_1_1.CNF TO WrongMetadaButNotAsked.REQ;
        SUBL_0.IND TO RegisterServiceFullHTTP.register;
        RegisterServiceFullHTTP.doneRegister TO FieldsToArrowheadService.REQ;
        LowerVersion.CNF TO FieldsToArrowheadService_1.REQ;
        SameVersion.CNF TO FieldsToArrowheadService_1_1.REQ;
        OneInterfaceOutOfTwo.CNF TO FieldsToArrowheadService_1_2.REQ;
        OneInterfaceOutOfTwo_2.CNF TO FieldsToArrowheadService_1_2_1_2.REQ;
        NoInterfaceProvided.CNF TO FieldsToArrowheadService_1_2_1.REQ;
        WrongInterfaceProvided.CNF TO FieldsToArrowheadService_1_2_1_1.REQ;
        OnlyOneMetadata.CNF TO FieldsToArrowheadService_1_2_1_1_1.REQ;
        NoMetadataAndAsked.CNF TO FieldsToArrowheadService_1_2_1_1_1_1.REQ;
        WrongMetadaButNotAsked.CNF TO RegisterServiceFullHTTP.unregister;
        SUBL_0.INITO TO PUBL_0.INIT;
        RegisterServiceFullHTTP.doneUnregister TO PUBL_0.REQ;
      END_CONNECTIONS
      DATA_CONNECTIONS
        FieldsToArrowheadService.arrowheadService TO QueryServiceHTTPSub.service;
        QueryServiceHTTPSub.serviceEntries TO GET_AT_INDEX.IN_ARRAY;
        GET_AT_INDEX.OUT TO GetEndpointFromServiceRegistryEntry.serviceRegistryEntry;
        GetEndpointFromServiceRegistryEntry.endpoint TO F_EQ_4.IN2;
        F_EQ_4.OUT TO LowerVersion.check;
        FieldsToArrowheadService_1.arrowheadService TO QueryServiceHTTPSub_1.service;
        QueryServiceHTTPSub_1.serviceEntries TO GET_AT_INDEX_1.IN_ARRAY;
        GET_AT_INDEX_1.OUT TO GetEndpointFromServiceRegistryEntry_1.serviceRegistryEntry;
        GetEndpointFromServiceRegistryEntry_1.endpoint TO F_EQ_4_1.IN2;
        F_EQ_4_1.OUT TO SameVersion.check;
        GetEndpointFromServiceRegistryEntry_1_1.endpoint TO F_EQ_4_1_1.IN2;
        F_EQ_4_1_1.OUT TO OneInterfaceOutOfTwo.check;
        FieldsToArrowheadService_1_1.arrowheadService TO QueryServiceHTTPSub_1_1.service;
        QueryServiceHTTPSub_1_1.serviceEntries TO GET_AT_INDEX_1_1.IN_ARRAY;
        GET_AT_INDEX_1_1.OUT TO GetEndpointFromServiceRegistryEntry_1_1.serviceRegistryEntry;
        GetEndpointFromServiceRegistryEntry_1_2.endpoint TO F_EQ_4_1_2.IN2;
        F_EQ_4_1_2.OUT TO OneInterfaceOutOfTwo_2.check;
        FieldsToArrowheadService_1_2.arrowheadService TO QueryServiceHTTPSub_1_2.service;
        QueryServiceHTTPSub_1_2.serviceEntries TO GET_AT_INDEX_1_2.IN_ARRAY;
        GET_AT_INDEX_1_2.OUT TO GetEndpointFromServiceRegistryEntry_1_2.serviceRegistryEntry;
        QueryServiceHTTPSub_1_2_1.serviceEntries TO GET_AT_INDEX_1_2_1.IN_ARRAY;
        GET_AT_INDEX_1_2_1.OUT TO GetEndpointFromServiceRegistryEntry_1_2_1.serviceRegistryEntry;
        FieldsToArrowheadService_1_2_1.arrowheadService TO QueryServiceHTTPSub_1_2_1.service;
        GetEndpointFromServiceRegistryEntry_1_2_1.endpoint TO F_EQ_4_1_2_1.IN2;
        F_EQ_4_1_2_1.OUT TO WrongInterfaceProvided.check;
        GetEndpointFromServiceRegistryEntry_1_2_1_1.endpoint TO F_EQ_4_1_2_1_1.IN2;
        F_EQ_4_1_2_1_1.OUT TO OnlyOneMetadata.check;
        GET_AT_INDEX_1_2_1_1.OUT TO GetEndpointFromServiceRegistryEntry_1_2_1_1.serviceRegistryEntry;
        FieldsToArrowheadService_1_2_1_1.arrowheadService TO QueryServiceHTTPSub_1_2_1_1.service;
        QueryServiceHTTPSub_1_2_1_1.serviceEntries TO GET_AT_INDEX_1_2_1_1.IN_ARRAY;
        FieldsToArrowheadService_1_2_1_1_1.arrowheadService TO QueryServiceHTTPSub_1_2_1_1_1.service;
        GetEndpointFromServiceRegistryEntry_1_2_1_1_1.endpoint TO F_EQ_4_1_2_1_1_1.IN2;
        QueryServiceHTTPSub_1_2_1_1_1.serviceEntries TO GET_AT_INDEX_1_2_1_1_1.IN_ARRAY;
        GET_AT_INDEX_1_2_1_1_1.OUT TO GetEndpointFromServiceRegistryEntry_1_2_1_1_1.serviceRegistryEntry;
        F_EQ_4_1_2_1_1_1.OUT TO NoMetadataAndAsked.check;
        GetEndpointFromServiceRegistryEntry_1_2_1_2.endpoint TO F_EQ_4_1_2_1_2.IN2;
        GET_AT_INDEX_1_2_1_2.OUT TO GetEndpointFromServiceRegistryEntry_1_2_1_2.serviceRegistryEntry;
        F_EQ_4_1_2_1_2.OUT TO NoInterfaceProvided.check;
        FieldsToArrowheadService_1_2_1_2.arrowheadService TO QueryServiceHTTPSub_1_2_1_2.service;
        QueryServiceHTTPSub_1_2_1_2.serviceEntries TO GET_AT_INDEX_1_2_1_2.IN_ARRAY;
        FieldsToArrowheadService_1_2_1_1_1_1.arrowheadService TO QueryServiceHTTPSub_1_2_1_1_1_1.service;
        QueryServiceHTTPSub_1_2_1_1_1_1.serviceEntries TO GET_AT_INDEX_1_2_1_1_1_1.IN_ARRAY;
        GET_AT_INDEX_1_2_1_1_1_1.OUT TO GetEndpointFromServiceRegistryEntry_1_2_1_1_1_1.serviceRegistryEntry;
        GetEndpointFromServiceRegistryEntry_1_2_1_1_1_1.endpoint TO F_EQ_4_1_2_1_1_1_1.IN2;
        F_EQ_4_1_2_1_1_1_1.OUT TO WrongMetadaButNotAsked.check;
      END_CONNECTIONS
    END_RESOURCE
    RESOURCE RegisterMoreServicesSubApp : EMB_RES
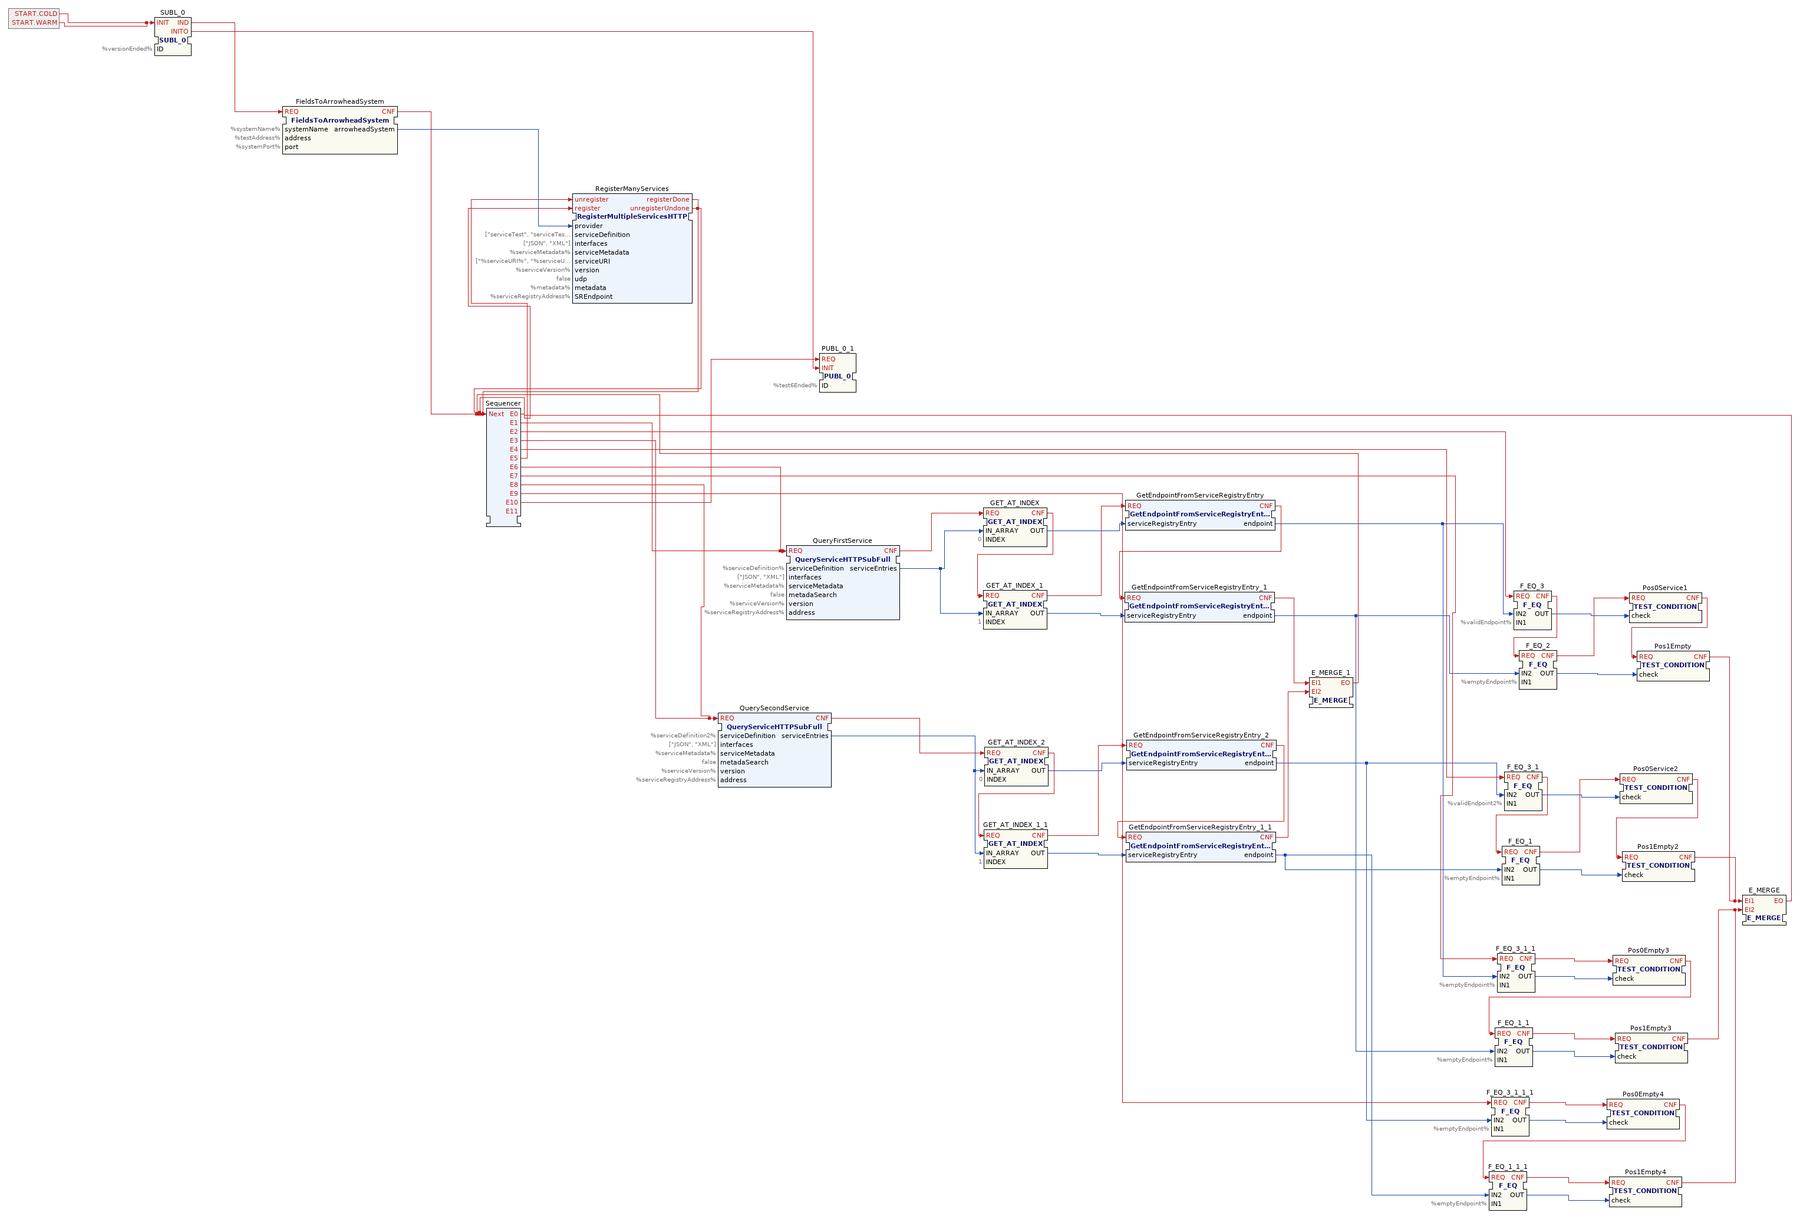
      FBS
        SUBL_0 : SUBL_0(ID := %versionEnded%);
        GET_AT_INDEX_1 : GET_AT_INDEX(INDEX := 1);
        FieldsToArrowheadSystem : FieldsToArrowheadSystem(systemName := %systemName%, address := %testAddress%, port := %systemPort%);
        F_EQ_2 : F_EQ(IN1 := %emptyEndpoint%);
        GET_AT_INDEX : GET_AT_INDEX(INDEX := 0);
        Pos1Empty2 : TEST_CONDITION;
        F_EQ_1 : F_EQ(IN1 := %emptyEndpoint%);
        Pos1Empty : TEST_CONDITION;
        GET_AT_INDEX_1_1 : GET_AT_INDEX(INDEX := 1);
        GET_AT_INDEX_2 : GET_AT_INDEX(INDEX := 0);
        Pos0Service1 : TEST_CONDITION;
        F_EQ_3 : F_EQ(IN1 := %validEndpoint%);
        F_EQ_3_1 : F_EQ(IN1 := %validEndpoint2%);
        Pos0Service2 : TEST_CONDITION;
        PUBL_0_1 : PUBL_0(ID := %test6Ended%);
        F_EQ_1_1 : F_EQ(IN1 := %emptyEndpoint%);
        F_EQ_3_1_1 : F_EQ(IN1 := %emptyEndpoint%);
        Pos1Empty3 : TEST_CONDITION;
        Pos0Empty3 : TEST_CONDITION;
        F_EQ_1_1_1 : F_EQ(IN1 := %emptyEndpoint%);
        Pos0Empty4 : TEST_CONDITION;
        Pos1Empty4 : TEST_CONDITION;
        F_EQ_3_1_1_1 : F_EQ(IN1 := %emptyEndpoint%);
        E_MERGE : E_MERGE;
        E_MERGE_1 : E_MERGE;
      END_FBS
      SUBAPPS
        GetEndpointFromServiceRegistryEntry_1 : GetEndpointFromServiceRegistryEntry;
        GetEndpointFromServiceRegistryEntry : GetEndpointFromServiceRegistryEntry;
        GetEndpointFromServiceRegistryEntry_1_1 : GetEndpointFromServiceRegistryEntry;
        GetEndpointFromServiceRegistryEntry_2 : GetEndpointFromServiceRegistryEntry;
        QuerySecondService : QueryServiceHTTPSubFull(serviceDefinition := %serviceDefinition2%, interfaces := ["JSON", "XML"], serviceMetadata := %serviceMetadata%, metadaSearch := false, version := %serviceVersion%, address := %serviceRegistryAddress%);
        QueryFirstService : QueryServiceHTTPSubFull(serviceDefinition := %serviceDefinition%, interfaces := ["JSON", "XML"], serviceMetadata := %serviceMetadata%, metadaSearch := false, version := %serviceVersion%, address := %serviceRegistryAddress%);
        RegisterManyServices : RegisterMultipleServicesHTTP(serviceDefinition := ["serviceTest", "serviceTest2"], interfaces := ["JSON", "XML"], serviceMetadata := %serviceMetadata%, serviceURI := ["%serviceURI%", "%serviceURI2%"], version := %serviceVersion%, udp := false, metadata := %metadata%, SREndpoint := %serviceRegistryAddress%);
      END_SUBAPPS
      SUBAPPLICATION Sequencer
        EVENT_INPUT
          Next;
        END_EVENT
        EVENT_OUTPUT
          E0;
          E1;
          E2;
          E3;
          E4;
          E5;
          E6;
          E7;
          E8;
          E9;
          E10;
          E11;
        END_EVENT
      END_SUBAPPLICATION
      EVENT_CONNECTIONS
        START.COLD TO SUBL_0.INIT;
        START.WARM TO SUBL_0.INIT;
        GET_AT_INDEX_1.CNF TO GetEndpointFromServiceRegistryEntry.REQ;
        GetEndpointFromServiceRegistryEntry.CNF TO GetEndpointFromServiceRegistryEntry_1.REQ;
        SUBL_0.IND TO FieldsToArrowheadSystem.REQ;
        GET_AT_INDEX.CNF TO GET_AT_INDEX_1.REQ;
        FieldsToArrowheadSystem.CNF TO Sequencer.Next;
        GET_AT_INDEX_1_1.CNF TO GetEndpointFromServiceRegistryEntry_2.REQ;
        GetEndpointFromServiceRegistryEntry_2.CNF TO GetEndpointFromServiceRegistryEntry_1_1.REQ;
        GET_AT_INDEX_2.CNF TO GET_AT_INDEX_1_1.REQ;
        F_EQ_2.CNF TO Pos0Service1.REQ;
        Pos0Service1.CNF TO Pos1Empty.REQ;
        Sequencer.E2 TO F_EQ_3.REQ;
        F_EQ_3.CNF TO F_EQ_2.REQ;
        Sequencer.E4 TO F_EQ_3_1.REQ;
        F_EQ_3_1.CNF TO F_EQ_1.REQ;
        F_EQ_1.CNF TO Pos0Service2.REQ;
        Pos0Service2.CNF TO Pos1Empty2.REQ;
        Sequencer.E3 TO QuerySecondService.REQ;
        Sequencer.E8 TO QuerySecondService.REQ;
        QuerySecondService.CNF TO GET_AT_INDEX_2.REQ;
        Sequencer.E1 TO QueryFirstService.REQ;
        Sequencer.E6 TO QueryFirstService.REQ;
        QueryFirstService.CNF TO GET_AT_INDEX.REQ;
        F_EQ_1_1.CNF TO Pos1Empty3.REQ;
        F_EQ_3_1_1.CNF TO Pos0Empty3.REQ;
        Pos0Empty3.CNF TO F_EQ_1_1.REQ;
        Pos0Empty4.CNF TO F_EQ_1_1_1.REQ;
        F_EQ_1_1_1.CNF TO Pos1Empty4.REQ;
        F_EQ_3_1_1_1.CNF TO Pos0Empty4.REQ;
        Pos1Empty.CNF TO E_MERGE.EI1;
        Pos1Empty2.CNF TO E_MERGE.EI1;
        Pos1Empty3.CNF TO E_MERGE.EI2;
        Pos1Empty4.CNF TO E_MERGE.EI2;
        E_MERGE.EO TO Sequencer.Next;
        GetEndpointFromServiceRegistryEntry_1.CNF TO E_MERGE_1.EI1;
        GetEndpointFromServiceRegistryEntry_1_1.CNF TO E_MERGE_1.EI2;
        E_MERGE_1.EO TO Sequencer.Next;
        Sequencer.E7 TO F_EQ_3_1_1.REQ;
        Sequencer.E9 TO F_EQ_3_1_1_1.REQ;
        RegisterManyServices.registerDone TO Sequencer.Next;
        RegisterManyServices.unregisterUndone TO Sequencer.Next;
        Sequencer.E5 TO RegisterManyServices.unregister;
        Sequencer.E0 TO RegisterManyServices.register;
        Sequencer.E10 TO PUBL_0_1.REQ;
        SUBL_0.INITO TO PUBL_0_1.INIT;
      END_CONNECTIONS
      DATA_CONNECTIONS
        GET_AT_INDEX_1.OUT TO GetEndpointFromServiceRegistryEntry_1.serviceRegistryEntry;
        GetEndpointFromServiceRegistryEntry_1.endpoint TO F_EQ_2.IN2;
        GET_AT_INDEX.OUT TO GetEndpointFromServiceRegistryEntry.serviceRegistryEntry;
        F_EQ_1.OUT TO Pos1Empty2.check;
        F_EQ_2.OUT TO Pos1Empty.check;
        GET_AT_INDEX_1_1.OUT TO GetEndpointFromServiceRegistryEntry_1_1.serviceRegistryEntry;
        GetEndpointFromServiceRegistryEntry_1_1.endpoint TO F_EQ_1.IN2;
        GET_AT_INDEX_2.OUT TO GetEndpointFromServiceRegistryEntry_2.serviceRegistryEntry;
        GetEndpointFromServiceRegistryEntry.endpoint TO F_EQ_3.IN2;
        F_EQ_3.OUT TO Pos0Service1.check;
        GetEndpointFromServiceRegistryEntry_2.endpoint TO F_EQ_3_1.IN2;
        F_EQ_3_1.OUT TO Pos0Service2.check;
        QuerySecondService.serviceEntries TO GET_AT_INDEX_1_1.IN_ARRAY;
        QuerySecondService.serviceEntries TO GET_AT_INDEX_2.IN_ARRAY;
        QueryFirstService.serviceEntries TO GET_AT_INDEX_1.IN_ARRAY;
        QueryFirstService.serviceEntries TO GET_AT_INDEX.IN_ARRAY;
        F_EQ_1_1.OUT TO Pos1Empty3.check;
        F_EQ_3_1_1.OUT TO Pos0Empty3.check;
        F_EQ_1_1_1.OUT TO Pos1Empty4.check;
        F_EQ_3_1_1_1.OUT TO Pos0Empty4.check;
        FieldsToArrowheadSystem.arrowheadSystem TO RegisterManyServices.provider;
        GetEndpointFromServiceRegistryEntry.endpoint TO F_EQ_3_1_1.IN2;
        GetEndpointFromServiceRegistryEntry_1.endpoint TO F_EQ_1_1.IN2;
        GetEndpointFromServiceRegistryEntry_2.endpoint TO F_EQ_3_1_1_1.IN2;
        GetEndpointFromServiceRegistryEntry_1_1.endpoint TO F_EQ_1_1_1.IN2;
      END_CONNECTIONS
    END_RESOURCE
    RESOURCE OrchestratorNoRule : EMB_RES
      FBS
        RequestOrchestrationHTTP : RequestOrchestrationHTTP;
        FieldsToServiceRequestForm : FieldsToServiceRequestForm;
        FieldsToArrowheadSystem : FieldsToArrowheadSystem(systemName := %systemName%, address := %testAddress%, port := %systemPort%);
        Service1 : FieldsToArrowheadService(serviceDefinition := %serviceDefinition2%, interfaces := ["JSON", "XML"], serviceMetadata := %serviceMetadata%);
        F_EQ : F_EQ(IN1 := %emptyEndpoint%);
        NoServiceAvailable : TEST_CONDITION;
        SERVER_1 : SERVER_1(ID := http[/serviceTest/start2]);
        E_SR : E_SR;
        SUBL_0 : SUBL_0(ID := %test6Ended%);
        PUBL_0 : PUBL_0(ID := %test7Ended%);
        GET_STRUCT_VALUE1 : GET_AT_INDEX(INDEX := 0);
        RequestOrchestrationForm : RequestOrchestrationForm(endpoint := %orchestratorAddress%);
      END_FBS
      SUBAPPS
        GetEndpointFromOrchestrationForm : GetEndpointFromOrchestrationForm;
        RegisterService2 : RegisterServicePartialHTTP(serviceURI := %serviceURI2%, version := %serviceVersion%, udp := false, metadata := %metadata%, SRendpoint := %serviceRegistryAddress%);
      END_SUBAPPS
      SUBAPPLICATION Sequencer_1
        EVENT_INPUT
          Next;
        END_EVENT
        EVENT_OUTPUT
          E0;
          E1;
          E2;
          E3;
          E4;
          E5;
          E6;
          E7;
          E8;
          E9;
          E10;
          E11;
        END_EVENT
      END_SUBAPPLICATION
      EVENT_CONNECTIONS
        FieldsToArrowheadSystem.CNF TO Service1.REQ;
        Service1.CNF TO FieldsToServiceRequestForm.REQ;
        GetEndpointFromOrchestrationForm.CNF TO F_EQ.REQ;
        F_EQ.CNF TO NoServiceAvailable.REQ;
        E_SR.EO TO SERVER_1.INIT;
        SUBL_0.IND TO FieldsToArrowheadSystem.REQ;
        START.WARM TO SUBL_0.INIT;
        GET_STRUCT_VALUE1.CNF TO GetEndpointFromOrchestrationForm.REQ;
        Sequencer_1.E1 TO RegisterService2.register;
        Sequencer_1.E3 TO E_SR.S;
        Sequencer_1.E5 TO E_SR.R;
        Sequencer_1.E7 TO E_SR.S;
        Sequencer_1.E8 TO RegisterService2.unregister;
        Sequencer_1.E10 TO E_SR.R;
        NoServiceAvailable.CNF TO Sequencer_1.Next;
        RegisterService2.doneUnregister TO Sequencer_1.Next;
        RegisterService2.doneRegister TO Sequencer_1.Next;
        FieldsToServiceRequestForm.CNF TO Sequencer_1.Next;
        START.COLD TO SUBL_0.INIT;
        SERVER_1.INITO TO Sequencer_1.Next;
        Sequencer_1.E0 TO RequestOrchestrationForm.requestOrchestator;
        Sequencer_1.E2 TO RequestOrchestrationForm.requestOrchestator;
        Sequencer_1.E4 TO RequestOrchestrationForm.requestOrchestator;
        Sequencer_1.E6 TO RequestOrchestrationForm.requestOrchestator;
        Sequencer_1.E9 TO RequestOrchestrationForm.requestOrchestator;
        RequestOrchestrationForm.responseReceived TO GET_STRUCT_VALUE1.REQ;
        Sequencer_1.E11 TO PUBL_0.REQ;
        SUBL_0.INITO TO PUBL_0.INIT;
      END_CONNECTIONS
      DATA_CONNECTIONS
        FieldsToArrowheadSystem.arrowheadSystem TO FieldsToServiceRequestForm.requesterSystem;
        Service1.arrowheadService TO FieldsToServiceRequestForm.requestedService;
